# B&R Automation Studio project TD52 (part 114)

### Module_HA_IO.var - HalIO IO variables
```iecst
(********************************************************************
* COPYRIGHT -- INNIO Company
********************************************************************
* Package: HAL_IO
* File: HAL_IO.var
* Author: Automatically generated code
* Created: 29.01.2014
* corrected version from 04.09.2017
*********************************************************************
* Variables of package HAL_IO
********************************************************************)
VAR
	EO_FreshOilPump_Dem : BOOL; (*DO Aux FreshOilPump V4.14*)
	tEO_FreshOilPump_Dem : HALioDo_Type; (*DO Aux FreshOilPump V4.14*)
	EO_WasteOilPump_Dem : BOOL; (*DO Aux WasteOilPump V4.14*)
	tEO_WasteOilPump_Dem : HALioDo_Type; (*DO Aux WasteOilPump V4.14*)
	ActFiltAlarm : BOOL; (*DIactivfilteralarm*)
	ActFiltWarn : BOOL; (*DIactivfilterwarning*)
	Actuator2_Rel : BOOL; (*DO:Actuatorreleasecommand*)
	Actuator_Ok : BOOL; (*DI:Actuatorokay*)
	Actuator_Ok_CBV1 : BOOL; (*DI:Actuatorokaycompressorbypassvalve1*)
	Actuator_Ok_CBV2 : BOOL; (*DI:Actuatorokaycompressorbypassvalve2*)
	Actuator_Ok_TV1A : BOOL; (*DI:Actuatorokaythrottlevalve1A*)
	Actuator_Ok_TV1B : BOOL; (*DI:Actuatorokaythrottlevalve1B*)
	Actuator_Ok_TV2A : BOOL; (*DI:Actuatorokaythrottlevalve2A*)
	Actuator_Ok_TV2B : BOOL; (*DI:Actuatorokaythrottlevalve2B*)
	Actuator_Ok_DAI_A : BOOL; (* DI: Actuator ok DAI bank A *)
	Actuator_Ok_DAI_B : BOOL; (* DI: Actuator ok DAI bank B *)
	Actuator_Rel : BOOL; (*DO:Actuatorreleasecommand*)
	AirER_FS : BOOL; (*DIengineroomVEflowswitch*)
	AI_UniAi : ARRAY[0..250] OF INT; (*CustomerIOsystemHAL-connector*)
	AuxErrWarn : BOOL; (*DIauxiliarieserror*)
	AuxFail : BOOL; (*DIauxilariesfailure*)
	AuxOverVoltProt_Ok : BOOL; (*failureovervoltageprotectionauxiliariespowersupply*)
	AuxPoSuMains : BOOL; (*DOauxiliariespowersupplyfrommains*)
	AuxPoSuUPS : BOOL; (*DOauxiliariespowersupplyfromUPS*)
	AuxV_Eng_ok : BOOL; (*DIauxiliariesvoltageengineok*)
	ChC_Heating : BOOL; (*DO Demand charge cooler pre heating*)
	Island_Op : BOOL; (*DO Island operation*)
	Parallel_Op : BOOL; (*DO Mains parallel operation*)
	AuxV_Supply_Ok : BOOL; (*DIauxiliaryvoltagesupplyok*)
	BbBlower : BOOL; (*DO Blow-by Blower*)
	BbBlower_FC_Rdy : BOOL; (*DI Blow-by Blower FC ready *)
	BbBlower_y : INT; (*AO Blow-by Blower Percentage value to FU*)
	BB_Alive : BOOL; (*DIbusbaralive*)
	BB_Dead_MMD : ARRAY[0..2] OF BOOL; (*DIbusbardeadfromMMD*)
	bCAsymDO1 : ARRAY[0..2] OF BOOL; (*Set function of MMDsynch DO1 terminal*)
	bCNMaxDO1 : ARRAY[0..2] OF BOOL; (*Set function of MMDsynch DO1 terminal*)
	bCThermDO1 : ARRAY[0..2] OF BOOL; (*Set function of MMDsynch DO1 terminal*)
	bMMDReadyDO1 : ARRAY[0..2] OF BOOL; (*Set function of MMDsynch DO1 terminal*)
	bOFreqDO1 : ARRAY[0..2] OF BOOL; (*Set function of MMDsynch DO1 terminal*)
	bOVoltDO1 : ARRAY[0..2] OF BOOL; (*Set function of MMDsynch DO1 terminal*)
	bReactMinDO1 : ARRAY[0..2] OF BOOL; (*Set function of MMDsynch DO1 terminal*)
	bShortDO1 : ARRAY[0..2] OF BOOL; (*Set function of MMDsynch DO1 terminal*)
	bSyncCheckMode : ARRAY[0..2] OF BOOL; (*sync mode: check*)
	bSyncDeadBusMode : ARRAY[0..2] OF BOOL; (*sync mode: dead bus*)
	bSyncSlipMode : ARRAY[0..2] OF BOOL; (*sync mode: slip*)
	bUFreqDO1 : ARRAY[0..2] OF BOOL; (*Set function of MMDsynch DO1 terminal*)
	bUVolt2DO1 : ARRAY[0..2] OF BOOL; (*Set function of MMDsynch DO1 terminal*)
	bUVoltDO1 : ARRAY[0..2] OF BOOL; (*Set function of MMDsynch DO1 terminal*)
	bVAsymDO1 : ARRAY[0..2] OF BOOL; (*Set function of MMDsynch DO1 terminal*)
	CA_IgnP_Set : INT; (*AO:timingpoint*)
	CCWP_Op : BOOL; (*DIchargecoolingwaterpumpoperating*)
	ChargeOff_Dem : BOOL; (*DOchargingunitoffdemand*)
	ChC_DemFan1 : BOOL; (*DOchargecoolerdemandfan1*)
	ChC_DemFan2 : BOOL; (*DOchargecoolerdemandfan2*)
	ChC_DemFan3 : BOOL; (*DOchargecoolerdemandfan3*)
	ChC_DemFan4 : BOOL; (*DOchargecoolerdemandfan4*)
	ChC_DemFan5 : BOOL; (*DOchargecoolerdemandfan5*)
	ChC_DemFan6 : BOOL; (*DOchargecoolerdemandfan6*)
	ChC_DemFan7 : BOOL; (*DOchargecoolerdemandfan7*)
	ChC_DemFan8 : BOOL; (*DOchargecoolerdemandfan8*)
	ChC_DemFan9 : BOOL; (*DOchargecoolerdemandfan9*)
	ChC_DemFan10 : BOOL; (*DOchargecoolerdemandfan10*)
	ChC_DemFan11 : BOOL; (*DOchargecoolerdemandfan11*)
	ChC_DemFan12 : BOOL; (*DOchargecoolerdemandfan12*)
	ChC_DemFan13 : BOOL; (*DOchargecoolerdemandfan13*)
	ChC_DemFan14 : BOOL; (*DOchargecoolerdemandfan14*)
	ChC_DemFan15 : BOOL; (*DOchargecoolerdemandfan15*)
	ChC_DemFan16 : BOOL; (*DOchargecoolerdemandfan16*)
	ChC_DemPump : BOOL; (*DOchargecoolerdemandpump*)
	ChC_Failure : BOOL; (*DIchargecoolerfailure*)
	ChC_FanRdy : BOOL; (*DIchargecoolerfanready*)
	ChUnit1_CB_On : BOOL; (*Circuit breaker tripped Charging unit 1*)
	ChUnit2_CB_On : BOOL; (*Circuit breaker tripped Charging unit 2*)
	ChUnit3_CB_On : BOOL; (*Circuit breaker tripped +ENGIA Charging unit 1*)
	ChUnit4_CB_On : BOOL; (*Circuit breaker tripped +ENGIA Charging unit 2*)
	Cnt_GasImp : BOOL; (*DI	Impulsegascounter*)
	Cnt_OilPulse : BOOL; (*DIoilcounter*)
	Cnt_Oil_DC2395 : UINT; (*AIoilcountercircularbuffer*)
	Cnt_Oil_NC150 : INT; (*AIoilcounter*)
	CO2_Alarm : BOOL; (*DOCO2alarm*)
	CO2_Demand : BOOL; (*DICO2demand*)
	CO2_DemCodinox : BOOL; (*DOCO2demandCODINOX*)
	CO2_DevFailure : BOOL; (*DICO2devicefailure*)
	CO2_FanCoOn : BOOL; (*DOCO2demandfan*)
	CO2_FanFailure : BOOL; (*DICO2fanfailure*)
	CO2_MPMode : BOOL; (*DOCO2setCODINOXtomainsparallelmode*)
	CO2_Rdy : BOOL; (*DOCO2ready*)
	CO2_VaClosed : BOOL; (*DICO2valveclosed*)
	CO2_VaCoClose : BOOL; (*DOCO2valvecommandclose*)
	CO2_VaCoOpen : BOOL; (*DOCO2valvecommandopen*)
	CO2_VaFailure : BOOL; (*DICO2valvefailure*)
	CO2_VaLockout : BOOL; (*DIlockoutCO2valve*)
	CO2_VaOpened : BOOL; (*DICO2valveopened*)
	CO2_WD : BOOL; (*DOCO2watchdog*)
	Codinox_Rdy : BOOL; (*DICODINOXreadyforoperation*)
	CO_Alarm : BOOL; (*DICOalarm*)
	CO_PreAlarm : BOOL; (*DICOprealarm*)
	CP_CBTrip : BOOL; (*DImoduleand/orinterfacecontrolpanel-circuitbreakertripped*)
	CtrGenPF_Set : INT; (*AOGenerator???*)
	CtrTR_Heater_Set : INT; (*AO->Controlleroutput*)
	Ctr_ChCHP_Set : INT; (*AOchargetemperaturecoolerhighpressurecontrolvalve*)
	Ctr_ChCV_Set : INT; (*AOchargetemperaturecoolerventilation*)
	Ctr_ChC_Set : INT; (*AOchargetemperaturecoolercontrolvalve*)
	Ctr_CustOut : ARRAY[0..45] OF INT; (*AI: new output channel für direct usage of customized controllers on HAL*)
	Ctr_ECW_Set : INT; (*AOenginecoolingewatertemp.controlvalvesetpoint*)
	Ctr_EC_Set : INT; (*AOheatwaterreturntemperaturecontrolvalveemergencycooler*)
	Ctr_GC_Set : INT; (*AO Gas compressor*)
	Ctr_Gen_Set : INT; (*AOGenerator???*)
	Ctr_HWRe_Set : INT; (*AOheatwaterreturntemperaturecontrolvalve*)
	Ctr_HWSu_Set : INT; (*AOheatwatersupplytemperaturecontrolvalve*)
	CustAnaIn : ARRAY[0..120] OF INT; (*ReplacementforRAN_KANAL...*)
	CustAnaOut : ARRAY[0..60] OF INT; (*newreserveoutputchannel(likeANA.RAN1forinputs)*)
	CustDigIn : ARRAY[0..200] OF BOOL; (*new,reservedforProjectspecificuse*)
	CustDigOut : ARRAY[0..150] OF BOOL; (*ConnectiontoHAL*)
	P0_BLOCK_DEIE : BOOL; (*DI : Installed 1/0 switch *) (*OldName:Cust_switch_erdf PV;Cycle:2;*)
	CV_Eng_Low : BOOL; (*Control voltage min*)
	CV_TCA_Low : BOOL; (*Control voltage min*)
	C_CB_EDC : BOOL; (*DIcustomercircuitbreaker(engine*)
	C_CB_ESL : BOOL; (*DIcustomercircuitbreaker(engine*)
	C_CB_Off : BOOL; (*DIcustomercircuitbreakeropened*)
	C_CB_On : BOOL; (*DIcustomercircuitbreakerclosed*)
	DAI_V_Dem : BOOL; (* DO: DAI shut off valve open command *)
	DAI_V_Opened : BOOL; (* DI: DAI shut off valve position opened *)
	DAI_V_Closed : BOOL; (* DI: DAI shut off valve position closed *)
	DAI_Dem : BOOL; (*DO: Demand DAI actuator bank A and B *)
	Pos_DAI_Set_A : INT; (* AO: Position setpoint DAI control valve bank A *)
	Pos_DAI_Act_A : INT; (* AI: Position feedback DAI control valve bank A *)
	Pos_DAI_Set_B : INT; (* AO: Position setpoint DAI control valve bank B *)
	Pos_DAI_Act_B : INT; (* AI: Position feedback DAI control valve bank B *)
	DAI_CB_On : BOOL; (* DAI curcuit breaker feedback signal *)
	DemandBB : BOOL; (*demandbusbar*)
	DemEngOpExt : BOOL; (*externaldemandofengineoperation*)
	DemFlair : BOOL; (*DI	Demandgascompressorforflairoperationmode*)
	DemPurgeER : BOOL; (*DOdemandroomVEforpurgecycle*)
	DiffPrct : BOOL; (*DI:Differentialprotection*)
	DI_Dem_EU_Block : BOOL; (*externalrequestfromutility(evu*)
	DI_Dem_P_Red_EVU_Stage1 : BOOL; (*externalrequestfromutility(evu*)
	DI_Dem_P_Red_EVU_Stage2 : BOOL; (*externalrequestfromutility(evu*)
	DI_Dem_P_Red_EVU_Stage3 : BOOL; (*externalrequestfromutility(evu*)
	DI_Dem_P_Red_EVU_Stage4 : BOOL; (*externalrequestfromutility(external,vintagestyledutilisation*)
	DI_Dem_P_Red_EVU_Stage5 : BOOL; (*externalrequestfromutility(external,vintagestyledutilisation*)
	DI_UniDi : ARRAY[0..250] OF BOOL; (*CustomerIOsystemHAL-connector*)
	DO_Eng_Block_EVU : BOOL; (*acknowlegerequestfromutility(evu*)
	DO_P_Red_EVU_Stage0 : BOOL; (*acknowlegerequestfromutility(evu*)
	DO_P_Red_EVU_Stage1 : BOOL; (*acknowlegerequestfromutility(evu*)
	DO_P_Red_EVU_Stage2 : BOOL; (*acknowlegerequestfromutility(evu*)
	DO_P_Red_EVU_Stage3 : BOOL; (*acknowlegerequestfromutility(evu*)
	DO_P_Red_EVU_Stage4 : BOOL; (*acknowlegerequestfromutility(external,vintagestyledutilisationfeedback*)
	DO_P_Red_EVU_Stage5 : BOOL; (*acknowlegerequestfromutility(external,vintagestyledutilisationfeedback*)
	DPr_AirFilt : INT; (*engineairinletfilterdifferencepressure[bar]*)
	DPr_AirFilt_A : INT; (*engineairinletfilterdifferencepressureA[bar]*)
	DPr_AirFilt_B : INT; (*engineairinletfilterdifferencepressureB[bar]*)
	DPr_InAirFiltERV_Hi : BOOL; (*air inlet filter difference pressure high - engine room ventilation*) (*V04.04.00.00*)
	DPr_OilSkid_FiltHP_DE_Hi : BOOL; (*DI OilSkid heater - circuit breaker*)
	DPr_OilSkid_FiltHP_NDE_Hi : BOOL; (*DI OilSkid difference pressure - oil high pressure filter to NDE bearing*)
	DPr_OilSkid_FiltLP_Hi : BOOL; (*DI OilSkid difference pressure - oil low pressure filter*)
	EarthCB_Off : BOOL; (*DIearthcircuitbreakeropened,francecountryspecific*)
	ECWP1Dem : BOOL; (*DOenginecoolingwaterpump1demand*)
	ECWP2Dem : BOOL; (*DOenginecoolingwaterpump2demand*)
	ECWPrehV_Opened : BOOL; (*DIenginecoolingwaterpreheatingvalveopened*)
	ECWP_FC_Rdy : BOOL; (*DIenginecoolingwaterpumpfrequencyconverterreadyforoperation*)
	ECWP_Op : BOOL; (*DIenginecoolingwaterpumpoperating*)
	ECWP_PreH_CB_On : BOOL; (*Failure Engine jacket water Preheating pump*)
	ECWP_PreH_Dem : BOOL; (*DOenginecoolingwaterpreheatingpumpdemand*)
	ECWP_Service : BOOL; (*Service Pump Engine jacket water*)
	ECWP_Service_CB_On : BOOL; (*Failure Service Pump Engine jacket water*)
	ECWP_Service_COn : BOOL; (*Demand Service Pump Engine jacket water*)
	ECWV_Fail : BOOL; (*Failure Flap Preheating Engine jacket water*)
	ECW_DemBpP : BOOL; (*DOdemandenginecoolingwaterbypasspump(AMOT*)
	ECW_DemBpV : BOOL; (*DOdemandenginecoolingwaterbypassvalve(AMOT*)
	ECW_PreH1Dem : BOOL; (*DOenginecoolingwaterpreheating1demand*)
	ECW_PreH2Dem : BOOL; (*DOenginecoolingwaterpreheating2demand*)
	ECW_PreH3Dem : BOOL; (*DOenginecoolingwaterpreheating3demand*)
	ECW_PreHV_Closed : BOOL; (*DIenginecoolingwaterpreheatingvalvestatusclosed*)
	ECW_PreHV_CoClose : BOOL; (*DOenginecoolingwaterpreheatingvalve-commandclose*)
	ECW_PreHV_CoOpen : BOOL; (*DOenginecoolingwaterpreheatingvalve-commandopen*)
	ECW_PreHV_Opened : BOOL; (*DIenginecoolingwaterpreheatingvalvestatusopened*)
	ECW_PreH_Dem : BOOL; (*DOenginecoolingwaterpreheatingdemand*)
	EC_DemFan1 : BOOL; (*DOemergencycoolerdemandfan1*)
	EC_DemFan2 : BOOL; (*DOemergencycoolerdemandfan2*)
	EC_DemFan3 : BOOL; (*DOemergencycoolerdemandfan3*)
	EC_DemFan4 : BOOL; (*DOemergencycoolerdemandfan4*)
	EC_DemFan5 : BOOL; (*DOemergencycoolerdemandfan5*)
	EC_DemFan6 : BOOL; (*DOemergencycoolerdemandfan6*)
	EC_DemFan7 : BOOL; (*DOemergencycoolerdemandfan7*)
	EC_DemFan8 : BOOL; (*DOemergencycoolerdemandfan8*)
	EC_DemFan9 : BOOL; (*DOemergencycoolerdemandfan9*)
	EC_DemFan10 : BOOL; (*DOemergencycoolerdemandfan10*)
	EC_DemFan11 : BOOL; (*DOemergencycoolerdemandfan11*)
	EC_DemFan12 : BOOL; (*DOemergencycoolerdemandfan12*)
	EC_DemFan13 : BOOL; (*DOemergencycoolerdemandfan13*)
	EC_DemFan14 : BOOL; (*DOemergencycoolerdemandfan14*)
	EC_DemFan15 : BOOL; (*DOemergencycoolerdemandfan15*)
	EC_DemFan16 : BOOL; (*DOemergencycoolerdemandfan16*)
	EC_DemPump : BOOL; (*DOemergencycoolerdemandpump*)
	EC_Failure : BOOL; (*DIemergencycoolerfailure*)
	EGScavStart_Ext : BOOL; (*DIexhaustgasscavengingstartfromexternal*)
	EG_BoVaClosed : BOOL; (*DIexhaustgasboilervalveclosed*)
	EG_BoVaClosedTo : BOOL; (*DIexhaustgasboilervalveclosedtorch*)
	EG_BoVaCoClose : BOOL; (*DOexhaustgasboilervalvecommandclose*)
	EG_BoVaCoOpen : BOOL; (*DOexhaustgasboilervalvecommandopen*)
	EG_BoVaFailure : BOOL; (*DIexhaustgasboilervalvefailure*)
	EG_BoVaOpened : BOOL; (*DIexhaustgasboilervalveopened*)
	EG_BypassDemand : BOOL; (*DIdemandexhaustgasbypass*)
	EG_ByVaClosed : BOOL; (*DIexhaustgasbypassvalveclosed*)
	EG_ByVaClosedTo : BOOL; (*DIexhaustgasbypassvalveclosedtorch*)
	EG_ByVaCoClose : BOOL; (*DOexhaustgasbypassvalvecommandclose*)
	EG_ByVaCoOpen : BOOL; (*DOexhaustgasbypassvalvecommandopen*)
	EG_ByVaFailure : BOOL; (*DIexhaustgasbypassvalvefailure*)
	EG_ByVaOpened : BOOL; (*DIexhaustgasbypassvalveopened*)
	EleStarter_Dem : BOOL; (*DOelectricstarterdemand*)
	EmStop_MC : BOOL; (*DI emergency stop push button - module control panel (+A/+MC)*) (* *) (*V04.04.00.00*)
	EmStop_M : BOOL; (*DI emergency stop push button - module interface panel (+M)*) (* *) (*V04.04.00.00*)
	EmStop_ST : BOOL; (*DI emergency stop push button - master control panel (+ST)*) (* *) (*V04.04.00.00*)
	EmStop_IS : BOOL; (*DI emergency stop push button - interlock panel (+IS)*) (* *) (*V04.04.00.00*)
	EmStop_TS : BOOL; (*DI emergency stop push button - thermal reactor control panel (+TS)*) (* *) (*V04.04.00.00*)
	EmStop_GENI : BOOL; (*DI emergency stop push button - generator interface panel (+GENI)*) (* *) (*V04.04.00.00*)
	EmStop_ENGIA : BOOL; (*DI emergency stop push button - engine interface panel bank A (+ENGIA)*) (* *) (*V04.04.00.00*)
	EmStop_TCMI : BOOL; (*DI emergency stop push button - turbocharger module interface panel (+TCMI)*) (* *) (*V04.04.00.00*)
	EmStop_JWMI : BOOL; (*DI emergency stop push button - jacket water module interface panel (+JWMI)*) (* *) (*V04.04.00.00*)
	EmStop_OILMI : BOOL; (*DI emergency stop push button - oil module interface panel (+OILMI)*) (* *) (*V04.04.00.00*)
	EmStop_SCR : BOOL; (*DI emergency stop push button - exhaust gas after treatment control panel (+SCR)*) (* *) (*V04.04.00.00*)
	EmStop_TCMSCAV : BOOL; (*DI emergency stop push button - exhaust gas scavenging system (+TCMSCAV)*) (* *) (*V04.07.00.00*)
	EngDemIsland : BOOL; (*DIenginedemandforislandoperation*)
	ENGIA_UPS_CB_On : BOOL; (*Circuit breaker tripped supply UPS +TCAI --> +ENGIA*)
	EngStartFailure : BOOL; (*DIenginestartfailure*)
	EngTurn : BOOL; (*DIengineturnequipmentactive*)
	EngTurn2 : BOOL; (*Failure engine turning device*)
	Eng_Aux_Dem_CDR : BOOL; (*engineauxiliariesdemandwithcooldownrun*)
	Eng_Aux_Dem_CDR2 : BOOL; (*engineauxiliariesdemandwithcooldownrun*)
	Eng_Aux_Dem_CDR3 : BOOL; (*engineauxiliariesdemandwithcooldownrun*)
	Eng_Dem : BOOL; (*enginedemandedforMSY*)
	Eng_Dem_EPS_Ext : BOOL; (*enginedemandemergencypowersupplyfromexternal*)
	Eng_Rdy_Rem : BOOL; (*ReadyforRemoteOperation*)
	Eng_Ready : BOOL; (* DO: aggregate available (PLC run) 							*)
	Eng_Run : BOOL; (*enginerunning*)
	Eng_Run_Sy : BOOL; (*engineruning-synchronization*)
	Eng_SUExc_Rel : BOOL; (*start-upexcitationrelease*)
	EOF_DiffMax : BOOL; (*DI:Oildifferencepressuremaximum*)
	EOF_PreheatRel : BOOL; (*DO:Releaseoilpreheatingvalve*)
	EOP1AC_CB_trip : BOOL; (*DIengineoilpump1ACcircuitbreakertrip*)
	EOP1AC_Dem : BOOL; (*DOengineoilpump1AC*)
	EOP1DC_Dem : BOOL; (*DOengineoilpump1DC*)
	EOP_DemExt : BOOL; (*DIengineoilpumpdemandfromexternal*)
	EOP_FC_Rdy : BOOL; (*DI:engineoilpumpfreq.converteroperation/ready*)
	EOP_FC_Set : INT; (*AO:Setpointfrequencyconvertermotoroilpumpprelubrication,[100%=1.0]*)
	EOP_On : BOOL; (*DO:Engineoilpump,NPO602*)
	EOP_Op : BOOL; (*DIengineoilpumpoperating*)
	EOVal_DemOpen : BOOL; (*DOengineoilrefillvalvedemandopen*)
	EOVal_LT_Set : INT; (*Control signal Regulator valve NT Oil circuit*)
	EO_Level : INT; (*EngineOilPanLevel*)
	EO_Level_Hi : BOOL; (*DIengineoillevelhighfromlevelswitch*)
	EO_Level_Lo : BOOL; (*DIengineoillevellowfromlevelswitch*)
	EO_Preheat1 : BOOL; (*DO:engineoilpreheatingelement1*)
	EO_Preheat2 : BOOL; (*DO:engineoilpreheatingelement2*)
	EO_Preheat3 : BOOL; (*DO:engineoilpreheatingelement3*)
	EO_Quality : INT; (*AI:Oilqualitysensor,QTOil1/AI_*)
	EO_Refill : BOOL; (*DIengineoilrefillONfromlevelswitch*)
	EO_Supply_Fail : BOOL; (*DI:Oilsupplyfailure*)
	ERDF_BLOCK : BOOL; (* DO: Block von ERDF *) (* OldName: DI_EVU_BLOCK ; Cycle: 5 *)
	ERV_Op : BOOL; (*DIengineroomventilationoperating/airflowok*)
	ERV_InlAir_Op : BOOL; (*DIengineroominletairventilationoperating/airflowok*)
	ERV_OutlAir_Op : BOOL; (*DIengineroomoutletairventilationoperating/airflowok*)
	ER_DoorClosed : BOOL; (*DI engine room doors closed*)
	ER_Ext_Err : BOOL; (*DIengineroomVEfailure*)
	ER_InlAir_Ext_Err : BOOL; (*DIengineroominletairVEfailure*)
	ER_OutlAir_Ext_Err : BOOL; (*DIengineroomoutletairVEfailure*)
	ER_FC_Set : INT; (*AOengineroomfrequencyconvertersetpoint[%]*)
	EU_RM_BLOCK : BOOL; (*DO:	Separateunitofutilityandofactivenetwork*)
	EVU_PowerSet3Dem : BOOL; (*demandmoduleblockedbyutility*)
	ExCo_Rel : BOOL; (*DOexternalcoolerrelease*)
	FastAO_KN_A : INT; (*fastanalogoutputsignalsforvalidation*)
	FastAO_KN_B : INT; (*fastanalogoutputsignalsforvalidation*)
	FireAlarm : BOOL; (*DIfirealarm*)
	FlairRdy : BOOL; (*DI	Flairready*)
	Flow_Gen_Lube : BOOL; (*generatorlubricationfailure*)
	Flow_HW_Lo : BOOL; (*DIheatwaterflowlow*)
	Flow_OilSkid_DE : INT; (*AI OilSkid oil flow to DE bearing *)
	Flow_OilSkid_NDE : INT; (*AI OilSkid oil flow to NDE bearing (G.03-FI-003)*)
	FS_ECW : BOOL; (*DIflowswitchenginecoolingwater*)
	F_GenBear_DE1 : INT; (*vibration generator bearing drive end 1*) (*Oldname:AI_v_GenBearDE1;Cycle:5;*)
	F_GenBear_DE2 : INT; (*vibration generator bearing drive end 2*) (*Oldname:AI_v_GenBearDE2;Cycle:5;*)
	F_GenBear_NDE1 : INT; (*vibration generator bearing non drive end 1*) (*Oldname:AI_v_GenBearNDE1;Cycle:5;*)
	F_GenBear_NDE2 : INT; (*vibration generator bearing non drive end 2*) (*Oldname:AI_v_GenBearNDE2;Cycle:5;*)
	F_MMD : ARRAY[0..2] OF UINT; (* frequency multi measure device*)
	F_MMD_LimHi : ARRAY[0..2] OF BOOL; (*generatorfrequencytoohigh*)
	F_MMD_LimLo : ARRAY[0..2] OF BOOL; (*generatorfrequencytoolow*)
	F_MMD_Synch1 : ARRAY[0..2] OF UINT; (* Frequency Sync-network 1 *)
	F_MMD_Synch2 : ARRAY[0..2] OF UINT; (* Frequency Sync-network 2 *)
	F_N_DI_Dec : BOOL; (*synch.digitalindecreasespeed*)
	F_N_DI_Inc : BOOL; (*synch.digitalinincreasespeed*)
	GasAlarm : BOOL; (*DIgasalarm*)
	GasPreAlarm : BOOL; (*DIgasprealarm*)
	GCB_AGO : BOOL; (*DIallothergeneratorcircuitbreakeroff*)
	GCB_COf : BOOL; (*commandgcboff*)
	GCB_COn : BOOL; (*commandgcbon*)
	GCB_DRM : BOOL; (*DIgeneratorcircuitbreakerdemandMCBclosingreturntomains*)
	GCB_DSY : BOOL; (*DIgeneratorcircuitbreakerdemandsynchronization(synchline*)
	GCB_DVM : BOOL; (*voltagematchingforsynchronization*)
	GCB_DVS : BOOL; (*generatorcircuitbreakerdemandvoltageselection*)
	GCB_Earth : BOOL; (*DIgeneratorcircuitbreakerpositionearth*)
	GCB_EDC : BOOL; (*generatorcircuitbreakerenginedemandclose*)
	GCB_ESL : BOOL; (*generatorcircuitbreakerstatuslocked*)
	GCB_MDL : BOOL; (*DIgeneratorcircuitbreakermasterdemandlock(forclosingotherGCBtodeadBB*)
	GCB_MRC : BOOL; (*DIgeneratorcircuitbreakermasterreleaseclose(todeadbusbar*)
	GCB_Off : BOOL; (*DIgeneratorcircuitbreakeropened*)
	GCB_OGP : BOOL; (*DIgeneratorcircuitbreakerothergeneratorparallel*)
	GCB_On : BOOL; (*generatorcircuitbreakerclosed*)
	GCB_On_ReturnSign : BOOL; (*ReleaseforUnitrolAVR*)
	GCB_OpF : BOOL; (*generatorcircuitbreakeropeningfailure*)
	GCB_Rac : BOOL; (*DIgeneratorcircuitbreakerrackedin*)
	GCB_Rdy : BOOL; (*DIgeneratorcircuitbreakerready(forclose*)
	GCB_Rel : BOOL; (*generatorcircuitbreakerreleaseclosing*)
	GCB_RI : BOOL; (*DIgeneratorcircuitbreakerreelaseisland*)
	GCB_RSP : BOOL; (*generatorcircuitbreakerreleasesynchpulse*)
	GCB_RT : BOOL; (*generatorcircuitbreakerreleasetrip*)
	GCB_RUC : BOOL; (*generatorcircuitbreakerreleaseundervoltagecoil*)
	GCB_SM1 : BOOL; (*DIgeneratorcircuitbreakeroutputsignalmonitoring1*)
	GCB_SM2 : BOOL; (*DIgeneratorcircuitbreakercontactsignalmonitoring2*)
	GCB_SOn : BOOL; (* DO: Generator switch is on 									*)
	GenCtrResetSp : BOOL; (*Generator controller reset setpoint*)
	GenCtr_CktBkr_Trip : BOOL; (*generatorcicuitbreakeroff*)
	GenDeexitDem : BOOL; (*DOgeneratordeexitationdemand*)
	GenIF_CB_On : BOOL; (*Circuit breaker tripped supply +TCAI --> +GENI*)
	GenPrctTrip : BOOL; (*DI:Generatorprotectiontrip*)
	Gen_DVM : BOOL; (*Generatorvoltagematchingoutput(LeroySomer*)
	Gen_Exc_Off : BOOL; (*de-excitation*)
	Gen_LO_CoolingSys_Fail : BOOL; (*generatorlubeoilcoolingsystemfailure*)
	Gen_PreHDem : BOOL; (*DOGeneratorpreheatdemand*)
	Gen_RVM : BOOL; (*DIgeneratorreleasevoltagematching(leroysomer*)
	Gen_T_In : INT; (*actualvaluegeneratorinlettemperature*)
	Gen_T_In2 : INT; (*actualvaluegeneratorinlettemperature2*)
	GF_OilSystem : BOOL; (*DI general failure oil system*) (*OldName:newPV; Cycle:5*) (*STM*)
	GndFailure : BOOL; (*DI:earthfailure*)
	GnlTrip : BOOL; (*DOenginegeneraltrip*)
	GnlWarning : BOOL; (*DOenginegeneralwarning*)
	GrC_DCon : BOOL; (* DO: FALSE = Disconnect from Grid due to GridCode Event*)
	GT1_1_SafeDevice : BOOL; (*DO	Gassafetydevice1line1*)
	GT1_1_SafeDevOK : BOOL; (*DIGassafetydevice1line1*)
	GT1_2_SafeDevice : BOOL; (*DO	Gassafetydevice1line2*)
	GT1_2_SafeDevOK : BOOL; (*DI	Gassafetydevice2line2*)
	GT1_3_SafeDevice : BOOL; (*DO	Gassafetydevice1line3*)
	GT1_3_SafeDevOK : BOOL; (*DIGassafetydevice3line3*)
	GT1_4_SafeDevice : BOOL; (*DO	Gassafetydevice1line4*)
	GT1_4_SafeDevOK : BOOL; (*DIGassafetydevice4line4*)
	GT1_SafeDevice : BOOL; (*DO	Gassafetydevice1*)
	GT1_SafeDevOK : BOOL; (*DI	Gassafetydevice1*)
	GT2_SafeDevice : BOOL; (*DO	Gassafetydevice2*)
	GT2_SafeDevOK : BOOL; (*DI	Gassafetydevice2*)
	GT3_SafeDevOK : BOOL; (*DI	Gassafetydevice3*) (*SAFETY PLC*) (*V04.14.00.00*)
	GT4_SafeDevOK : BOOL; (*DI	Gassafetydevice4*) (*SAFETY PLC*) (*V04.14.00.00*)
	GT_AirSupply_LoLo : BOOL; (*DI FALSE = compressed air supply pressure for gas train too low - error*) (*Oldname : DI_GT_AirSupply_LoLo Cyclic: 2; *)
	GT1_1_BackFireDev : BOOL; (*DIAntibackfiredevice1line1*)
	GT1_2_BackFireDev : BOOL; (*DIAntibackfiredevice1line2*)
	GT1_3_BackFireDev : BOOL; (*DIAntibackfiredevice1line3*)
	GT1_4_BackFireDev : BOOL; (*DIAntibackfiredevice1line4*)
	PCbComp_BackFireDev : BOOL; (*DIAntibackfire device prechamper before compressor*)
	PCaComp_BackFireDev : BOOL; (*DIAntibackfire device prechamper after compressor*)
	GT_BackFireDev : BOOL; (*DI	Antibackfiredevice*)
	GT_CalibrateActive : BOOL; (*DI	CalibrationGasanalysis*)
	GT_CH4 : INT; (*IF653CH4content	*)
	GT_CV : INT; (*AI	Calorificvalue*)
	GT_FlairFail : BOOL; (*DI	Flarefailure*)
	GT_Flap1_Close : BOOL; (*DO	Closegasflap1*)
	GT_Flap1_Closed : BOOL; (*DI	Gasflap1closed(Feedback*)
	GT_Flap1_Open : BOOL; (*DO	Opengasflap1*)
	GT_Flap1_Opened : BOOL; (*DI	Gasflap1opened(Feedback*)
	GT_Flap2_Close : BOOL; (*DO	Closegasflap2*)
	GT_Flap2_Closed : BOOL; (*DI	Gasflap2closed(Feedback*)
	GT_Flap2_Open : BOOL; (*DO	Opengasflap2*)
	GT_Flap2_Opened : BOOL; (*DI	Gasflap2opened(Feedback*)
	GT_FlareOpMod : BOOL; (*DI	Flareinoperationalmode*)
	GT_GC_Dem : BOOL; (*DO	Demandgascompressor*)
	GT_GC_Fail : BOOL; (*DI	Gascompressorfailure*)
	GT_O2 : INT; (*IF656O2content	*)
	GT_RelFlair : BOOL; (*DO	Releaseflare*)
	GT_SelectRatioMix : BOOL; (*DI: Digital input to select gas mixing (1-3 or 1_2-3)*)
	GT_TypSwitch : BOOL; (*DI	Gastypeswitchtosecondgas*)
	GV1Mega_Open : BOOL; (*DO	Openmegagasvalve1*)
	GV1_1_Open : BOOL; (*DO	opengasvalve1_1(GASV1_1*)
	GV1_2_Open : BOOL; (*DO	opengasvalve1_1(GASV1_2*)
	GV1_Open : BOOL; (*DO	opengasvalve1*)
	GV2Mega_Open : BOOL; (*DO	Openmegagasvalve2*)
	GV2_Open : BOOL; (*DO	opengasvalve2*)
	GV3_Open : BOOL; (*DO	opengasvalve3*) (*SAFETY PLC*) (*V04.14.00.00*)
	GV4_Open : BOOL; (*DO	opengasvalve4*) (*SAFETY PLC*) (*V04.14.00.00*)
	GT1_GV1_Open : BOOL; (*DO Gastrain1 - Gasvalve 1*) (*SAFETY PLC*) (*V04.14.00.00*)
	GT1_GV2_Open : BOOL; (*DO Gastrain1 - Gasvalve 2*) (*SAFETY PLC*) (*V04.14.00.00*)
	GT2_GV1_Open : BOOL; (*DO Gastrain2 - Gasvalve 1*) (*SAFETY PLC*) (*V04.14.00.00*)
	GT2_GV2_Open : BOOL; (*DO Gastrain2 - Gasvalve 2*) (*SAFETY PLC*) (*V04.14.00.00*)
	GT3_GV1_Open : BOOL; (*DO Gastrain3 - Gasvalve 1*) (*SAFETY PLC*) (*V04.14.00.00*)
	GT3_GV2_Open : BOOL; (*DO Gastrain3 - Gasvalve 2*) (*SAFETY PLC*) (*V04.14.00.00*)
	GT4_GV1_Open : BOOL; (*DO Gastrain4 - Gasvalve 1*) (*SAFETY PLC*) (*V04.14.00.00*)
	GT4_GV2_Open : BOOL; (*DO Gastrain4 - Gasvalve 2*) (*SAFETY PLC*) (*V04.14.00.00*)
	GV_Rel : BOOL; (*DO	Releasegasvalves*)
	Horn : BOOL; (*DOhorn*)
	Horn_Trip : BOOL; (*DOhornengineshutdown*)
	Horn_Warning : BOOL; (*DOhornwarning*)
	Humidity_AirIn : INT;
	HWP_Dem : BOOL; (*DOheatingwaterpumpdemand*)
	HWP_Op : BOOL; (*DIheatingwaterpumpoperating*)
	IFCP_CBTrip : BOOL; (*DIinterfacecontrolpanel-circuitbreakertripped*)
	Ign2_Run_Hal : BOOL; (*DI:Ignitionsystemdoublerunning*)
	Ign_Dem : BOOL; (*demandignition*)
	Ign_OverspeedRelay : BOOL; (*DI:Overspeedrelay*)
	Ign_Run_Hal : BOOL; (*DI:Ignitionsystemrunning*)
	Imp_OpHour : BOOL; (*impulseforoperationhourcounter*)
	InAirER_Fan1DemOn : BOOL; (*DOdemandairinletventilator1*)
	InAirER_Fan2DemOn : BOOL; (*DOdemandairinletventilator2*)
	InAirER_Lou1DemOpen : BOOL; (*DOdemandopenairinletlouver1*)
	InAirER_Lou1Opened : BOOL; (*DIintakeairengineroomlouver1open*)
	InAirER_Lou2DemOpen : BOOL; (*DOdemandopenairinletlouver2*)
	InAirER_Lou2Opened : BOOL; (*DIintakeairengineroomlouver2open*)
	DemERVentInLou_Cust : BOOL; (*DO inlet louvers demand for customer*)
	IsoCB_Off : BOOL; (*DIdisconnectingcircuitbreakeropened,francecountryspecific*)
	I_Avg : ARRAY[0..2] OF INT; (*IF513gen.currentaveragev.	*)
	I_Diff : BOOL; (*generatordifferentialprotectiontrip*)
	I_L1 : ARRAY[0..2] OF INT; (*PhasecurrentgeneratorI1*)
	I_L2 : ARRAY[0..2] OF INT; (*PhasecurrentgeneratorI2*)
	I_L3 : ARRAY[0..2] OF INT; (*PhasecurrentgeneratorI3*)
	I_MMD_Asy : ARRAY[0..2] OF BOOL; (*generatorcurrentnegativesequencetoohigh*)
	I_MMD_LimHi : BOOL; (*MMD:overloadshortcircuit*)
	I_MMD_Neutr_LimHi : ARRAY[0..2] OF BOOL; (*generatorneutralcurrenttoohigh*)
	KLS90_1 : INT; (*AI:KLS90sensor1signal*)
	KLS90_2 : INT; (*AI:KLS90sensor1signal*)
	Lam_Act : INT; (*actualLambdavalue*)
	LOS_Dem : BOOL; (*Generatordemandlubeoilsystem*)
	LeroySomer_AuxContactor : BOOL; (*LEROY-SOMERAuxiliaryContactor*)
	Lev_OilSkid_Sump_Hi : BOOL; (*DI OilSkid oil in safety sump *)
	Lev_OilSkid_Tank : INT; (*AI OilSkid tank level*)
	LineCB_On : BOOL; (*DIlinecircuitbreakerclosed*)
	Lock_C_MCB : BOOL; (*lockcustomermainscircuitbreaker*)
	LSL_In : INT; (*AIloadsharingline*)
	LSL_Out : INT; (*AOloadsharingline*)
	LS_Dem : BOOL; (*DOloadsheddingdemand*)
	L_ECW_Lo : BOOL; (*DIenginecoolingwaterlevellow*)
	L_ECW_LoLo : BOOL; (*DIenginecoolingwaterlevellowlow*)
	L_FreshOilTank_Lo : BOOL; (*DIfreshoiltanklevellow*)
	L_FreshOilTank_Hi : BOOL; (*DI fresh oil tank level high*) (*OldName:newPV; Cycle:5*) (*STM*)
	Leak_FreshOilPump : BOOL; (*DI leakage fresh oil pump*) (*OldName:newPV; Cycle:5*) (*STM*)
	Leak_FreshOilTank : BOOL; (*DI leakage fresh oil tank*) (*OldName:newPV; Cycle:5*) (*STM*)
	Leak_WasteOilPump : BOOL; (*DI leakage waste oil pump*) (*OldName:newPV; Cycle:5*) (*STM*)
	Leak_WasteOilTank : BOOL; (*DI leakage waste oil tank*) (*OldName:newPV; Cycle:5*) (*STM*)
	L_InMa_Hi : BOOL; (*DIwateringressintoinletmanifold*)
	L_InMa_NotHi : BOOL; (*DIwateringressintoinletmanifoldnegated*)
	L_OilSump3Hi : BOOL; (*DIleveloilsump3high*)
	L_OilSump2Hi : BOOL; (*DIleveloilsump2high*)
	L_OilSumpHi : BOOL; (*DIleveloilsumphigh*)
	L_WasteOilTank_Hi : BOOL; (*DIwasteoiltanklevelhigh*)
	MainGV_Rel : BOOL; (*DOmaingasvalverelease*)
	MainsStartDevDem : BOOL; (*DOmainsstartdevicedemand*)
	MainsStartDevFail : BOOL; (*DImainsstartdevicefailure*)
	MainsStartDevOk : BOOL; (*DImainsstartingdeviceOK*)
	MCB_COf : BOOL; (*commandmcboff*)
	MCB_COn : BOOL; (*mainscircuitbreakercomandon*)
	MCB_DcpQu_SetEUCOf : BOOL; (* DI: reset decoupling quickly from EU (ERDF) *) (*OldName:DI_RFDemMCBoff PV;Cycle:2;*)
	MCB_DcpQu_SetEUCOn : BOOL; (* DI: set decoupling quickly from EU (ERDF) *) (*OldName:DI_SFDemMCBoff PV;Cycle:2;*)
	MCB_Dcp_SetEUCOf : BOOL; (* DI: rest requirement decoupling from EU(ERDF),DIs *) (*OldName:DI_RDemandMCBoff PV;Cycle:2;*)
	MCB_Dcp_SetEUCOn : BOOL; (* DI: set requirement  decoupling from EU(ERDF),DIs *) (*OldName:DI_SDemandMCBoff PV;Cycle:2;*)
	MCB_DVS : BOOL; (*mainscircuitbreakerdemandvoltageselection*)
	MCB_EDF_SOn : BOOL; (* DO: feedback Engine off get  								*)
	MCB_Off : BOOL; (*DImainscircuitbreakeropened*)
	MCB_OL : BOOL; (*DImainscircuitbreakeroverload*)
	MCB_On : BOOL; (*SS447NetzschalterEIN*)
	MCB_Rac : BOOL; (*DImainscircuitbreakerrackedin*)
	MCB_Rdy : BOOL; (*DImainscircuitbreakerready(forclose*)
	MCB_Rel_Sync : BOOL; (* DI: release synchronization from EU(ERDF) *) (*OldName:DI_ReleaseMCBon PV;Cycle:2;*)
	MCB_Rel_Sync_SOn : BOOL; (* DO: releas decoupling quickly from EU (ERDF)  				*)
	MCB_Rem : BOOL; (*DImainscircuitbreakerremote(operatingmode*)
	MCB_RSP : BOOL; (*mainscircuitbreakerreleasesynchpulse*)
	MCB_RT : BOOL; (*mainscircuitbreakerreleasetrip*)
	MCB_SM : BOOL; (*DImainscircuitbreakersignalmonitoring*)
	MCB_SOn : BOOL; (* DO: receive requested Command form machine 					*)
	MCP_CBTrip : BOOL; (*DImodulecontrolpanel-circuitbreakertripped*)
	MGT_BOV : BOOL; (*DO BlowOff valve*) (*Oldname: DO_MGT_BOV; Cycle:5; *)
	MGT_DBOV : BOOL; (* DO Main gas train dome blow off valve *)
	MMD_FW_Version : ARRAY[0..2] OF UINT; (* program version MMD firmware *)
	MnsOk : BOOL; (*DImainsok	*)
	MnsOk_C13100 : BOOL; (*DImainsokC13.100monitoringdevice,francecountryspecific*)
	MnsOk_GTE : BOOL; (*DImainsokGTEmonitoringdevice,francecountryspecific*)
	MnsOk_TGS : BOOL; (*DImainsokTGSmonitoringdevice,francecountryspecific*)
	Mns_MDF : BOOL; (*DImainsmonitoringdevicefailure*)
	MonitoringOn : BOOL; (*DOmonitoringonpulse(safetyloop*)
	MO_PowerOverload : BOOL; (*DI:SAFI ignition power module 1 overload*)
	MO_PowerOverload2 : BOOL; (*DI:SAFI ignition power module 2 overload*)
	MO_PowerOverload3 : BOOL; (*DI:SAFI ignition power module 3 overload*)
	MO_PowerOverload4 : BOOL; (*DI:SAFI ignition power module 4 overload*)
	MO_PwrReply : BOOL; (*DI:MORIS Ignition Power Module 1 On*)
	MO_PwrReply2 : BOOL; (*DI:MORIS Ignition Power Module 2 On*)
	MO_PwrReply3 : BOOL; (*DI:MORIS Ignition Power Module 3 On*)
	MO_PwrReply4 : BOOL; (*DI:MORIS Ignition Power Module 4 On*)
	MO_PwrRequest : BOOL; (*DO:MORIS Ignition Power Module 1 Request*)
	MO_PwrRequest2 : BOOL; (*DO:MORIS Ignition Power Module 2 Request*)
	MO_PwrRequest3 : BOOL; (*DO:MORIS Ignition Power Module 3 Request*)
	MO_PwrRequest4 : BOOL; (*DO:MORIS Ignition Power Module 4 Request*)
	MO_SaftyLoop : BOOL; (*DI:MORISSavetyloopclosed*)
	N2_GV1_Closed : BOOL; (*DIN2gasvalve1closedstatus*)
	N2_GV2_Closed : BOOL; (*DIN2gasvalve2closedstatus*)
	N2_ScavGV_CoOpen : BOOL; (*DON2GasValvesvommandopen*)
	N2_ScavSigLampOn : BOOL; (*DOSignallampforscavenging*)
	N_ECWP_Set : INT; (*AOspeedenginecoolingwaterpumpsetpoint*)
	N_EngStart : BOOL; (*DOenginestartupspeedexceeded*)
	N_Set_ExtAI_Norm : INT; (*Externalspeedsetpoint*)
	N_TCHP : INT; (*highpressureturbochargerspeed[rpm]*)
	N_TCHP_A : INT; (*highpressureturbochargerspeedA[rpm]*)
	N_TCHP_B : INT; (*highpressureturbochargerspeedB[rpm]*)
	N_TCLP : INT; (*lowpressureturbochargerspeed[rpm]*)
	N_TCLP_A : INT; (*lowpressureturbochargerspeedA[rpm]*)
	N_TCLP_B : INT; (*lowpressureturbochargerspeedB[rpm]*)
	OilSkid_AuxV_Ok : BOOL; (*DI OilSkid auxiliaries voltage not available*)
	OilSkid_AuxV_Ok_UPS : BOOL; (*DI OilSkid auxiliaries voltage not available - UPS*)
	OilSkid_Fan : BOOL; (*DO OilSkid fan*)
	OilSkid_Fan_CBOk : BOOL; (*DI OilSkid fan - circuit breaker*)
	OilSkid_Heater : BOOL; (*DO OilSkid heater*)
	OilSkid_Heater_CBOk : BOOL; (*DI OilSkid heater - circuit breaker*)
	OilSkid_MCB : BOOL; (*DI OilSkid main switch auxiliaries opened*)
	OilSkid_PumpC : BOOL; (*DO OilSkid circulation pump (G.03-M-004)*)
	OilSkid_PumpC_CBOk : BOOL; (*DI OilSkid circulation pump - circuit breaker*)
	OilSkid_PumpHP : BOOL; (*DO OilSkid high pressure pump *)
	OilSkid_PumpHP_CBOk : BOOL; (*DI OilSkid high pressure pump - circuit breaker*)
	OilSkid_PumpHP_CBOk_UPS : BOOL; (*DI OilSkid high pressure pump - circuit breaker UPS*)
	OilSkid_PumpHP_DemOff : BOOL; (*DI OilSkid high pressure pump - demand OFF*)
	OilSkid_PumpHP_DemOn : BOOL; (*DI OilSkid high pressure pump - demand ON*)
	OilSkid_PumpHP_Soft : BOOL; (*DO OilSkid high pressure pump - Soft*)
	OilSkid_PumpHP_UPS : BOOL; (*DO OilSkid high pressure pump - UPS *)
	OilSkid_PumpLP : BOOL; (*DO OilSkid low pressure pump *)
	OilSkid_PumpLP_CBOk : BOOL; (*DI OilSkid low pressure pump - circuit breaker*)
	OlShortCirc : BOOL; (*DI:Overload/shortcircuit*)
	OF_FreshOilTank : BOOL; (*DI overfill prevention device fresh oil tank*) (*OldName:newPV; Cycle:5*) (*STM*)
	OF_WasteOilTank : BOOL; (*DI overfill prevention device waste oil tank*) (*OldName:newPV; Cycle:5*) (*STM*)
	OMSS_Aut : BOOL; (*operationmodeselectorswitch-AUTO*)
	OMSS_Man : BOOL; (*operationmodeselectorswitch-MANUAL*)
	OMSS_MAT : BOOL; (*operationmodeselectorswitch-MANUALAUTOTEST*)
	Only_Island : BOOL; (*DIonlyislandoperation*)
	OutAirER_LouDemOpen : BOOL; (*DOdemandopenairoutletlouver*)
	OutAirER_LouOpened : BOOL; (*DIoutletairengineroomlouveropen*)
	OV_Ctrl_Set : INT; (*AO:hightemperatureengineoilcoolersetpoint*)
	PCG_DemCoolFan : BOOL; (*DO	Prechambergascompressor,Demandcoolingventilator*)
	PCG_DemReliefValve : BOOL; (*DO	DemandReliefvalve*)
	PCG_DemValCW : BOOL; (*DO	Prechambergascompressor,Demandcoolingwatervalve*)
	PCG_GC_Fail : BOOL; (*DI	Failureprechambergascompressor*)
	PCG_GC_Oil_Min : BOOL; (*DI	prechambergascompressoroillevel*)
	PCG_GV_DelOpen : BOOL; (*DO	PrechambergasvalveswithdelayON*)
	PCG_GV_Open : BOOL; (*DO	Prechambergasvalves*)
	PCG_BPV_Open : BOOL; (*DO Pre chamber gas bypass valve*)
	PFC_SetCOf : BOOL; (*DI:primaryfrequencycontrol-off(deactivate*)
	PFC_SetCOn : BOOL; (*DI:primaryfrequencycontrol-on(activate*)
	PFC_SOf : BOOL; (*DO:primaryfrequencycontrolisoff*)
	PFC_SOn : BOOL; (*DO:primaryfrequencycontrolison*)
	PFUC_GenC_SetEUCOf : BOOL; (*DI:setpointreactivepowercharacteristicsCOS(phi*)
	PFUC_GenC_SetEUCOn : BOOL; (*DI:setpointreactivepowercharacteristicsCOS(phi*)
	QP_GenC_SetEUCOn : BOOL; (*DI:setpointreactivepowercharacteristicsQ(P)*)
	QP_GenC_SetEUCOf : BOOL; (*DI:setpointreactivepowercharacteristicsQ(P)*)
	PFUC_GenC_SOf : BOOL; (*DO:reactivepowercharacteristicsCOS(phi*)
	PFUC_GenC_SOn : BOOL; (*DO:reactivepowercharacteristicsCOS(phi*)
	QP_GenC_SOn : BOOL; (*DO:reactivepowercharacteristicsQ(P)*)
	QP_GenC_SOf : BOOL; (*DO:reactivepowercharacteristicsQ(P)*)
	PF_Act : ARRAY[0..2] OF INT; (*powerfactor,actualcosphivalue*)
	PF_AO_PF_I : INT; (*AOpowerfactorgenerator,mAsignal*)
	PF_AO_PF_U : INT; (*AO:powerfactorgenerator*)
	PF_CosPCtr_Ena : BOOL; (*powerfactorcontrollerenabled*)
	PF_CUSTGenC : INT; (*customiz:scalingvaluegenetarorpowerfactor(COSPHI*)
	PF_GenC_Act : INT; (*AO:generatorpowerfactor(COSPHI*)
	PF_GenC_Fix1SOn : BOOL; (*DO:genetarorpowerfactor(COSPHI*)
	PF_GenC_Fix2SOn : BOOL; (*DO:genetarorpowerfactor(COSPHI*)
	PF_GenC_Fix3SOn : BOOL; (*DO:genetarorpowerfactor(COSPHI*)
	PF_GenC_Fix4SOn : BOOL; (*DO:genetarorpowerfactor(COSPHI*)
	PF_GenC_Fix5SOn : BOOL; (*DO:genetarorpowerfactor(COSPHI*)
	PF_GenC_SetEU : INT; (*AI:setpointgenetarorpowerfactor(COSPHI*)
	PF_GenC_SetEUCOf : BOOL; (*DI:setpointgenetarorpowerfactor(COSPHI*)
	PF_GenC_SetEUCOn : BOOL; (*DI:setpointgenetarorpowerfactor(COSPHI*)
	PF_GenC_SetFix1EU : BOOL; (*DI:setpointgenetarorpowerfactor(COSPHI*)
	PF_GenC_SetFix2EU : BOOL; (*DI:setpointgenetarorpowerfactor(COSPHI*)
	PF_GenC_SetFix3EU : BOOL; (*DI:setpointgenetarorpowerfactor(COSPHI*)
	PF_GenC_SetFix4EU : BOOL; (*DI:setpointgenetarorpowerfactor(COSPHI*)
	PF_GenC_SetFix5EU : BOOL; (*DI:setpointgenetarorpowerfactor(COSPHI*)
	PF_GenC_SOf : BOOL; (*DO:generatorpowerfactor(COSPHI*)
	PF_GenC_SOn : BOOL; (*DO:generatorpowerfactor(COSPHI*)
	PLim_GenC_Act : BOOL; (*DO:powerlimitation(Plim*)
	PLim_GenC_SetEU : INT; (*AI:setpointpowerlimitation(Plim*)
	PLim_GenC_SetEUCOf : BOOL; (*DI:setpointpowerlimitation(Plim*)
	PLim_GenC_SetEUCOn : BOOL; (*DI:setpointpowerlimitation(Plim*)
	PLim_GenC_SetEUPFix1 : BOOL; (*DI:powerlimitationfixvalue1*)
	PLim_GenC_SetEUPFix2 : BOOL; (*DI:powerlimitationfixvalue2*)
	PLim_GenC_SetEUPFix3 : BOOL; (*DI:powerlimitationfixvalue3*)
	PLim_GenC_SetEUPFix4 : BOOL; (*DI:powerlimitationfixvalue4*)
	PLim_GenC_SetEUPFix5 : BOOL; (*DI:powerlimitationfixvalue5*)
	PLim_GenC_SOf : BOOL; (*DO:powerlimitation(Plim*)
	PLim_GenC_SOn : BOOL; (*DO:powerlimitation(Plim*)
	Pos_Act_CBV_A1 : INT; (*AI: compressor bypass valve position A1*)
	Pos_Act_CBV_A2 : INT; (*AI: compressor bypass valve position A2*)
	Pos_Act_CBV_B1 : INT; (*AI: compressor bypass valve position B1*)
	Pos_Act_CBV_B2 : INT; (*AI: compressor bypass valve position B2*)
	Pos_Act_GM1_Norm : INT; (*gasmixer1-normedactualpositionfrompotentiometer[%]*)
	Pos_Act_GM2_Norm : INT; (*gasmixer2-normedactualpositionfrompotentiometer[%]*)
	Pos_Act_TV : INT; (*AI: throttle valve bypass valve position*)
	Pos_Act_TV_A1 : INT; (*AI: throttle valve bypass valve position A1*)
	Pos_Act_TV_A2 : INT; (*AI: throttle valve bypass valve position A2*)
	Pos_Act_TV_B1 : INT; (*AI: throttle valve bypass valve position B1*)
	Pos_Act_TV_B2 : INT; (*AI: throttle valve bypass valve position B2*)
	Pos_Act_WG : INT; (*wastegatevalveposition*)
	Pos_Act_WG_A : INT; (*wastegatevalvepositionA*)
	Pos_Act_WG_B : INT; (*wastegatevalvepositionB*)
	Pos_CBV : INT; (*compressorbypassvalveposition*)
	Pos_CBV34 : INT; (*compressorbypassvalveposition*)
	Pos_CBV_A1 : INT; (*compressorbypassvalvepositionA1*)
	Pos_CBV_A2 : INT; (*compressorbypassvalvepositionA2*)
	Pos_CBV_B1 : INT; (*compressorbypassvalvepositionB1*)
	Pos_CBV_B2 : INT; (*compressorbypassvalvepositionB2*)
	Pos_Set_WG : INT; (*wastegatevalveposition*)
	Pos_Set_WG_A : INT; (*wastegatevalvepositionA*)
	Pos_Set_WG_B : INT; (*wastegatevalvepositionB*)
	Pos_SGM_Enc1 : INT; (*SGM encoder position stepper 1 [1]*)
	Pos_SGM_Enc2 : INT; (*SGM encoder position stepper 2 [1]*)
	Pos_SGM_Enc3 : INT; (*SGM encoder position stepper 3 [1]*)
	Pos_ThR_Val_In1 : BOOL; (*DI1thermalreactorflapinpositionmovedin*)
	Pos_ThR_Val_In2 : BOOL; (*DI2thermalreactorflapinpositionmovedin*)
	Pos_ThR_Val_Mid : BOOL; (*DIthermalreactorflapinmiddleposition*)
	Pos_ThR_Val_Out1 : BOOL; (*DI1thermalreactorflapinpositionmovedout*)
	Pos_ThR_Val_Out2 : BOOL; (*DI2thermalreactorflapinpositionmovedout*)
	Pos_TV : INT; (*throttlevalveposition*)
	Pos_TV_A1 : INT; (*throttlevalvepositionA1*)
	Pos_TV_A2 : INT; (*throttlevalvepositionA2*)
	Pos_TV_B1 : INT; (*throttlevalvepositionB1*)
	Pos_TV_B2 : INT; (*throttlevalvepositionB2*)
	P_Heat : INT; (*heating power engine heat water circuit*) (*STM 2*)
	P_Heat_Imp : BOOL; (*heating power engine heat water circuit impulse*) (*STM 2*)
	Pr_a_BbFilt : INT; (*AI Pressure after Blow-by filter *)
	Pr_a_BbFilt_A : INT; (*AI Pressure after Blow-by filter A*)
	Pr_a_BbFilt_B : INT; (*AI Pressure after Blow-by filter B*)
	Pr_Baro : INT; (*AI	Barometricpressure*)
	Pr_CC : INT; (*AIpressurecrankcase[bar]*)
	Pr_CCircuit_Lo : BOOL; (*DIwaterpressurecoolercircuitlow*)
	Pr_ChC_Lo : BOOL; (*DIchargecoolerwaterpressurelow*)
	Pr_Ch_P1HP : INT; (*chargepressurep1beforehighpressureTC[bar]*)
	Pr_Ch_P1HP_A : INT; (*chargepressurep1beforehighpressureTCA[bar]*)
	Pr_Ch_P1HP_B : INT; (*chargepressurep1beforehighpressureTCB[bar]*)
	Pr_Ch_P1LP_A : INT; (*charge pressure before low-pressure TC A [bar]*) (*V04.04.00.00*)
	Pr_Ch_P1LP_B : INT; (*charge pressure before low-pressure TC B [bar]*) (*V04.04.00.00*)
	Pr_Ch_P2 : INT; (*actualchargepressurebeforethrottlevalve*)
	Pr_Ch_P2s : INT; (*actualchargepressure*)
	Pr_Ch_P2s_A : INT; (*chargepressurep2'afterthrottlevalveA[bar]*)
	Pr_Ch_P2s_B : INT; (*chargepressurep2'afterthrottlevalveB[bar]*)
	Pr_Ch_P2_A : INT; (*chargepressurep2beforethrottlevalveA[bar]*)
	Pr_Ch_P2_B : INT; (*chargepressurep2beforethrottlevalveB[bar]*)
	Pr_DAI_A : INT; (*pressure before DAI control valve bank A [bar]*)
	Pr_DAI_B : INT; (*pressure before DAI control valve bank B [bar]*)
	Pr_DAI_In : INT; (*pressure before DAI shut off valve [bar]*)
	Pr_ECW : INT; (*AIpressureenginecoolingwater*)
	Pr_ECWaEng : INT; (*Cooling water pressure downstream of the engine*)
	Pr_EGaHPTC_A : INT; (* AI: Exhaust gas pressure after high-pressure turbocharger A  (M.02-PI-153) *) (* OldName: AI_M_02_PI_153	; Cyclic: 5; *)
	Pr_EGaHPTC_B : INT; (* AI: Exhaust gas pressure after high-pressure turbocharger B  (M.02-PI-253) *) (* OldName: AI_M_02_PI_253	; Cyclic: 5; *)
	Pr_EGaLPTC_A : INT; (* AI: Exhaust gas pressure after low-pressure turbocharger A  (M.02-PI-154) *) (* OldName: AI_M_02_PI_154	; Cyclic: 5; *)
	Pr_EGaLPTC_B : INT; (* AI: Exhaust gas pressure after low-pressure turbocharger B  (M.02-PI-254) *) (* OldName: AI_M_02_PI_254	; Cyclic: 5; *)
	Pr_EGbHPTC_A : INT; (* AI: Exhaust gas pressure before high-pressure turbocharger A (M.02-PI-152) *) (* OldName: AI_M_02_PI_152	; Cyclic: 5; *)
	Pr_EGbHPTC_B : INT; (* AI: Exhaust gas pressure before high-pressure turbocharger B (M.02-PI-252) *) (* OldName: AI_M_02_PI_252	; Cyclic: 5; *)
	Pr_EG_Hi : BOOL; (*DIexhaustgasbackpressurehigh*)
	Pr_EngLubOil : INT; (*AIenginelubricatingoilpressure*)
	Pr_EOF_After : INT; (*AI:Engineoilpressureafteroilfilter,NUP57/AI_M_03_PI_057*)
	Pr_EOF_DiffMon : INT; (*AI:Oilpressurebeforeoilfilter*)
	Pr_EO_Gear_Min : BOOL; (*DI:Oilpressurelowtransmission*)
	Pr_f_BbFilt : INT; (*AI Pressure before Blow-by filter *)
	Pr_f_BbFilt_A : INT; (*AI Pressure before Blow-by filter A*)
	Pr_f_BbFilt_B : INT; (*AI Pressure before Blow-by filter B*)
	Pr_GR_I : INT; (*AI Gas Pressure in Gas Rail number 1 *) (* OldName: AIPressGasRail	; Cyclic: 2; *)
	Pr_GR_II : INT; (*AI Gas Pressure in Gas Rail number 2*) (* OldName: AIPressGasRail_II	; Cyclic: 2; *)
	Pr_GT1 : INT; (*AI	Gaspressuregastrain1afterfilter*)
	Pr_GT1_1_Max : BOOL; (*DI	Gaspressuremaximumgastrain1-line1*)
	Pr_GT1_1_Min : BOOL; (*DI	Gaspressurelowgastrain1-line1*)
	Pr_GT1_2_Max : BOOL; (*DI	Gaspressuremaximumgastrain1-line2*)
	Pr_GT1_2_Min : BOOL; (*DI	Gaspressurelowgastrain1-line2*)
	Pr_GT1_3_Max : BOOL; (*DI	Gaspressuremaximumgastrain1-line3*)
	Pr_GT1_3_Min : BOOL; (*DI	Gaspressurelowgastrain1-line3*)
	Pr_GT1_4_Max : BOOL; (*DI	Gaspressuremaximumgastrain1-line4*)
	Pr_GT1_4_Min : BOOL; (*DI	Gaspressurelowgastrain1-line4*)
	Pr_GT1_Max : BOOL; (*DI	Gaspressuremaximumgastrain1*)
	Pr_GT1_Min : BOOL; (*DI	Gaspressurelowgastrain1*)
	Pr_GT2_Max : BOOL; (*DI	Gaspressuremaximumgastrain2*)
	Pr_GT2_Min : BOOL; (*DI	Gaspressurelowgastrain2*)
	Pr_GT_Gas : INT; (*IF654gaspressure	*)
	Pr_GT_MinBefCompr : BOOL; (*DI	Gaspressurelowbeforegascompressor*)
	Pr_GT_Suct : INT; (*IF655suctionpressure	*)
	Pr_HW_Hi : BOOL; (*DIheatwaterpressurehigh*)
	Pr_HW_Hi1 : BOOL; (*DIheatwaterpressurehigh*)
	Pr_HW_Lo : BOOL; (*DIheatwaterpressurelow*)
	Pr_HW_Su_HT : INT; (*supply water pressure HT circuit*) (*OldName:AI_p_VL_HT; Cycle:5;*)
	Pr_HW_Su_LT : INT; (*supply water pressure LT circuit*) (*OldName:AI_p_VL_NT; Cycle:5;*)
	Pr_MGT_a_Filt : INT; (*AI main gas train pressure after filter [bar]*) (* OldName: AI_p_GT1; Cyclic: 2; *)
	Pr_MGT_sp : INT; (*AO pressure gas rail set point with Offset considered*) (*OldName:rPr_MGT_sp; Cycle:5;*)
	Pr_N2_Hi : BOOL; (*DIpressureN2high*)
	Pr_N2_Lo : BOOL; (*DIpressureN2low*)
	Pr_OilSkid_HP_DE : INT; (*AI OilSkid oil pressure in high pressure circuit to DE bearing*)
	Pr_OilSkid_HP_NDE : INT; (*AI OilSkid oil pressure in high pressure circuit to NDE bearing *)
	Pr_Oil_LPTC_In_A : INT; (*oil pressure LP turbo charger A inlet*) (*OldName:P_OEL_ND_EintrittA; Cycle:5;*)
	Pr_Oil_LPTC_In_B : INT; (*oil pressure LP turbo charger B inlet*) (*OldName:P_OEL_ND_EintrittB; Cycle:5;*)
	Pr_PC : INT; (*AI	Pressureprechamber*)
	Pr_PCG : INT; (*IF650prechambergaspressure	*)
	Pr_PCGBefComp_Lo : BOOL; (*DIsuctionpressureprechambergascompressorhigh*)
	Pr_PCGT : INT; (*AI	Gaspressureprechambergastrainafterfilter*)
	Pr_PCGT_Out : INT; (*AI Warning measuring signal failure - gas pressure after pre chamber gas pressure regulator*) (* OldName: AI_p_PCGT_Out; Cyclic: 2; *)
	Pr_PCGT_sp : INT; (*AO main gas train pressure - set point with Offset considered*) (*OldName:rPr_PCGT_sp; Cycle:5;*)
	Pr_PCG_GC_Dem : BOOL; (*DO	Demandprechampergascompressor*)
	Pr_PCG_Min : BOOL; (*DI	Prechambergascompressorpressureminimum*)
	Pr_PC_Diff : INT; (*IFF	-	IF652prechamberdiff.pressure	*)
	Pr_TCOF_EOF_DiffMax : BOOL; (*DI:Differencepressureturbochargeroilfilterhigh*)
	Pr_TC_EOF_After : INT; (*AIoilpressureafterturbochargeroilfilter,NUP62/AI_M_03_PI_062*)
	Pr_TC_EOF_Before : INT; (*AI:Oilpressureinfrontofturbochargeroilfilter,NUP61/AI_M_03_PI_061*)
	Pr_ThR_AirLo : BOOL; (*DIthermalreactorcompressedairpressurelow*)
	PS400V_ENGIA_CB_On : BOOL; (*Supply disconnecting device 400VAC +ENGIA on*)
	PulseMainsOk : BOOL; (*pulsemainsok*)
	P_Act : ARRAY[0..2] OF INT; (*actualelectricpower[kW]*)
	P_Act_AO : INT; (*actualpowerrelatedtorP_nomfilteredT=1s*)
	P_GenC_Bloc : BOOL; (*DO:internalblockingsignal*)
	P_GenC_Fix0SOn : BOOL; (*DO:nolimitingpowervalue-P-fixvalue0fromEUison*)
	P_GenC_Fix1SOn : BOOL; (*DO:powervalue-P-fixvalue1fromEUison*)
	P_GenC_Fix2SOn : BOOL; (*DO:powervalue-P-fixvalue2fromEUison*)
	P_GenC_Fix3SOn : BOOL; (*DO:powervalue-P-fixvalue3fromEUison*)
	P_GenC_Fix4SOn : BOOL; (*DO:powervalue-P-fixvalue4fromEUison*)
	P_GenC_Fix5SOn : BOOL; (*DO:powervalue-P-fixvalue5fromEUison*)
	P_GenC_SetEU : INT; (*AI:requestpowervaluefromEU*)
	P_GenC_SetEUCOf : BOOL; (*DI:requestpowervaluefromEU-off(deactivate*)
	P_GenC_SetEUCOn : BOOL; (*DI:requestpowervaluefromEU-on(activate*)
	P_GenC_SetFix1EU : BOOL; (*DI:powervalue-P-fixvalue1fromEU*)
	P_GenC_SetFix2EU : BOOL; (*DI:powervalue-P-fixvalue2fromEU*)
	P_GenC_SetFix3EU : BOOL; (*DI:powervalue-P-fixvalue3fromEU*)
	P_GenC_SetFix4EU : BOOL; (*DI:powervalue-P-fixvalue4fromEU*)
	P_GenC_SetFix5EU : BOOL; (*DI:powervalue-P-fixvalue5fromEU*)
	P_GenC_SOf : BOOL; (*DO:powervaluefonEUisoff*)
	P_GenC_SOn : BOOL; (*DO:powervaluefonEUison*)
	P_GT_Max_Backfire : BOOL; (*DI	gaspressurehigh-backfire*)
	P_Lo : BOOL; (*DOpowerlow(foropeningGCB*)
	P_Red_Active : BOOL; (*powerreductionactive-anykind-HALIOOutput*)
	P_Red_AI_Norm : INT; (*Externalpowerreduction	*)
	P_Red_CH4Active : BOOL; (* Power limitation because of CH4 content active *) (*OldName: CH4RED_0; Cyclic:5*)
	P_Red_GasPrActive : BOOL; (* Power limitation because OF gas pressure active*) (*OldName: GD_RED_0; Cyclic:5;*)
	P_Red_Norm : INT; (*powerreduction*)
	P_Red_SuctPrActive : BOOL; (* Power limitation because OF suction pressure active*) (*OldName: SD_RED_0; Cyclic:5;*)
	P_Set_ExtAI_Norm : INT; (*Externalpowersetpoint	*)
	QLim_GenC_Act : BOOL; (*DO:reactivepowerlimitation(Plim*)
	QLim_GenC_SetEU : INT; (*AI:setpointreactivepowerlimitation(Qlim*)
	QLim_GenC_SetEUCOf : BOOL; (*DI:setpointreactivepowerlimitation(Qlim*)
	QLim_GenC_SetEUCOn : BOOL; (*DI:setpointreactivepowerlimitation(Qlim*)
	QLim_GenC_SOf : BOOL; (*DO:reactivepowerlimiting(QLim*)
	QLim_GenC_SOn : BOOL; (*DO:reactivepowerlimiting(QLim*)
	QPC_GenC_SetEUCOf : BOOL; (*DI:setpointreactivepowercharacteristicsCOS(phi*)
	QPC_GenC_SetEUCOn : BOOL; (*DI:setpointreactivepowercharacteristicsCOS(phi*)
	QPC_GenC_SOf : BOOL; (*DO:reactivepowercharacteristicsCOS(phi*)
	QPC_GenC_SOn : BOOL; (*DO:reactivepowercharacteristicsCOS(phi*)
	QUC_GenC_SetEUCOf : BOOL; (*DI:setpointreactivepowercharacteristicsQ=f(U*)
	QUC_GenC_SetEUCOn : BOOL; (*DI:setpointreactivepowercharacteristicsQ=f(U*)
	QUC_GenC_SOf : BOOL; (*DO:reactivepowercharacteristicsQ=f(U*)
	QUC_GenC_SOn : BOOL; (*DO:reactivepowercharacteristicsQ=f(U*)
	QU_GenC_Set : INT; (*AI:setpointgeneratorvoltageforrectivepowercontrol[%]vorEU*)
	Q_Act : ARRAY[0..2] OF INT; (*actualreactivepower[kVar]*)
	Q_GenC_Act : INT; (*AO:reactivepoweractuelevalue*)
	Q_GenC_CUST : INT; (*costumiz:scalingvalueforreactivepower(Q*)
	Q_GenC_Fix1SOn : BOOL; (*DO:reactivepower(Q*)
	Q_GenC_Fix2SOn : BOOL; (*DO:reactivepower(Q*)
	Q_GenC_Fix3SOn : BOOL; (*DO:reactivepower(Q*)
	Q_GenC_Fix4SOn : BOOL; (*DO:reactivepower(Q*)
	Q_GenC_Fix5SOn : BOOL; (*DO:reactivepower(Q*)
	Q_GenC_SetEU : INT; (*AI:setpointreactivepowercharacteristic(Q*)
	Q_GenC_SetEUCOf : BOOL; (*DI:setpointreactivepowercharacteristic(Q*)
	Q_GenC_SetEUCOn : BOOL; (*DI:setpointreactivepowercharacteristic(Q*)
	Q_GenC_SetFix1EU : BOOL; (*DI:reactivepower(Q*)
	Q_GenC_SetFix2EU : BOOL; (*DI:reactivepower(Q*)
	Q_GenC_SetFix3EU : BOOL; (*DI:reactivepower(Q*)
	Q_GenC_SetFix4EU : BOOL; (*DI:reactivepower(Q*)
	Q_GenC_SetFix5EU : BOOL; (*DI:reactivepower(Q*)
	Q_GenC_SOf : BOOL; (*DO:reactivepowercharacteristic(Q*)
	Q_GenC_SOn : BOOL; (*DO:reactivepowercharacteristic(Q*)
	Rdy_MSy : BOOL; (*enginereadyforMSY*)
	RelAux : BOOL; (*DIreleaseengineoperationfromauxiliarieswithmonitoring*)
	RelAuxNoMon : BOOL; (*DIreleaseengineoperationfromauxiliarieswithnomonitoring*)
	RelEngOpFromGSy : BOOL; (*DIreleaseengineoperationfrom'gemeinsame'synchronization*)
	RelGasPlant : BOOL; (*DI	Releasefromgasplantmissing.FALSE=Missing*)
	RelMainGVext : BOOL; (*DIreleasemaingasvalvefromexternal*)
	Rel_BS : BOOL; (*DIreleaseblackstart*)
	Rel_ER_Fan : BOOL; (*DOdemandVE>min.speed*)
	Rel_ER_FC : BOOL; (*DOreleasefrequencyconverterforroomVE*)
	Rel_ER_PurgeCycle : BOOL; (*DIreleasepurgecycle*)
	Rel_I : BOOL; (*DIreleaseislandoperation*)
	Rel_LS : BOOL; (*DIreleaseloadshedding*)
	Rel_MasCtr : BOOL; (*releasefrommastercontrol*)
	Rel_Sync_Load : BOOL; (*DO:releaseofsynchronizationandload*)
	Rel_U_Sel_LS_Gen : BOOL; (*ReleasevoltageselectionLS-Generator*)
	Req_PeakLoad : BOOL; (*requestpeakload*)
	Req_PowMod : BOOL; (*DIrequestpoweroperationmode*)
	Req_Test : BOOL; (*requesttestmode*)
	ResetRemExt : BOOL; (*resetremoteexternal*)
	ResetRemoteExt : BOOL; (*resetremoteexternal*)
	ResetTrip : BOOL; (*DOresettrippulse*)
	ResetWarning : BOOL; (*DOresetwarningpulse*)
	RMC_SetCOf : BOOL; (*DI:regulationmargincontrol-off(deactivate*)
	RMC_SetCOn : BOOL; (*DI:regulationmargincontrol-on(activate*)
	RMC_SOf : BOOL; (*DO:regulationmargincontrolisoff*)
	RMC_SOn : BOOL; (*DO:regulationmargincontrolison*)
	RotatingLight : BOOL; (*DOrotatinglightyellow*)
	RSE_SetEUCOf : BOOL; (* DI: reset decoupling RSE from EU (ERDF) *) (*OldName:DI_RDEmRSE PV;Cycle:2;*)
	RSE_SetEUCOn : BOOL; (* DI: set decoupling RSE from EU (ERDF) *) (*OldName:DI_SDEmRSE PV;Cycle:2;*)
	RSE_SOn : BOOL; (* DO: decoupling RSE from EU (ERDF)  							*)
	SafetyLoop_EmStop : BOOL; (*safetyloopemergencystopok*)
	SafetyLoop_Eng : BOOL; (*safetyloopengine*)
	SafetyLoop_Gas : BOOL; (*DIsafetyloopgasok*)
	SafetyLoop_HWC : BOOL; (*safetyloopheatwatercircuitok*)
	ScavFanCB_trip : BOOL; (*DIexhaustgasscavengingfancircuitbreakertripped*)
	ScavFanCoOn : BOOL; (*DOscavengingfancomandON*)
	ScavFanFC_P_Lo : BOOL; (*DIexhaustgasscavengingfanfrequencyconverterpowerlow*)
	ScavFanFC_Rdy : BOOL; (*DIexhaustgasscavengingfanfrequencyconverterreadyforoperation*)
	ScavFanOp : BOOL; (*DIexhaustgasscavengingfanoperating*)
	ScavFan_Sp : INT; (*AOscavengingfansetpoint*)
	ScavVaClosed : BOOL; (*DIscavengingvalveclosed*)
	ScavVaCoClose : BOOL; (*DOscavengingvalvecommandclose*)
	ScavVaCoOpen : BOOL; (*DOscavengingvalvecommandopen*)
	ScavVaFailure : BOOL; (*DIscavengingvalvefailure*)
	ScavVaOpened : BOOL; (*DIscavengingvalveopened*)
	SelGasTyp : BOOL; (*DI:Selectiongastype-general*)
	SelGasTyp2 : BOOL; (*DI:Selectiongastype2*)
	SelGasTyp3 : BOOL; (*DI:Selectiongastype3*)
	SelGasTyp4 : BOOL; (*DI:Selectiongastype4*)
	Set_ER_Fan_Min : BOOL; (*DOdemandVEmin.speed*)
	SGM_DirStepper1 : BOOL; (*DO SGM direction stepper 1 *)
	SGM_DirStepper2 : BOOL; (*DO SGM direction stepper 2 *)
	SGM_DirStepper3 : BOOL; (*DO SGM direction stepper 3 *)
	SGM_EnabStepper1 : BOOL; (*DO SGM enable stepper 1 *)
	SGM_EnabStepper2 : BOOL; (*DO SGM enable stepper 2 *)
	SGM_EnabStepper3 : BOOL; (*DO SGM enable stepper 3 *)
	Signal1R1 : BOOL; (*DOsignallamp1redcontinuouslight*)
	Signal1R2 : BOOL; (*DOsignallamp2redcontinuouslight*)
	SignalG1 : BOOL; (*DOsignallamp1greencontinuouslight*)
	SignalG2 : BOOL; (*DOsignallamp2greencontinuouslight*)
	SignalR1 : BOOL; (*DOsignallamp1redflashing*)
	SignalR2 : BOOL; (*DOsignallamp2redflashing*)
	SignalY1 : BOOL; (*DOsignallamp1yellowcontinuouslight*)
	SignalY2 : BOOL; (*DOsignallamp2yellowcontinuouslight*)
	ssFreqDiffMin : ARRAY[0..2] OF INT; (*maximum frequence difference (negative) [-0,49..0,00Hz]*)
	ssIN : ARRAY[0..2] OF INT; (* neutral current [A] *)
	ssReactMin : ARRAY[0..2] OF INT; (* min. reactive power monit. limit *)
	ssSynchAngleDeviation : ARRAY[0..2] OF INT; (*Deviation angle between synchronis *)
	ssSynchVoltDeviation : ARRAY[0..2] OF INT; (*Deviation voltage between synchron *)
	StUpSpeed : BOOL; (*DOstartupspeed*)
	Sys_Run : BOOL; (*RUNDigitaOutbittoHAL*)
	Sys_Run1 : BOOL; (*RUNDigitaOutbittoHAL*)
	Sys_Run2 : BOOL; (*RUNDigitaOutbittoHAL*)
	Sys_Run3 : BOOL; (*RUNDigitaOutbittoHAL*)
	Sys_Run4 : BOOL; (*RUNDigitaOutbittoHAL*)
	Sys_Run5 : BOOL; (*RUNDigitaOutbittoHAL*)
	Sys_Run6 : BOOL; (*RUNDigitaOutbittoHAL*)
	Sy_N_Down : BOOL; (*DIexternalspeedmatchingDOWN*)
	Sy_N_Up : BOOL; (*DIexternalspeedmatchingUP*)
	S_Act : ARRAY[0..2] OF INT; (* appearent power [kV] *)
	tActFiltAlarm : HALioDi_Type; (*DIactivfilteralarm*)
	tActFiltWarn : HALioDi_Type; (*DIactivfilterwarning*)
	tActuator2_Rel : HALioDo_Type; (*DO:Actuatorreleasecommand*)
	tActuator_Ok : HALioDi_Type; (*DI:Actuatorokay*)
	tActuator_Ok_CBV1 : HALioDi_Type; (*DI:Actuatorokaycompressorbypassvalve1*)
	tActuator_Ok_CBV2 : HALioDi_Type; (*DI:Actuatorokaycompressorbypassvalve2*)
	tActuator_Ok_TV1A : HALioDi_Type; (*DI:Actuatorokaythrottlevalve1A*)
	tActuator_Ok_TV1B : HALioDi_Type; (*DI:Actuatorokaythrottlevalve1B*)
	tActuator_Ok_TV2A : HALioDi_Type; (*DI:Actuatorokaythrottlevalve2A*)
	tActuator_Ok_TV2B : HALioDi_Type; (*DI:Actuatorokaythrottlevalve2B*)
	tActuator_Rel : HALioDo_Type; (*DO:Actuatorreleasecommand*)
	tAirER_FS : HALioDi_Type; (*DIengineroomVEflowswitch*)
	tAI_UniAi : ARRAY[0..250] OF HALioAi_Type; (*CustomerIOsystemHAL-connector*)
	tAuxErrWarn : HALioDi_Type; (*DIauxiliarieserror*)
	tAuxFail : HALioDi_Type; (*DIauxilariesfailure*)
	tAuxOverVoltProt_Ok : HALioDi_Type; (*failureovervoltageprotectionauxiliariespowersupply*)
	tAuxPoSuMains : HALioDo_Type; (*DOauxiliariespowersupplyfrommains*)
	tAuxPoSuUPS : HALioDo_Type; (*DOauxiliariespowersupplyfromUPS*)
	tAuxV_Eng_ok : HALioDi_Type; (*DIauxiliariesvoltageengineok*)
	tChC_Heating : HALioDo_Type; (*Demand charge cooler pre heating*)
	tIsland_Op : HALioDo_Type; (*Island operation*)
	tParallel_Op : HALioDo_Type; (*Mains parallel operation*)
	tAuxV_Supply_Ok : HALioDi_Type; (*DIauxiliaryvoltagesupplyok*)
	tBbBlower : HALioDo_Type; (*DO Blow-by Blower*)
	tBbBlower_FC_Rdy : HALioDi_Type; (*DI Blow-by Blower FC ready *)
	tBbBlower_y : HALioAo_Type; (*AO Blow-by Blower Percentage value to FU*)
	tBB_Alive : HALioDi_Type; (*DIbusbaralive*)
	tBB_Dead_MMD : ARRAY[0..2] OF HALioDi_Type; (*DIbusbardeadfromMMD*)
	TBMode : BOOL; (*DItestbenchmode*)
	tCA_IgnP_Set : HALioAo_Type; (*AO:timingpoint*)
	tCCWP_Op : HALioDi_Type; (*DIchargecoolingwaterpumpoperating*)
	tChargeOff_Dem : HALioDo_Type; (*DOchargingunitoffdemand*)
	tChC_DemFan1 : HALioDo_Type; (*DOchargecoolerdemandfan1*)
	tChC_DemFan2 : HALioDo_Type; (*DOchargecoolerdemandfan2*)
	tChC_DemFan3 : HALioDo_Type; (*DOchargecoolerdemandfan3*)
	tChC_DemFan4 : HALioDo_Type; (*DOchargecoolerdemandfan4*)
	tChC_DemFan5 : HALioDo_Type; (*DOchargecoolerdemandfan5*)
	tChC_DemFan6 : HALioDo_Type; (*DOchargecoolerdemandfan6*)
	tChC_DemFan7 : HALioDo_Type; (*DOchargecoolerdemandfan7*)
	tChC_DemFan8 : HALioDo_Type; (*DOchargecoolerdemandfan8*)
	tChC_DemFan9 : HALioDo_Type; (*DOchargecoolerdemandfan9*)
	tChC_DemFan10 : HALioDo_Type; (*DOchargecoolerdemandfan10*)
	tChC_DemFan11 : HALioDo_Type; (*DOchargecoolerdemandfan11*)
	tChC_DemFan12 : HALioDo_Type; (*DOchargecoolerdemandfan12*)
	tChC_DemFan13 : HALioDo_Type; (*DOchargecoolerdemandfan13*)
	tChC_DemFan14 : HALioDo_Type; (*DOchargecoolerdemandfan14*)
	tChC_DemFan15 : HALioDo_Type; (*DOchargecoolerdemandfan15*)
	tChC_DemFan16 : HALioDo_Type; (*DOchargecoolerdemandfan16*)
	tChC_DemPump : HALioDo_Type; (*DOchargecoolerdemandpump*)
	tChC_Failure : HALioDi_Type; (*DIchargecoolerfailure*)
	tChC_FanRdy : HALioDi_Type; (*DIchargecoolerfanready*)
	tChUnit1_CB_On : HALioDi_Type; (*Circuit breaker tripped Charging unit 1*)
	tChUnit2_CB_On : HALioDi_Type; (*Circuit breaker tripped Charging unit 2*)
	tChUnit3_CB_On : HALioDi_Type; (*Circuit breaker tripped +ENGIA Charging unit 1*)
	tChUnit4_CB_On : HALioDi_Type; (*Circuit breaker tripped +ENGIA Charging unit 2*)
	tCnt_GasImp : HALioDi_Type; (*DI	Impulsegascounter*)
	tCnt_OilPulse : HALioDi_Type; (*DIoilcounter*)
	tCnt_Oil_DC2395 : HALioAi_INT_Type; (*AIoilcountercircularbuffer*)
	tCnt_Oil_NC150 : HALioAi_Type; (*AIoilcounter*)
	tCO2_Alarm : HALioDo_Type; (*DOCO2alarm*)
	tCO2_Demand : HALioDi_Type; (*DICO2demand*)
	tCO2_DemCodinox : HALioDo_Type; (*DOCO2demandCODINOX*)
	tCO2_DevFailure : HALioDi_Type; (*DICO2devicefailure*)
	tCO2_FanCoOn : HALioDo_Type; (*DOCO2demandfan*)
	tCO2_FanFailure : HALioDi_Type; (*DICO2fanfailure*)
	tCO2_MPMode : HALioDo_Type; (*DOCO2setCODINOXtomainsparallelmode*)
	tCO2_Rdy : HALioDo_Type; (*DOCO2ready*)
	tCO2_VaClosed : HALioDi_Type; (*DICO2valveclosed*)
	tCO2_VaCoClose : HALioDo_Type; (*DOCO2valvecommandclose*)
	tCO2_VaCoOpen : HALioDo_Type; (*DOCO2valvecommandopen*)
	tCO2_VaFailure : HALioDi_Type; (*DICO2valvefailure*)
	tCO2_VaLockout : HALioDi_Type; (*DIlockoutCO2valve*)
	tCO2_VaOpened : HALioDi_Type; (*DICO2valveopened*)
	tCO2_WD : HALioDo_Type; (*DOCO2watchdog*)
	tCodinox_Rdy : HALioDi_Type; (*DICODINOXreadyforoperation*)
	TCOP_CB_On : BOOL; (*Failure Pump Turbocharger pressure*)
	TCOP_Grid : BOOL; (*turbo charger oil pump mains voltage ok*)
	TCOP_GridOk : BOOL; (*turbo charger oil pump mains voltage ok*)
	TCOP_Op : BOOL; (*DIturbochargeroilpumpoperating*)
	TCOP_UPS_CB_On : BOOL; (*Circuit breaker tripped Prelubrication oil pump / Cool down oilpump*)
	tCO_Alarm : HALioDi_Type; (*DICOalarm*)
	tCO_PreAlarm : HALioDi_Type; (*DICOprealarm*)
	tCP_CBTrip : HALioDi_Type; (*DImoduleand/orinterfacecontrolpanel-circuitbreakertripped*)
	tCtrGenPF_Set : HALioAo_Type; (*AOGenerator???*)
	tCtrTR_Heater_Set : HALioAo_Type; (*AO->Controlleroutput*)
	tCtr_ChCHP_Set : HALioAo_Type; (*AOchargetemperaturecoolerhighpressurecontrolvalve*)
	tCtr_ChCV_Set : HALioAo_Type; (*AOchargetemperaturecoolerventilation*)
	tCtr_ChC_Set : HALioAo_Type; (*AOchargetemperaturecoolercontrolvalve*)
	tCtr_CustOut : ARRAY[0..45] OF HALioAo_Type; (*AI: new output channel für direct usage of customized controllers on HAL*)
	tCtr_ECW_Set : HALioAo_Type; (*AOenginecoolingewatertemp.controlvalvesetpoint*)
	tCtr_EC_Set : HALioAo_Type; (*AOheatwaterreturntemperaturecontrolvalveemergencycooler*)
	tCtr_GC_Set : HALioAo_Type; (*AO Gas compressor*)
	tCtr_Gen_Set : HALioAo_Type; (*AOGenerator???*)
	tCtr_HWRe_Set : HALioAo_Type; (*AOheatwaterreturntemperaturecontrolvalve*)
	tCtr_HWSu_Set : HALioAo_Type; (*AOheatwatersupplytemperaturecontrolvalve*)
	tCustAnaIn : ARRAY[0..120] OF HALioAi_Type; (*ReplacementforRAN_KANAL...*)
	tCustAnaOut : ARRAY[0..60] OF HALioAo_Type; (*newreserveoutputchannel(likeANA.RAN1forinputs)*)
	tCustDigIn : ARRAY[0..200] OF HALioDi_Type; (*new,reservedforProjectspecificuse*)
	tCustDigOut : ARRAY[0..150] OF HALioDo_Type; (*ConnectiontoHAL*)
	tP0_BLOCK_DEIE : HALioDi_Type; (*DI : Installed 1/0 switch *) (*OldName:Cust_switch_erdf PV;Cycle:2;*)
	tCV_Eng_Low : HALioDi_Type; (*Control voltage min*)
	tCV_TCA_Low : HALioDi_Type; (*Control voltage min*)
	tC_CB_EDC : HALioDi_Type; (*DIcustomercircuitbreaker(engine*)
	tC_CB_ESL : HALioDi_Type; (*DIcustomercircuitbreaker(engine*)
	tC_CB_Off : HALioDi_Type; (*DIcustomercircuitbreakeropened*)
	tC_CB_On : HALioDi_Type; (*DIcustomercircuitbreakerclosed*)
	TC_EOP_On : BOOL; (*DO:Engineoilpump,NPO601*)
	TC_EOP_OnUSV : BOOL; (*DO:Engineoilpump,NPO601viaUSV*)
	tDAI_V_Dem : HALioDo_Type; (*DO: DAI shut off valve open command *)
	tDAI_V_Opened : HALioDi_Type; (*DI: DAI shut off valve position opened *)
	tDAI_V_Closed : HALioDi_Type; (*DI: DAI shut off valve position closed *)
	tDAI_Dem : HALioDo_Type; (*DO: Demand DAI actuator bank A and B *)
	tPos_DAI_Set_A : HALioAo_Type; (* AO: Position setpoint DAI control valve bank A *)
	tPos_DAI_Act_A : HALioAi_Type; (* AI: Position feedback DAI control valve bank A *)
	tPos_DAI_Set_B : HALioAo_Type; (* AO: Position setpoint DAI control valve bank B *)
	tPos_DAI_Act_B : HALioAi_Type; (* AI: Position feedback DAI control valve bank B *)
	tDAI_CB_On : HALioDi_Type; (* DI: DAI curcuit breaker feedback signal *)
	tActuator_Ok_DAI_A : HALioDi_Type; (* DI: Actuator ok DAI bank A *)
	tActuator_Ok_DAI_B : HALioDi_Type; (* DI: Actuator ok DAI bank B *)
	tDemandBB : HALioDo_Type; (*demandbusbar*)
	tDemEngOpExt : HALioDi_Type; (*externaldemandofengineoperation*)
	tDemFlair : HALioDi_Type; (*DI	Demandgascompressorforflairoperationmode*)
	tDemPurgeER : HALioDo_Type; (*DOdemandroomVEforpurgecycle*)
	tDiffPrct : HALioDi_Type; (*DI:Differentialprotection*)
	tDI_Dem_EU_MnsConBlock : HALioDi_Type; (*Demand block mains connection energy provider*)
	tDI_Dem_EU_Block : HALioDi_Type; (*externalrequestfromutility(evu*)
	tDI_Dem_P_Red_EVU_Stage1 : HALioDi_Type; (*externalrequestfromutility(evu*)
	tDI_Dem_P_Red_EVU_Stage2 : HALioDi_Type; (*externalrequestfromutility(evu*)
	tDI_Dem_P_Red_EVU_Stage3 : HALioDi_Type; (*externalrequestfromutility(evu*)
	tDI_Dem_P_Red_EVU_Stage4 : HALioDi_Type; (*externalrequestfromutility(external,vintagestyledutilisation*)
	tDI_Dem_P_Red_EVU_Stage5 : HALioDi_Type; (*externalrequestfromutility(external,vintagestyledutilisation*)
	tDI_UniDi : ARRAY[0..250] OF HALioDi_Type; (*CustomerIOsystemHAL-connector*)
	tDO_Eng_Block_EVU : HALioDo_Type; (*acknowlegerequestfromutility(evu*)
	tDO_P_Red_EVU_Stage0 : HALioDo_Type; (*acknowlegerequestfromutility(evu*)
	tDO_P_Red_EVU_Stage1 : HALioDo_Type; (*acknowlegerequestfromutility(evu*)
	tDO_P_Red_EVU_Stage2 : HALioDo_Type; (*acknowlegerequestfromutility(evu*)
	tDO_P_Red_EVU_Stage3 : HALioDo_Type; (*acknowlegerequestfromutility(evu*)
	tDO_P_Red_EVU_Stage4 : HALioDo_Type; (*acknowlegerequestfromutility(external,vintagestyledutilisationfeedback*)
	tDO_P_Red_EVU_Stage5 : HALioDo_Type; (*acknowlegerequestfromutility(external,vintagestyledutilisationfeedback*)
	tDPr_AirFilt : HALioAi_Type; (*engineairinletfilterdifferencepressure[bar]*)
	tDPr_AirFilt_A : HALioAi_Type; (*engineairinletfilterdifferencepressureA[bar]*)
	tDPr_AirFilt_B : HALioAi_Type; (*engineairinletfilterdifferencepressureB[bar]*)
	tDPr_InAirFiltERV_Hi : HALioDi_Type; (*air inlet filter difference pressure high - engine room ventilation*) (*V04.04.00.00*)
	tDPr_OilSkid_FiltHP_DE_Hi : HALioDi_Type; (*DI OilSkid difference pressure - oil high pressure filter to DE bearing*)
	tDPr_OilSkid_FiltHP_NDE_Hi : HALioDi_Type; (*DI OilSkid fan - circuit breaker*)
	tDPr_OilSkid_FiltLP_Hi : HALioDi_Type; (*DI OilSkid difference pressure - oil low pressure filter*)
	tEarthCB_Off : HALioDi_Type; (*DIearthcircuitbreakeropened,francecountryspecific*)
	tECWP1Dem : HALioDo_Type; (*DOenginecoolingwaterpump1demand*)
	tECWP2Dem : HALioDo_Type; (*DOenginecoolingwaterpump2demand*)
	tECWPrehV_Opened : HALioDi_Type; (*DIenginecoolingwaterpreheatingvalveopened*)
	tECWP_FC_Rdy : HALioDi_Type; (*DIenginecoolingwaterpumpfrequencyconverterreadyforoperation*)
	tECWP_Op : HALioDi_Type; (*DIenginecoolingwaterpumpoperating*)
	tECWP_PreH_CB_On : HALioDi_Type; (*Failure Engine jacket water Preheating pump*)
	tECWP_PreH_Dem : HALioDo_Type; (*DOenginecoolingwaterpreheatingpumpdemand*)
	tECWP_Service : HALioDo_Type; (*Service Pump Engine jacket water*)
	tECWP_Service_CB_On : HALioDi_Type; (*Failure Service Pump Engine jacket water*)
	tECWP_Service_COn : HALioDi_Type; (*Demand Service Pump Engine jacket water*)
	tECWV_Fail : HALioDi_Type; (*Failure Flap Preheating Engine jacket water*)
	tECW_DemBpP : HALioDo_Type; (*DOdemandenginecoolingwaterbypasspump(AMOT*)
	tECW_DemBpV : HALioDo_Type; (*DOdemandenginecoolingwaterbypassvalve(AMOT*)
	tECW_PreH1Dem : HALioDo_Type; (*DOenginecoolingwaterpreheating1demand*)
	tECW_PreH2Dem : HALioDo_Type; (*DOenginecoolingwaterpreheating2demand*)
	tECW_PreH3Dem : HALioDo_Type; (*DOenginecoolingwaterpreheating3demand*)
	tECW_PreHV_Closed : HALioDi_Type; (*DIenginecoolingwaterpreheatingvalvestatusclosed*)
	tECW_PreHV_CoClose : HALioDo_Type; (*DOenginecoolingwaterpreheatingvalve-commandclose*)
	tECW_PreHV_CoOpen : HALioDo_Type; (*DOenginecoolingwaterpreheatingvalve-commandopen*)
	tECW_PreHV_Opened : HALioDi_Type; (*DIenginecoolingwaterpreheatingvalvestatusopened*)
	tECW_PreH_Dem : HALioDo_Type; (*DOenginecoolingwaterpreheatingdemand*)
	tEC_DemFan1 : HALioDo_Type; (*DOemergencycoolerdemandfan1*)
	tEC_DemFan2 : HALioDo_Type; (*DOemergencycoolerdemandfan2*)
	tEC_DemFan3 : HALioDo_Type; (*DOemergencycoolerdemandfan3*)
	tEC_DemFan4 : HALioDo_Type; (*DOemergencycoolerdemandfan4*)
	tEC_DemFan5 : HALioDo_Type; (*DOemergencycoolerdemandfan5*)
	tEC_DemFan6 : HALioDo_Type; (*DOemergencycoolerdemandfan6*)
	tEC_DemFan7 : HALioDo_Type; (*DOemergencycoolerdemandfan7*)
	tEC_DemFan8 : HALioDo_Type; (*DOemergencycoolerdemandfan8*)
	tEC_DemFan9 : HALioDo_Type; (*DOemergencycoolerdemandfan9*)
	tEC_DemFan10 : HALioDo_Type; (*DOemergencycoolerdemandfan10*)
	tEC_DemFan11 : HALioDo_Type; (*DOemergencycoolerdemandfan11*)
	tEC_DemFan12 : HALioDo_Type; (*DOemergencycoolerdemandfan12*)
	tEC_DemFan13 : HALioDo_Type; (*DOemergencycoolerdemandfan13*)
	tEC_DemFan14 : HALioDo_Type; (*DOemergencycoolerdemandfan14*)
	tEC_DemFan15 : HALioDo_Type; (*DOemergencycoolerdemandfan15*)
	tEC_DemFan16 : HALioDo_Type; (*DOemergencycoolerdemandfan16*)
	tEC_DemPump : HALioDo_Type; (*DOemergencycoolerdemandpump*)
	tEC_Failure : HALioDi_Type; (*DIemergencycoolerfailure*)
	tEGScavStart_Ext : HALioDi_Type; (*DIexhaustgasscavengingstartfromexternal*)
	tEG_BoVaClosed : HALioDi_Type; (*DIexhaustgasboilervalveclosed*)
	tEG_BoVaClosedTo : HALioDi_Type; (*DIexhaustgasboilervalveclosedtorch*)
	tEG_BoVaCoClose : HALioDo_Type; (*DOexhaustgasboilervalvecommandclose*)
	tEG_BoVaCoOpen : HALioDo_Type; (*DOexhaustgasboilervalvecommandopen*)
	tEG_BoVaFailure : HALioDi_Type; (*DIexhaustgasboilervalvefailure*)
	tEG_BoVaOpened : HALioDi_Type; (*DIexhaustgasboilervalveopened*)
	tEG_BypassDemand : HALioDi_Type; (*DIdemandexhaustgasbypass*)
	tEG_ByVaClosed : HALioDi_Type; (*DIexhaustgasbypassvalveclosed*)
	tEG_ByVaClosedTo : HALioDi_Type; (*DIexhaustgasbypassvalveclosedtorch*)
	tEG_ByVaCoClose : HALioDo_Type; (*DOexhaustgasbypassvalvecommandclose*)
	tEG_ByVaCoOpen : HALioDo_Type; (*DOexhaustgasbypassvalvecommandopen*)
	tEG_ByVaFailure : HALioDi_Type; (*DIexhaustgasbypassvalvefailure*)
	tEG_ByVaOpened : HALioDi_Type; (*DIexhaustgasbypassvalveopened*)
	tEleStarter_Dem : HALioDo_Type; (*DOelectricstarterdemand*)
	tEmStop_MC : HALioDi_Type; (*DI emergency stop push button - module control panel (+A/+MC)*) (* *) (*V04.04.00.00*)
	tEmStop_M : HALioDi_Type; (*DI emergency stop push button - module interface panel (+M)*) (* *) (*V04.04.00.00*)
	tEmStop_ST : HALioDi_Type; (*DI emergency stop push button - master control panel (+ST)*) (* *) (*V04.04.00.00*)
	tEmStop_IS : HALioDi_Type; (*DI emergency stop push button - interlock panel (+IS)*) (* *) (*V04.04.00.00*)
	tEmStop_TS : HALioDi_Type; (*DI emergency stop push button - thermal reactor control panel (+TS)*) (* *) (*V04.04.00.00*)
	tEmStop_GENI : HALioDi_Type; (*DI emergency stop push button - generator interface panel (+GENI)*) (* *) (*V04.04.00.00*)
	tEmStop_ENGIA : HALioDi_Type; (*DI emergency stop push button - engine interface panel bank A (+ENGIA)*) (* *) (*V04.04.00.00*)
	tEmStop_TCMI : HALioDi_Type; (*DI emergency stop push button - turbocharger module interface panel (+TCMI)*) (* *) (*V04.04.00.00*)
	tEmStop_JWMI : HALioDi_Type; (*DI emergency stop push button - jacket water module interface panel (+JWMI)*) (* *) (*V04.04.00.00*)
	tEmStop_OILMI : HALioDi_Type; (*DI emergency stop push button - oil module interface panel (+OILMI)*) (* *) (*V04.04.00.00*)
	tEmStop_SCR : HALioDi_Type; (*DI emergency stop push button - exhaust gas after treatment control panel (+SCR)*) (* *) (*V04.04.00.00*)
	tEmStop_TCMSCAV : HALioDi_Type; (*DI emergency stop push button - exhaust gas scavenging system (+TCMSCAV)*) (* *) (*V04.07.00.00*)
	tEngDemIsland : HALioDi_Type; (*DIenginedemandforislandoperation*)
	tENGIA_UPS_CB_On : HALioDi_Type; (*Circuit breaker tripped supply UPS +TCAI --> +ENGIA*)
	tEngStartFailure : HALioDi_Type; (*DIenginestartfailure*)
	tEngTurn : HALioDi_Type; (*DIengineturnequipmentactive*)
	tEngTurn2 : HALioDi_Type; (*Failure engine turning device*)
	tEng_Aux_Dem_CDR : HALioDo_Type; (*engineauxiliariesdemandwithcooldownrun*)
	tEng_Aux_Dem_CDR2 : HALioDo_Type; (*engineauxiliariesdemandwithcooldownrun*)
	tEng_Aux_Dem_CDR3 : HALioDo_Type; (*engineauxiliariesdemandwithcooldownrun*)
	tEng_Dem : HALioDo_Type; (*enginedemandedforMSY*)
	tEng_Dem_EPS_Ext : HALioDi_Type; (*enginedemandemergencypowersupplyfromexternal*)
	tEng_Rdy_Rem : HALioDo_Type; (*ReadyforRemoteOperation*)
	tEng_Ready : HALioDo_Type; (* DO: aggregate available (PLC run) 							*)
	tEng_Run : HALioDo_Type; (*enginerunning*)
	tEng_Run_Sy : HALioDo_Type; (*engineruning-synchronization*)
	tEng_SUExc_Rel : HALioDi_Type; (*start-upexcitationrelease*)
	tEOF_DiffMax : HALioDi_Type; (*DI:Oildifferencepressuremaximum*)
	tEOF_PreheatRel : HALioDo_Type; (*DO:Releaseoilpreheatingvalve*)
	tEOP1AC_CB_trip : HALioDi_Type; (*DIengineoilpump1ACcircuitbreakertrip*)
	tEOP1AC_Dem : HALioDo_Type; (*DOengineoilpump1AC*)
	tEOP1DC_Dem : HALioDo_Type; (*DOengineoilpump1DC*)
	tEOP_DemExt : HALioDi_Type; (*DIengineoilpumpdemandfromexternal*)
	tEOP_FC_Rdy : HALioDi_Type; (*DI:engineoilpumpfreq.converteroperation/ready*)
	tEOP_FC_Set : HALioAo_Type; (*AO:Setpointfrequencyconvertermotoroilpumpprelubrication,[100%=1.0]*)
	tEOP_On : HALioDo_Type; (*DO:Engineoilpump,NPO602*)
	tEOP_Op : HALioDi_Type; (*DIengineoilpumpoperating*)
	tEOVal_DemOpen : HALioDo_Type; (*DOengineoilrefillvalvedemandopen*)
	tEOVal_LT_Set : HALioAo_Type; (*Control signal Regulator valve NT Oil circuit*)
	tEO_Level : HALioAi_Type; (*EngineOilPanLevel*)
	tEO_Level_Hi : HALioDi_Type; (*DIengineoillevelhighfromlevelswitch*)
	tEO_Level_Lo : HALioDi_Type; (*DIengineoillevellowfromlevelswitch*)
	tEO_Preheat1 : HALioDo_Type; (*DO:engineoilpreheatingelement1*)
	tEO_Preheat2 : HALioDo_Type; (*DO:engineoilpreheatingelement2*)
	tEO_Preheat3 : HALioDo_Type; (*DO:engineoilpreheatingelement3*)
	tEO_Quality : HALioAi_Type; (*AI:Oilqualitysensor,QTOil1/AI_*)
	tEO_Refill : HALioDi_Type; (*DIengineoilrefillONfromlevelswitch*)
	tEO_Supply_Fail : HALioDi_Type; (*DI:Oilsupplyfailure*)
	tERDF_BLOCK : HALioDo_Type; (* DO: Block von ERDF *) (* OldName: DI_EVU_BLOCK ; Cycle: 5 *)
	tERV_Op : HALioDi_Type; (*DIengineroomventilationoperating/airflowok (Safety-related application software source code (EN 13849-1 / 4.6.3))*)
	tERV_InlAir_Op : HALioDi_Type; (*DIengineroominletairventilationoperating/airflowok*)
	tERV_OutlAir_Op : HALioDi_Type; (*DIengineroomoutletairventilationoperating/airflowok*)
	tER_DoorClosed : HALioDi_Type; (*DI engine room doors closed (Safety-related application software source code (EN 13849-1 / 4.6.3))*)
	tER_Ext_Err : HALioDi_Type; (*DIengineroomVEfailure*)
	tER_InlAir_Ext_Err : HALioDi_Type; (*DIengineroominletairVEfailure*)
	tER_OutlAir_Ext_Err : HALioDi_Type; (*DIengineroomoutletairVEfailure*)
	tER_FC_Set : HALioAo_Type; (*AOengineroomfrequencyconvertersetpoint[%]*)
	tEU_RM_BLOCK : HALioDo_Type; (*DO:	Separateunitofutilityandofactivenetwork*)
	tEVU_PowerSet3Dem : HALioDi_Type; (*demandmoduleblockedbyutility*)
	tExCo_Rel : HALioDo_Type; (*DOexternalcoolerrelease*)
	tFastAO_KN_A : HALioAo_Type; (*fastanalogoutputsignalsforvalidation*)
	tFastAO_KN_B : HALioAo_Type; (*fastanalogoutputsignalsforvalidation*)
	tFireAlarm : HALioDi_Type; (*DIfirealarm*)
	tFlairRdy : HALioDi_Type; (*DI	Flairready*)
	tFlow_Gen_Lube : HALioDi_Type; (*generatorlubricationfailure*)
	tFlow_HW_Lo : HALioDi_Type; (*DIheatwaterflowlow*)
	tFlow_OilSkid_DE : HALioAi_Type; (*AI OilSkid oil flow to DE bearing *)
	tFlow_OilSkid_NDE : HALioAi_Type; (*AI OilSkid oil flow to NDE bearing (G.03-FI-003)*)
	tFS_ECW : HALioDi_Type; (*DIflowswitchenginecoolingwater*)
	tF_GenBear_DE1 : HALioAi_Type; (*vibration generator bearing drive end 1*) (*Oldname:AI_v_GenBearDE1;Cycle:5;*)
	tF_GenBear_DE2 : HALioAi_Type; (*vibration generator bearing drive end 2*) (*Oldname:AI_v_GenBearDE2;Cycle:5;*)
	tF_GenBear_NDE1 : HALioAi_Type; (*vibration generator bearing non drive end 1*) (*Oldname:AI_v_GenBearNDE1;Cycle:5;*)
	tF_GenBear_NDE2 : HALioAi_Type; (*vibration generator bearing non drive end 2*) (*Oldname:AI_v_GenBearNDE2;Cycle:5;*)
	tF_MMD : ARRAY[0..2] OF HALioAi_Type; (*actualgeneratorfrequency*)
	tF_MMD_LimHi : ARRAY[0..2] OF HALioDi_Type; (*generatorfrequencytoohigh*)
	tF_MMD_LimLo : ARRAY[0..2] OF HALioDi_Type; (*generatorfrequencytoolow*)
	tF_MMD_Synch1 : ARRAY[0..2] OF HALioAi_Type; (* Frequency Sync-network 1 *)
	tF_MMD_Synch2 : ARRAY[0..2] OF HALioAi_Type; (* Frequency Sync-network 2 *)
	tF_N_DI_Dec : HALioDi_Type; (*synch.digitalindecreasespeed*)
	tF_N_DI_Inc : HALioDi_Type; (*synch.digitalinincreasespeed*)
	tGasAlarm : HALioDi_Type; (*DIgasalarm*)
	tGasPreAlarm : HALioDi_Type; (*DIgasprealarm*)
	tGCB_AGO : HALioDi_Type; (*DIallothergeneratorcircuitbreakeroff*)
	tGCB_COf : HALioDo_Type; (*commandgcboff*)
	tGCB_COn : HALioDo_Type; (*commandgcbon*)
	tGCB_DRM : HALioDi_Type; (*DIgeneratorcircuitbreakerdemandMCBclosingreturntomains*)
	tGCB_DSY : HALioDi_Type; (*DIgeneratorcircuitbreakerdemandsynchronization(synchline*)
	tGCB_DVM : HALioDi_Type; (*voltagematchingforsynchronization*)
	tGCB_DVS : HALioDo_Type; (*generatorcircuitbreakerdemandvoltageselection*)
	tGCB_Earth : HALioDi_Type; (*DIgeneratorcircuitbreakerpositionearth*)
	tGCB_EDC : HALioDo_Type; (*generatorcircuitbreakerenginedemandclose*)
	tGCB_ESL : HALioDo_Type; (*generatorcircuitbreakerstatuslocked*)
	tGCB_MDL : HALioDi_Type; (*DIgeneratorcircuitbreakermasterdemandlock(forclosingotherGCBtodeadBB*)
	tGCB_MRC : HALioDi_Type; (*DIgeneratorcircuitbreakermasterreleaseclose(todeadbusbar*)
	tGCB_Off : HALioDi_Type; (*DIgeneratorcircuitbreakeropened*)
	tGCB_OGP : HALioDi_Type; (*DIgeneratorcircuitbreakerothergeneratorparallel*)
	tGCB_On : HALioDi_Type; (*generatorcircuitbreakerclosed*)
	tGCB_On_ReturnSign : HALioDo_Type; (*ReleaseforUnitrolAVR*)
	tGCB_OpF : HALioDo_Type; (*generatorcircuitbreakeropeningfailure*)
	tGCB_Rac : HALioDi_Type; (*DIgeneratorcircuitbreakerrackedin*)
	tGCB_Rdy : HALioDi_Type; (*DIgeneratorcircuitbreakerready(forclose*)
	tGCB_Rel : HALioDo_Type; (*generatorcircuitbreakerreleaseclosing*)
	tGCB_RI : HALioDi_Type; (*DIgeneratorcircuitbreakerreelaseisland*)
	tGCB_RSP : HALioDo_Type; (*generatorcircuitbreakerreleasesynchpulse*)
	tGCB_RT : HALioDo_Type; (*generatorcircuitbreakerreleasetrip*)
	tGCB_RUC : HALioDo_Type; (*generatorcircuitbreakerreleaseundervoltagecoil*)
	tGCB_SM1 : HALioDi_Type; (*DIgeneratorcircuitbreakeroutputsignalmonitoring1*)
	tGCB_SM2 : HALioDi_Type; (*DIgeneratorcircuitbreakercontactsignalmonitoring2*)
	tGCB_SOn : HALioDo_Type; (* DO: Generator switch is on 									*)
	tGenCtrResetSp : HALioDo_Type; (*Generator controller reset setpoint*)
	tGenCtr_CktBkr_Trip : HALioDi_Type; (*generatorcicuitbreakeroff*)
	tGenDeexitDem : HALioDo_Type; (*DOgeneratordeexitationdemand*)
	tGenIF_CB_On : HALioDi_Type; (*Circuit breaker tripped supply +TCAI --> +GENI*)
	tGenPrctTrip : HALioDi_Type; (*DI:Generatorprotectiontrip*)
	tGen_DVM : HALioDo_Type; (*Generatorvoltagematchingoutput(LeroySomer*)
	tGen_Exc_Off : HALioDi_Type; (*de-excitation*)
	tGen_LO_CoolingSys_Fail : HALioDi_Type; (*generatorlubeoilcoolingsystemfailure*)
	tGen_PreHDem : HALioDo_Type; (*DOGeneratorpreheatdemand*)
	tGen_RVM : HALioDi_Type; (*DIgeneratorreleasevoltagematching(leroysomer*)
	tGen_T_In : HALioAi_Type; (*actualvaluegeneratorinlettemperature*)
	tGen_T_In2 : HALioAi_Type; (*actualvaluegeneratorinlettemperature2*)
	tGndFailure : HALioDi_Type; (*DI:earthfailure*)
	tGnlTrip : HALioDo_Type; (*DOenginegeneraltrip*)
	tGnlWarning : HALioDo_Type; (*DOenginegeneralwarning*)
	tGrC_DCon : HALioDo_Type; (* DO: FALSE = Disconnect from Grid due to GridCode Event*)
	tGT1_1_SafeDevice : HALioDo_Type; (*DO	Gassafetydevice1line1*)
	tGT1_1_SafeDevOK : HALioDi_Type; (*DIGassafetydevice1line1*)
	tGT1_2_SafeDevice : HALioDo_Type; (*DO	Gassafetydevice1line2*)
	tGT1_2_SafeDevOK : HALioDi_Type; (*DI	Gassafetydevice2line2*)
	tGT1_3_SafeDevice : HALioDo_Type; (*DO	Gassafetydevice1line3*)
	tGT1_3_SafeDevOK : HALioDi_Type; (*DIGassafetydevice3line3*)
	tGT1_4_SafeDevice : HALioDo_Type; (*DO	Gassafetydevice1line4*)
	tGT1_4_SafeDevOK : HALioDi_Type; (*DIGassafetydevice4line4*)
	tGT1_SafeDevice : HALioDo_Type; (*DO	Gassafetydevice1*)
	tGT1_SafeDevOK : HALioDi_Type; (*DI	Gassafetydevice1*)
	tGT2_SafeDevice : HALioDo_Type; (*DO	Gassafetydevice2*)
	tGT2_SafeDevOK : HALioDi_Type; (*DI	Gassafetydevice2*)
	tGT3_SafeDevOK : HALioDi_Type; (*DI	Gassafetydevice3*) (*SAFETY PLC*) (*V04.14.00.00*)
	tGT4_SafeDevOK : HALioDi_Type; (*DI	Gassafetydevice4*) (*SAFETY PLC*) (*V04.14.00.00*)
	tGT_AirSupply_LoLo : HALioDi_Type; (*DI FALSE = compressed air supply pressure for gas train too low - error*) (*Oldname : DI_GT_AirSupply_LoLo Cyclic: 2; *)
	tGT_BackFireDev : HALioDi_Type; (*DI	Antibackfiredevice*)
	tGT1_1_BackFireDev : HALioDi_Type; (*DIAntibackfiredevice1line1*)
	tGT1_2_BackFireDev : HALioDi_Type; (*DIAntibackfiredevice1line2*)
	tGT1_3_BackFireDev : HALioDi_Type; (*DIAntibackfiredevice1line3*)
	tGT1_4_BackFireDev : HALioDi_Type; (*DIAntibackfiredevice1line4*)
	tPCbComp_BackFireDev : HALioDi_Type; (*DIAntibackfire device prechamper before compressor*)
	tPCaComp_BackFireDev : HALioDi_Type; (*DIAntibackfire device prechamper after compressor*)
	tGT_CalibrateActive : HALioDi_Type; (*DI	CalibrationGasanalysis*)
	tGT_CH4 : HALioAi_Type; (*IF653CH4content	*)
	tGT_CV : HALioAi_Type; (*AI	Calorificvalue*)
	tGT_FlairFail : HALioDi_Type; (*DI	Flarefailure*)
	tGT_Flap1_Close : HALioDo_Type; (*DO	Closegasflap1*)
	tGT_Flap1_Closed : HALioDi_Type; (*DI	Gasflap1closed(Feedback*)
	tGT_Flap1_Open : HALioDo_Type; (*DO	Opengasflap1*)
	tGT_Flap1_Opened : HALioDi_Type; (*DI	Gasflap1opened(Feedback*)
	tGT_Flap2_Close : HALioDo_Type; (*DO	Closegasflap2*)
	tGT_Flap2_Closed : HALioDi_Type; (*DI	Gasflap2closed(Feedback*)
	tGT_Flap2_Open : HALioDo_Type; (*DO	Opengasflap2*)
	tGT_Flap2_Opened : HALioDi_Type; (*DI	Gasflap2opened(Feedback*)
	tGT_FlareOpMod : HALioDi_Type; (*DI	Flareinoperationalmode*)
	tGT_GC_Dem : HALioDo_Type; (*DO	Demandgascompressor*)
	tGT_GC_Fail : HALioDi_Type; (*DI	Gascompressorfailure*)
	tGT_O2 : HALioAi_Type; (*IF656O2content	*)
	tGT_RelFlair : HALioDo_Type; (*DO	Releaseflare*)
	tGT_SelectRatioMix : HALioDi_Type; (*DI: Digital input to select gas mixing (1-3 or 1_2-3)*)
	tGT_TypSwitch : HALioDi_Type; (*DI	Gastypeswitchtosecondgas*)
	tGV1Mega_Open : HALioDo_Type; (*DO	Openmegagasvalve1*)
	tGV1_1_Open : HALioDo_Type; (*DO	opengasvalve1_1(GASV1_1*)
	tGV1_2_Open : HALioDo_Type; (*DO	opengasvalve1_1(GASV1_2*)
	tGV1_Open : HALioDo_Type; (*DO	opengasvalve1*)
	tGV2Mega_Open : HALioDo_Type; (*DO	Openmegagasvalve2*)
	tGV2_Open : HALioDo_Type; (*DO	opengasvalve2*)
	tGV3_Open : HALioDo_Type; (*DO	opengasvalve3*) (*SAFETY PLC*) (*V04.14.00.00*)
	tGV4_Open : HALioDo_Type; (*DO	opengasvalve4*) (*SAFETY PLC*) (*V04.14.00.00*)
	tGT1_GV1_Open : HALioDo_Type; (*DO Gastrain1 - Gasvalve 1*) (*SAFETY PLC*) (*V04.14.00.00*)
	tGT1_GV2_Open : HALioDo_Type; (*DO Gastrain1 - Gasvalve 2*) (*SAFETY PLC*) (*V04.14.00.00*)
	tGT2_GV1_Open : HALioDo_Type; (*DO Gastrain2 - Gasvalve 1*) (*SAFETY PLC*) (*V04.14.00.00*)
	tGT2_GV2_Open : HALioDo_Type; (*DO Gastrain2 - Gasvalve 2*) (*SAFETY PLC*) (*V04.14.00.00*)
	tGT3_GV1_Open : HALioDo_Type; (*DO Gastrain3 - Gasvalve 1*) (*SAFETY PLC*) (*V04.14.00.00*)
	tGT3_GV2_Open : HALioDo_Type; (*DO Gastrain3 - Gasvalve 2*) (*SAFETY PLC*) (*V04.14.00.00*)
	tGT4_GV1_Open : HALioDo_Type; (*DO Gastrain4 - Gasvalve 1*) (*SAFETY PLC*) (*V04.14.00.00*)
	tGT4_GV2_Open : HALioDo_Type; (*DO Gastrain4 - Gasvalve 2*) (*SAFETY PLC*) (*V04.14.00.00*)
	tGV_Rel : HALioDo_Type; (*DO	Releasegasvalves*)
	tHorn : HALioDo_Type; (*DOhorn*)
	tHorn_Trip : HALioDo_Type; (*DOhornengineshutdown*)
	tHorn_Warning : HALioDo_Type; (*DOhornwarning*)
	ThR_Contactor : BOOL; (*DOthermalreactorcontactor*)
	ThR_CV_CDec : BOOL; (*DOthermalreactorgascontrolvalvecommanddecrease*)
	ThR_CV_CInc : BOOL; (*DOthermalreactorgascontrolvalvecommandincrease*)
	ThR_EH11 : BOOL; (*DOthermalreactorelectricalheatingelementgroup1output1*)
	ThR_EH12 : BOOL; (*DOthermalreactorelectricalheatingelementgroup1output2*)
	ThR_EH13 : BOOL; (*DOthermalreactorelectricalheatingelementgroup1output3*)
	ThR_EH21 : BOOL; (*DOthermalreactorelectricalheatingelementgroup2output1*)
	ThR_EH22 : BOOL; (*DOthermalreactorelectricalheatingelementgroup2output2*)
	ThR_EH23 : BOOL; (*DOthermalreactorelectricalheatingelementgroup2output3*)
	ThR_EH31 : BOOL; (*DOthermalreactorelectricalheatingelementgroup3output1*)
	ThR_EH32 : BOOL; (*DOthermalreactorelectricalheatingelementgroup3output2*)
	ThR_EH33 : BOOL; (*DOthermalreactorelectricalheatingelementgroup3output3*)
	ThR_ErrLamp : BOOL; (*DOthermalreactorfailurelamp*)
	ThR_GT_COn1 : BOOL; (*DO1thermalreactorgasinjectioncommandon*)
	ThR_GT_COn2 : BOOL; (*DO2thermalreactorgasinjectioncommandon*)
	ThR_LampTest : BOOL; (*DIthermalreactorlamptest*)
	ThR_RunLamp : BOOL; (*DOthermalreactoroperatinglamp*)
	ThR_SL : BOOL; (*DIthermalreactorsafetyloop*)
	ThR_Swth_On : BOOL; (*DIthermalreactoroperationswitchon*)
	ThR_Val_Air : BOOL; (*DOthermalreactorpurgeairvalve*)
	ThR_Val_CCylIn : BOOL; (*DOthermalreactorflapcommandmoveincylinder*)
	ThR_Val_CCylOut : BOOL; (*DOthermalreactorflapcommandmoveoutcylinder*)
	tGF_OilSystem : HALioDi_Type; (*DI general failure oil system*) (*OldName:newPV; Cycle:5*) (*STM*)
	tHumidity_AirIn : HALioAi_Type;
	tHWP_Dem : HALioDo_Type; (*DOheatingwaterpumpdemand*)
	tHWP_Op : HALioDi_Type; (*DIheatingwaterpumpoperating*)
	tIFCP_CBTrip : HALioDi_Type; (*DIinterfacecontrolpanel-circuitbreakertripped*)
	tIgn2_Run_Hal : HALioDi_Type; (*DI:Ignitionsystemdoublerunning*)
	tIgn_Dem : HALioDo_Type; (*demandignition*)
	tIgn_OverspeedRelay : HALioDi_Type; (*DI:Overspeedrelay*)
	tIgn_Run_Hal : HALioDi_Type; (*DI:Ignitionsystemrunning*)
	tImp_OpHour : HALioDo_Type; (*impulseforoperationhourcounter*)
	tInAirER_Fan1DemOn : HALioDo_Type; (*DOdemandairinletventilator1*)
	tInAirER_Fan2DemOn : HALioDo_Type; (*DOdemandairinletventilator2*)
	tInAirER_Lou1DemOpen : HALioDo_Type; (*DOdemandopenairinletlouver1*)
	tInAirER_Lou1Opened : HALioDi_Type; (*DIintakeairengineroomlouver1open*)
	tInAirER_Lou2DemOpen : HALioDo_Type; (*DOdemandopenairinletlouver2*)
	tInAirER_Lou2Opened : HALioDi_Type; (*DIintakeairengineroomlouver2open*)
	tDemERVentInLou_Cust : HALioDo_Type; (*DO inlet louvers demand for customer*)
	tIsoCB_Off : HALioDi_Type; (*DIdisconnectingcircuitbreakeropened,francecountryspecific*)
	tI_Avg : ARRAY[0..2] OF HALioAi_Type; (*IF513gen.currentaveragev.	*)
	tI_Diff : HALioDi_Type; (*generatordifferentialprotectiontrip*)
	tI_L1 : ARRAY[0..2] OF HALioAi_Type; (*PhasecurrentgeneratorI1*)
	tI_L2 : ARRAY[0..2] OF HALioAi_Type; (*PhasecurrentgeneratorI2*)
	tI_L3 : ARRAY[0..2] OF HALioAi_Type; (*PhasecurrentgeneratorI3*)
	tI_MMD_Asy : ARRAY[0..2] OF HALioDi_Type; (*generatorcurrentnegativesequencetoohigh*)
	tI_MMD_LimHi : HALioDi_Type; (*MMD:overloadshortcircuit*)
	tI_MMD_Neutr_LimHi : ARRAY[0..2] OF HALioDi_Type; (*generatorneutralcurrenttoohigh*)
	tKLS90_1 : HALioAi_Type; (*AI:KLS90sensor1signal*)
	tKLS90_2 : HALioAi_Type; (*AI:KLS90sensor1signal*)
	tLam_Act : HALioAi_Type; (*actualLambdavalue*)
	tLOS_Dem : HALioDo_Type; (*Generatordemandlubeoilsystem*)
	tLeroySomer_AuxContactor : HALioDo_Type; (*LEROY-SOMERAuxiliaryContactor*)
	tLev_OilSkid_Sump_Hi : HALioDi_Type; (*DI OilSkid oil in safety sump *)
	tLev_OilSkid_Tank : HALioAi_Type; (*AI OilSkid tank level*)
	tLineCB_On : HALioDi_Type; (*DIlinecircuitbreakerclosed*)
	tLock_C_MCB : HALioDo_Type; (*lockcustomermainscircuitbreaker*)
	tLSL_In : HALioAi_Type; (*AIloadsharingline*)
	tLSL_Out : HALioAo_Type; (*AOloadsharingline*)
	tLS_Dem : HALioDo_Type; (*DOloadsheddingdemand*)
	tL_ECW_Lo : HALioDi_Type; (*DIenginecoolingwaterlevellow*)
	tL_ECW_LoLo : HALioDi_Type; (*DIenginecoolingwaterlevellowlow*)
	tL_FreshOilTank_Lo : HALioDi_Type; (*DIfreshoiltanklevellow*)
	tL_FreshOilTank_Hi : HALioDi_Type; (*DI fresh oil tank level high*) (*OldName:newPV; Cycle:5*) (*STM*)
	tL_InMa_Hi : HALioDi_Type; (*DIwateringressintoinletmanifold*)
	tL_InMa_NotHi : HALioDi_Type; (*DIwateringressintoinletmanifoldnegated*)
	tL_OilSump3Hi : HALioDi_Type; (*DIleveloilsump3high*)
	tL_OilSump2Hi : HALioDi_Type; (*DIleveloilsump2high*)
	tL_OilSumpHi : HALioDi_Type; (*DIleveloilsumphigh*)
	tL_WasteOilTank_Hi : HALioDi_Type; (*DIwasteoiltanklevelhigh*)
	tLeak_FreshOilPump : HALioDi_Type; (*DI leakage fresh oil pump*) (*OldName:newPV; Cycle:5*) (*STM*)
	tLeak_FreshOilTank : HALioDi_Type; (*DI leakage fresh oil tank*) (*OldName:newPV; Cycle:5*) (*STM*)
	tLeak_WasteOilPump : HALioDi_Type; (*DI leakage waste oil pump*) (*OldName:newPV; Cycle:5*) (*STM*)
	tLeak_WasteOilTank : HALioDi_Type; (*DI leakage waste oil tank*) (*OldName:newPV; Cycle:5*) (*STM*)
	tMainGV_Rel : HALioDo_Type; (*DOmaingasvalverelease*)
	tMainsStartDevDem : HALioDo_Type; (*DOmainsstartdevicedemand*)
	tMainsStartDevFail : HALioDi_Type; (*DImainsstartdevicefailure*)
	tMainsStartDevOk : HALioDi_Type; (*DImainsstartingdeviceOK*)
	tMCB_COf : HALioDo_Type; (*commandmcboff*)
	tMCB_COn : HALioDo_Type; (*mainscircuitbreakercomandon*)
	tMCB_DcpQu_SetEUCOf : HALioDi_Type; (* DI: reset decoupling quickly from EU (ERDF) *) (*OldName:DI_RFDemMCBoff PV;Cycle:2;*)
	tMCB_DcpQu_SetEUCOn : HALioDi_Type; (* DI: set decoupling quickly from EU (ERDF) *) (*OldName:DI_SFDemMCBoff PV;Cycle:2;*)
	tMCB_Dcp_SetEUCOf : HALioDi_Type; (* DI: rest requirement decoupling from EU(ERDF),DIs *) (*OldName:DI_RDemandMCBoff PV;Cycle:2;*)
	tMCB_Dcp_SetEUCOn : HALioDi_Type; (* DI: set requirement  decoupling from EU(ERDF),DIs *) (*OldName:DI_SDemandMCBoff PV;Cycle:2;*)
	tMCB_DVS : HALioDo_Type; (*mainscircuitbreakerdemandvoltageselection*)
	tMCB_EDF_SOn : HALioDo_Type; (* DO: feedback Engine off get  								*)
	tMCB_Off : HALioDi_Type; (*DImainscircuitbreakeropened*)
	tMCB_OL : HALioDi_Type; (*DImainscircuitbreakeroverload*)
	tMCB_On : HALioDi_Type; (*SS447NetzschalterEIN*)
	tMCB_Rac : HALioDi_Type; (*DImainscircuitbreakerrackedin*)
	tMCB_Rdy : HALioDi_Type; (*DImainscircuitbreakerready(forclose*)
	tMCB_Rel_Sync : HALioDi_Type; (* DI: release synchronization from EU(ERDF) *) (*OldName:DI_ReleaseMCBon PV;Cycle:2;*)
	tMCB_Rel_Sync_SOn : HALioDo_Type; (* DO: releas decoupling quickly from EU (ERDF)  				*)
	tMCB_Rem : HALioDi_Type; (*DImainscircuitbreakerremote(operatingmode*)
	tMCB_RSP : HALioDo_Type; (*mainscircuitbreakerreleasesynchpulse*)
	tMCB_RT : HALioDo_Type; (*mainscircuitbreakerreleasetrip*)
	tMCB_SM : HALioDi_Type; (*DImainscircuitbreakersignalmonitoring*)
	tMCB_SOn : HALioDo_Type; (* DO: receive requested Command form machine 					*)
	tMCP_CBTrip : HALioDi_Type; (*DImodulecontrolpanel-circuitbreakertripped*)
	tMGT_BOV : HALioDo_Type; (*DO BlowOff valve*) (*Oldname: DO_MGT_BOV; Cycle:5; *)
	tMGT_DBOV : HALioDo_Type; (*DO main gas train dome blow off valve *)
	tMMD_FW_Version : ARRAY[0..2] OF HALioAi_INT_Type; (* program version MMD firmware *)
	tMnsOk : HALioDi_Type; (*DImainsok	*)
	tMnsOk_C13100 : HALioDi_Type; (*DImainsokC13.100monitoringdevice,francecountryspecific*)
	tMnsOk_GTE : HALioDi_Type; (*DImainsokGTEmonitoringdevice,francecountryspecific*)
	tMnsOk_TGS : HALioDi_Type; (*DImainsokTGSmonitoringdevice,francecountryspecific*)
	tMns_MDF : HALioDi_Type; (*DImainsmonitoringdevicefailure*)
	tMonitoringOn : HALioDo_Type; (*DOmonitoringonpulse(safetyloop*)
	tMO_PowerOverload : HALioDi_Type; (*DI:SAFI ignition power module 1 overload *)
	tMO_PowerOverload2 : HALioDi_Type; (*DI:SAFI ignition power module 2 overload *)
	tMO_PowerOverload3 : HALioDi_Type; (*DI:SAFI ignition power module 3 overload *)
	tMO_PowerOverload4 : HALioDi_Type; (*DI:SAFI ignition power module 4 overload *)
	tMO_PwrReply : HALioDi_Type; (*DI:MORIS Ignition Power Module 1 On*)
	tMO_PwrReply2 : HALioDi_Type; (*DI:MORIS Ignition Power Module 2 On*)
	tMO_PwrReply3 : HALioDi_Type; (*DI:MORIS Ignition Power Module 3 On*)
	tMO_PwrReply4 : HALioDi_Type; (*DI:MORIS Ignition Power Module 4 On*)
	tMO_PwrRequest : HALioDo_Type; (*DO:MORIS Ignition Power Module 1 Request*)
	tMO_PwrRequest2 : HALioDo_Type; (*DO:MORIS Ignition Power Module 2 Request*)
	tMO_PwrRequest3 : HALioDo_Type; (*DO:MORIS Ignition Power Module 3 Request*)
	tMO_PwrRequest4 : HALioDo_Type; (*DO:MORIS Ignition Power Module 4 Request*)
	tMO_SaftyLoop : HALioDi_Type; (*DI:MORISSavetyloopclosed*)
	tN2_GV1_Closed : HALioDi_Type; (*DIN2gasvalve1closedstatus*)
	tN2_GV2_Closed : HALioDi_Type; (*DIN2gasvalve2closedstatus*)
	tN2_ScavGV_CoOpen : HALioDo_Type; (*DON2GasValvesvommandopen*)
	tN2_ScavSigLampOn : HALioDo_Type; (*DOSignallampforscavenging*)
	tN_ECWP_Set : HALioAo_Type; (*AOspeedenginecoolingwaterpumpsetpoint*)
	tN_EngStart : HALioDo_Type; (*DOenginestartupspeedexceeded*)
	tN_Set_ExtAI_Norm : HALioAi_Type; (*Externalspeedsetpoint*)
	tN_TCHP : HALioAi_Type; (*highpressureturbochargerspeed[rpm]*)
	tN_TCHP_A : HALioAi_Type; (*highpressureturbochargerspeedA[rpm]*)
	tN_TCHP_B : HALioAi_Type; (*highpressureturbochargerspeedB[rpm]*)
	tN_TCLP : HALioAi_Type; (*lowpressureturbochargerspeed[rpm]*)
	tN_TCLP_A : HALioAi_Type; (*lowpressureturbochargerspeedA[rpm]*)
	tN_TCLP_B : HALioAi_Type; (*lowpressureturbochargerspeedB[rpm]*)
	tOF_FreshOilTank : HALioDi_Type; (*DI overfill prevention device fresh oil tank*) (*OldName:newPV; Cycle:5*) (*STM*)
	tOF_WasteOilTank : HALioDi_Type; (*DI overfill prevention device waste oil tank*) (*OldName:newPV; Cycle:5*) (*STM*)
	tOilSkid_AuxV_Ok : HALioDi_Type; (*DI OilSkid auxiliaries voltage not available*)
	tOilSkid_AuxV_Ok_UPS : HALioDi_Type; (*DI OilSkid auxiliaries voltage not available - UPS*)
	tOilSkid_Fan : HALioDo_Type; (*DO OilSkid fan*)
	tOilSkid_Fan_CBOk : HALioDi_Type; (*DI OilSkid fan - circuit breaker*)
	tOilSkid_Heater : HALioDo_Type; (*DO OilSkid heater*)
	tOilSkid_Heater_CBOk : HALioDi_Type; (*DI OilSkid heater - circuit breaker*)
	tOilSkid_MCB : HALioDi_Type; (*DI OilSkid main switch auxiliaries opened*)
	tOilSkid_PumpC : HALioDo_Type; (*DO OilSkid circulation pump (G.03-M-004)*)
	tOilSkid_PumpC_CBOk : HALioDi_Type; (*DI OilSkid circulation pump - circuit breaker*)
	tOilSkid_PumpHP : HALioDo_Type; (*DO OilSkid high pressure pump *)
	tOilSkid_PumpHP_CBOk : HALioDi_Type; (*DI OilSkid high pressure pump - circuit breaker*)
	tOilSkid_PumpHP_CBOk_UPS : HALioDi_Type; (*DI OilSkid high pressure pump - circuit breaker UPS*)
	tOilSkid_PumpHP_DemOff : HALioDi_Type; (*DI OilSkid high pressure pump - demand OFF*)
	tOilSkid_PumpHP_DemOn : HALioDi_Type; (*DI OilSkid high pressure pump - demand ON*)
	tOilSkid_PumpHP_Soft : HALioDo_Type; (*DO OilSkid high pressure pump - Soft*)
	tOilSkid_PumpHP_UPS : HALioDo_Type; (*DO OilSkid high pressure pump - UPS *)
	tOilSkid_PumpLP : HALioDo_Type; (*DO OilSkid low pressure pump *)
	tOilSkid_PumpLP_CBOk : HALioDi_Type; (*DI OilSkid low pressure pump - circuit breaker*)
	tOlShortCirc : HALioDi_Type; (*DI:Overload/shortcircuit*)
	tOMSS_Aut : HALioDo_Type; (*operationmodeselectorswitch-AUTO*)
	tOMSS_Man : HALioDo_Type; (*operationmodeselectorswitch-MANUAL*)
	tOMSS_MAT : HALioDo_Type; (*operationmodeselectorswitch-MANUALAUTOTEST*)
	tOnly_Island : HALioDi_Type; (*DIonlyislandoperation*)
	tOutAirER_LouDemOpen : HALioDo_Type; (*DOdemandopenairoutletlouver*)
	tOutAirER_LouOpened : HALioDi_Type; (*DIoutletairengineroomlouveropen*)
	tOV_Ctrl_Set : HALioAo_Type; (*AO:hightemperatureengineoilcoolersetpoint*)
	tPCG_DemCoolFan : HALioDo_Type; (*DO	Prechambergascompressor,Demandcoolingventilator*)
	tPCG_DemReliefValve : HALioDo_Type; (*DO	DemandReliefvalve*)
	tPCG_DemValCW : HALioDo_Type; (*DO	Prechambergascompressor,Demandcoolingwatervalve*)
	tPCG_GC_Fail : HALioDi_Type; (*DI	Failureprechambergascompressor*)
	tPCG_GC_Oil_Min : HALioDi_Type; (*DI	prechambergascompressoroillevel*)
	tPCG_GV_DelOpen : HALioDo_Type; (*DO	PrechambergasvalveswithdelayON*)
	tPCG_GV_Open : HALioDo_Type; (*DO	Prechambergasvalves*)
	tPCG_BPV_Open : HALioDo_Type; (*DO Pre chamber gas bypass valve*)
	tPFC_SetCOf : HALioDi_Type; (*DI:primaryfrequencycontrol-off(deactivate*)
	tPFC_SetCOn : HALioDi_Type; (*DI:primaryfrequencycontrol-on(activate*)
	tPFC_SOf : HALioDo_Type; (*DO:primaryfrequencycontrolisoff*)
	tPFC_SOn : HALioDo_Type; (*DO:primaryfrequencycontrolison*)
	tPFUC_GenC_SetEUCOf : HALioDi_Type; (*DI:setpointreactivepowercharacteristicsCOS(phi*)
	tPFUC_GenC_SetEUCOn : HALioDi_Type; (*DI:setpointreactivepowercharacteristicsCOS(phi*)
	tQP_GenC_SetEUCOn : HALioDi_Type; (*DI:setpointreactivepowercharacteristicsQ(P)*)
	tQP_GenC_SetEUCOf : HALioDi_Type; (*DI:setpointreactivepowercharacteristicsQ(P)*)
	tPFUC_GenC_SOf : HALioDo_Type; (*DO:reactivepowercharacteristicsCOS(phi*)
	tPFUC_GenC_SOn : HALioDo_Type; (*DO:reactivepowercharacteristicsCOS(phi*)
	tQP_GenC_SOn : HALioDo_Type; (*DO:reactivepowercharacteristicsQ(P)*)
	tQP_GenC_SOf : HALioDo_Type; (*DO:reactivepowercharacteristicsQ(P)*)
	tPF_Act : ARRAY[0..2] OF HALioAi_Type; (*powerfactor,actualcosphivalue*)
	tPF_AO_PF_I : HALioAo_Type; (*AOpowerfactorgenerator,mAsignal*)
	tPF_AO_PF_U : HALioAo_Type; (*AO:powerfactorgenerator*)
	tPF_CosPCtr_Ena : HALioDo_Type; (*powerfactorcontrollerenabled*)
	tPF_CUSTGenC : HALioAi_Type; (*customiz:scalingvaluegenetarorpowerfactor(COSPHI*)
	tPF_GenC_Act : HALioAo_Type; (*AO:generatorpowerfactor(COSPHI*)
	tPF_GenC_Fix1SOn : HALioDo_Type; (*DO:genetarorpowerfactor(COSPHI*)
	tPF_GenC_Fix2SOn : HALioDo_Type; (*DO:genetarorpowerfactor(COSPHI*)
	tPF_GenC_Fix3SOn : HALioDo_Type; (*DO:genetarorpowerfactor(COSPHI*)
	tPF_GenC_Fix4SOn : HALioDo_Type; (*DO:genetarorpowerfactor(COSPHI*)
	tPF_GenC_Fix5SOn : HALioDo_Type; (*DO:genetarorpowerfactor(COSPHI*)
	tPF_GenC_SetEU : HALioAi_Type; (*AI:setpointgenetarorpowerfactor(COSPHI*)
	tPF_GenC_SetEUCOf : HALioDi_Type; (*DI:setpointgenetarorpowerfactor(COSPHI*)
	tPF_GenC_SetEUCOn : HALioDi_Type; (*DI:setpointgenetarorpowerfactor(COSPHI*)
	tPF_GenC_SetFix1EU : HALioDi_Type; (*DI:setpointgenetarorpowerfactor(COSPHI*)
	tPF_GenC_SetFix2EU : HALioDi_Type; (*DI:setpointgenetarorpowerfactor(COSPHI*)
	tPF_GenC_SetFix3EU : HALioDi_Type; (*DI:setpointgenetarorpowerfactor(COSPHI*)
	tPF_GenC_SetFix4EU : HALioDi_Type; (*DI:setpointgenetarorpowerfactor(COSPHI*)
	tPF_GenC_SetFix5EU : HALioDi_Type; (*DI:setpointgenetarorpowerfactor(COSPHI*)
	tPF_GenC_SOf : HALioDo_Type; (*DO:generatorpowerfactor(COSPHI*)
	tPF_GenC_SOn : HALioDo_Type; (*DO:generatorpowerfactor(COSPHI*)
	tPLim_GenC_Act : HALioDo_Type; (*DO:powerlimitation(Plim*)
	tPLim_GenC_SetEU : HALioAi_Type; (*AI:setpointpowerlimitation(Plim*)
	tPLim_GenC_SetEUCOf : HALioDi_Type; (*DI:setpointpowerlimitation(Plim*)
	tPLim_GenC_SetEUCOn : HALioDi_Type; (*DI:setpointpowerlimitation(Plim*)
	tPLim_GenC_SetEUPFix1 : HALioDi_Type; (*DI:powerlimitationfixvalue1*)
	tPLim_GenC_SetEUPFix2 : HALioDi_Type; (*DI:powerlimitationfixvalue2*)
	tPLim_GenC_SetEUPFix3 : HALioDi_Type; (*DI:powerlimitationfixvalue3*)
	tPLim_GenC_SetEUPFix4 : HALioDi_Type; (*DI:powerlimitationfixvalue4*)
	tPLim_GenC_SetEUPFix5 : HALioDi_Type; (*DI:powerlimitationfixvalue5*)
	tPLim_GenC_SOf : HALioDo_Type; (*DO:powerlimitation(Plim*)
	tPLim_GenC_SOn : HALioDo_Type; (*DO:powerlimitation(Plim*)
	tPos_Act_CBV_A1 : HALioAi_Type; (*AI: compressor bypass valve position A1*)
	tPos_Act_CBV_A2 : HALioAi_Type; (*AI: compressor bypass valve position A2*)
	tPos_Act_CBV_B1 : HALioAi_Type; (*AI: compressor bypass valve position B1*)
	tPos_Act_CBV_B2 : HALioAi_Type; (*AI: compressor bypass valve position B2*)
	tPos_Act_GM1_Norm : HALioAi_Type; (*gasmixer1-normedactualpositionfrompotentiometer[%]*)
	tPos_Act_GM2_Norm : HALioAi_Type; (*gasmixer2-normedactualpositionfrompotentiometer[%]*)
	tPos_Act_TV : HALioAi_Type; (*AI: throttle valve bypass valve position*)
	tPos_Act_TV_A1 : HALioAi_Type; (*AI: throttle valve bypass valve position A1*)
	tPos_Act_TV_A2 : HALioAi_Type; (*AI: throttle valve bypass valve position A2*)
	tPos_Act_TV_B1 : HALioAi_Type; (*AI: throttle valve bypass valve position B1*)
	tPos_Act_TV_B2 : HALioAi_Type; (*AI: throttle valve bypass valve position B2*)
	tPos_Act_WG : HALioAi_Type; (*wastegatevalveposition*)
	tPos_Act_WG_A : HALioAi_Type; (*wastegatevalvepositionA*)
	tPos_Act_WG_B : HALioAi_Type; (*wastegatevalvepositionB*)
	tPos_CBV : HALioAo_Type; (*compressorbypassvalveposition*)
	tPos_CBV34 : HALioAo_Type; (*compressorbypassvalveposition*)
	tPos_CBV_A1 : HALioAo_Type; (*compressorbypassvalvepositionA1*)
	tPos_CBV_A2 : HALioAo_Type; (*compressorbypassvalvepositionA2*)
	tPos_CBV_B1 : HALioAo_Type; (*compressorbypassvalvepositionB1*)
	tPos_CBV_B2 : HALioAo_Type; (*compressorbypassvalvepositionB2*)
	tPos_Set_WG : HALioAo_Type; (*wastegatevalveposition*)
	tPos_Set_WG_A : HALioAo_Type; (*wastegatevalvepositionA*)
	tPos_Set_WG_B : HALioAo_Type; (*wastegatevalvepositionB*)
	tPos_SGM_Enc1 : HALioAi_INT_Type; (*SGM encoder position stepper 1 [1]*)
	tPos_SGM_Enc2 : HALioAi_INT_Type; (*SGM encoder position stepper 2 [1]*)
	tPos_SGM_Enc3 : HALioAi_INT_Type; (*SGM encoder position stepper 3 [1]*)
	tPos_ThR_Val_In1 : HALioDi_Type; (*DI1thermalreactorflapinpositionmovedin*)
	tPos_ThR_Val_In2 : HALioDi_Type; (*DI2thermalreactorflapinpositionmovedin*)
	tPos_ThR_Val_Mid : HALioDi_Type; (*DIthermalreactorflapinmiddleposition*)
	tPos_ThR_Val_Out1 : HALioDi_Type; (*DI1thermalreactorflapinpositionmovedout*)
	tPos_ThR_Val_Out2 : HALioDi_Type; (*DI2thermalreactorflapinpositionmovedout*)
	tPos_TV : HALioAo_Type; (*throttlevalveposition*)
	tPos_TV_A1 : HALioAo_Type; (*throttlevalvepositionA1*)
	tPos_TV_A2 : HALioAo_Type; (*throttlevalvepositionA2*)
	tPos_TV_B1 : HALioAo_Type; (*throttlevalvepositionB1*)
	tPos_TV_B2 : HALioAo_Type; (*throttlevalvepositionB2*)
	tP_Heat_Imp : HALioDi_Type; (*heating power engine heat water circuit impulse*) (*STM 2*)
	tPr_a_BbFilt : HALioAi_Type; (*AI Pressure after Blow-by filter *)
	tPr_a_BbFilt_A : HALioAi_Type; (*AI Pressure after Blow-by filter A*)
	tPr_a_BbFilt_B : HALioAi_Type; (*AI Pressure after Blow-by filter B*)
	tPr_Baro : HALioAi_Type; (*AI	Barometricpressure*)
	tPr_CC : HALioAi_Type; (*AIpressurecrankcase[bar]*)
	tPr_CCircuit_Lo : HALioDi_Type; (*DIwaterpressurecoolercircuitlow*)
	tPr_ChC_Lo : HALioDi_Type; (*DIchargecoolerwaterpressurelow*)
	tPr_Ch_P1HP : HALioAi_Type; (*chargepressurep1beforehighpressureTC[bar]*)
	tPr_Ch_P1HP_A : HALioAi_Type; (*chargepressurep1beforehighpressureTCA[bar]*)
	tPr_Ch_P1HP_B : HALioAi_Type; (*chargepressurep1beforehighpressureTCB[bar]*)
	tPr_Ch_P1LP_A : HALioAi_Type; (*charge pressure before low-pressure TC A [bar]*) (*V04.04.00.00*)
	tPr_Ch_P1LP_B : HALioAi_Type; (*charge pressure before low-pressure TC B [bar]*) (*V04.04.00.00*)
	tPr_Ch_P2 : HALioAi_Type; (*actualchargepressurebeforethrottlevalve*)
	tPr_Ch_P2s : HALioAi_Type; (*actualchargepressure*)
	tPr_Ch_P2s_A : HALioAi_Type; (*chargepressurep2'afterthrottlevalveA[bar]*)
	tPr_Ch_P2s_B : HALioAi_Type; (*chargepressurep2'afterthrottlevalveB[bar]*)
	tPr_Ch_P2_A : HALioAi_Type; (*chargepressurep2beforethrottlevalveA[bar]*)
	tPr_Ch_P2_B : HALioAi_Type; (*chargepressurep2beforethrottlevalveB[bar]*)
	tPr_DAI_A : HALioAi_Type; (*Pressure before DAI control valve bank A [bar] *)
	tPr_DAI_B : HALioAi_Type; (*Pressure before DAI control valve bank B [bar] *)
	tPr_DAI_In : HALioAi_Type; (*Pressure before DAI shut off valve [bar] *)
	tPr_ECW : HALioAi_Type; (*AIpressureenginecoolingwater (Safety-related application software source code (EN 13849-1 / 4.6.3))*)
	tPr_ECWaEng : HALioAi_Type; (*Cooling water pressure downstream of the engine*)
	tPr_EGaHPTC_A : HALioAi_Type; (* AI: Exhaust gas pressure after high-pressure turbocharger A  (M.02-PI-153) *) (* OldName: AI_M_02_PI_153	; Cyclic: 5; *)
	tPr_EGaHPTC_B : HALioAi_Type; (* AI: Exhaust gas pressure after high-pressure turbocharger B  (M.02-PI-253) *) (* OldName: AI_M_02_PI_253	; Cyclic: 5; *)
	tPr_EGaLPTC_A : HALioAi_Type; (* AI: Exhaust gas pressure after low-pressure turbocharger A  (M.02-PI-154) *) (* OldName: AI_M_02_PI_154	; Cyclic: 5; *)
	tPr_EGaLPTC_B : HALioAi_Type; (* AI: Exhaust gas pressure after low-pressure turbocharger B  (M.02-PI-254) *) (* OldName: AI_M_02_PI_254	; Cyclic: 5; *)
	tPr_EGbHPTC_A : HALioAi_Type; (* AI: Exhaust gas pressure before high-pressure turbocharger A (M.02-PI-152) *) (* OldName: AI_M_02_PI_152	; Cyclic: 5; *)
	tPr_EGbHPTC_B : HALioAi_Type; (* AI: Exhaust gas pressure before high-pressure turbocharger B (M.02-PI-252) *) (* OldName: AI_M_02_PI_252	; Cyclic: 5; *)
	tPr_EG_Hi : HALioDi_Type; (*DIexhaustgasbackpressurehigh*)
	tPr_EngLubOil : HALioAi_Type; (*AIenginelubricatingoilpressure (Safety-related application software source code (EN 13849-1 / 4.6.3))*)
	tPr_EOF_After : HALioAi_Type; (*AI:Engineoilpressureafteroilfilter,NUP57/AI_M_03_PI_057 (Safety-related application software source code (EN 13849-1 / 4.6.3))*)
	tPr_EOF_DiffMon : HALioAi_Type; (*AI:Oilpressurebeforeoilfilter*)
	tPr_EO_Gear_Min : HALioDi_Type; (*DI:Oilpressurelowtransmission*)
	tPr_f_BbFilt : HALioAi_Type; (*AI Pressure before Blow-by filter *)
	tPr_f_BbFilt_A : HALioAi_Type; (*AI Pressure before Blow-by filter A*)
	tPr_f_BbFilt_B : HALioAi_Type; (*AI Pressure before Blow-by filter B*)
	tPr_GR_I : HALioAi_Type; (*AI Gas Pressure in Gas Rail number 1 *) (* OldName: AIPressGasRail	; Cyclic: 2; *)
	tPr_GR_II : HALioAi_Type; (*AI Gas Pressure in Gas Rail number 2*) (* OldName: AIPressGasRail_II	; Cyclic: 2; *)
	tPr_GT1 : HALioAi_Type; (*AI	Gaspressuregastrain1afterfilter*)
	tPr_GT1_1_Max : HALioDi_Type; (*DI	Gaspressuremaximumgastrain1-line1*)
	tPr_GT1_1_Min : HALioDi_Type; (*DI	Gaspressurelowgastrain1-line1*)
	tPr_GT1_2_Max : HALioDi_Type; (*DI	Gaspressuremaximumgastrain1-line2*)
	tPr_GT1_2_Min : HALioDi_Type; (*DI	Gaspressurelowgastrain1-line2*)
	tPr_GT1_3_Max : HALioDi_Type; (*DI	Gaspressuremaximumgastrain1-line3*)
	tPr_GT1_3_Min : HALioDi_Type; (*DI	Gaspressurelowgastrain1-line3*)
	tPr_GT1_4_Max : HALioDi_Type; (*DI	Gaspressuremaximumgastrain1-line4*)
	tPr_GT1_4_Min : HALioDi_Type; (*DI	Gaspressurelowgastrain1-line4*)
	tPr_GT1_Max : HALioDi_Type; (*DI	Gaspressuremaximumgastrain1*)
	tPr_GT1_Min : HALioDi_Type; (*DI	Gaspressurelowgastrain1*)
	tPr_GT2_Max : HALioDi_Type; (*DI	Gaspressuremaximumgastrain2*)
	tPr_GT2_Min : HALioDi_Type; (*DI	Gaspressurelowgastrain2*)
	tPr_GT_Gas : HALioAi_Type; (*IF654gaspressure	*)
	tPr_GT_MinBefCompr : HALioDi_Type; (*DI	Gaspressurelowbeforegascompressor*)
	tPr_GT_Suct : HALioAi_Type; (*IF655suctionpressure	*)
	tPr_HW_Hi : HALioDi_Type; (*DIheatwaterpressurehigh*)
	tPr_HW_Hi1 : HALioDi_Type; (*DIheatwaterpressurehigh*)
	tPr_HW_Lo : HALioDi_Type; (*DIheatwaterpressurelow*)
	tPr_HW_Su_HT : HALioAi_Type; (*supply water pressure HT circuit*) (*OldName:AI_p_VL_HT; Cycle:5;*)
	tPr_HW_Su_LT : HALioAi_Type; (*supply water pressure LT circuit*) (*OldName:AI_p_VL_NT; Cycle:5;*)
	tPr_MGT_a_Filt : HALioAi_Type; (*AI main gas train pressure after filter [bar]*) (* OldName: AI_p_GT1; Cyclic: 2; *)
	tPr_MGT_sp : HALioAo_Type; (*AO pressure gas rail set point with Offset considered*) (*OldName:rPr_MGT_sp; Cycle:5;*)
	tPr_N2_Hi : HALioDi_Type; (*DIpressureN2high*)
	tPr_N2_Lo : HALioDi_Type; (*DIpressureN2low*)
	tPr_OilSkid_HP_DE : HALioAi_Type; (*AI OilSkid oil pressure in high pressure circuit to DE bearing*)
	tPr_OilSkid_HP_NDE : HALioAi_Type; (*AI OilSkid oil pressure in high pressure circuit to NDE bearing *)
	tPr_Oil_LPTC_In_A : HALioAi_Type; (*oil pressure LP turbo charger A inlet*) (*OldName:P_OEL_ND_EintrittA; Cycle:5;*)
	tPr_Oil_LPTC_In_B : HALioAi_Type; (*oil pressure LP turbo charger B inlet*) (*OldName:P_OEL_ND_EintrittB; Cycle:5;*)
	tPr_PC : HALioAi_Type; (*AI	Pressureprechamber*)
	tPr_PCG : HALioAi_Type; (*IF650prechambergaspressure	*)
	tPr_PCGBefComp_Lo : HALioDi_Type; (*DIsuctionpressureprechambergascompressorhigh*)
	tPr_PCGT : HALioAi_Type; (*AI	Gaspressureprechambergastrainafterfilter*)
	tPr_PCGT_Out : HALioAi_Type; (*AI Warning measuring signal failure - gas pressure after pre chamber gas pressure regulator*) (* OldName: AI_p_PCGT_Out; Cyclic: 2; *)
	tPr_PCGT_sp : HALioAo_Type; (*AO main gas train pressure - set point with Offset considered*) (*OldName:rPr_PCGT_sp; Cycle:5;*)
	tPr_PCG_GC_Dem : HALioDo_Type; (*DO	Demandprechampergascompressor*)
	tPr_PCG_Min : HALioDi_Type; (*DI	Prechambergascompressorpressureminimum*)
	tPr_PC_Diff : HALioAi_Type; (*IFF	-	IF652prechamberdiff.pressure	*)
	tPr_TCOF_EOF_DiffMax : HALioDi_Type; (*DI:Differencepressureturbochargeroilfilterhigh*)
	tPr_TC_EOF_After : HALioAi_Type; (*AIoilpressureafterturbochargeroilfilter,NUP62/AI_M_03_PI_062*)
	tPr_TC_EOF_Before : HALioAi_Type; (*AI:Oilpressureinfrontofturbochargeroilfilter,NUP61/AI_M_03_PI_061*)
	tPr_ThR_AirLo : HALioDi_Type; (*DIthermalreactorcompressedairpressurelow*)
	tPS400V_ENGIA_CB_On : HALioDi_Type; (*Supply disconnecting device 400VAC +ENGIA on*)
	tPulseMainsOk : HALioDo_Type; (*pulsemainsok*)
	tP_Act : ARRAY[0..2] OF HALioAi_Type; (*actualelectricpower[kW]*)
	tP_Act_AO : HALioAo_Type; (*actualpowerrelatedtorP_nomfilteredT=1s*)
	tP_GenC_Bloc : HALioDo_Type; (*DO:internalblockingsignal*)
	tP_GenC_Fix0SOn : HALioDo_Type; (*DO:nolimitingpowervalue-P-fixvalue0fromEUison*)
	tP_GenC_Fix1SOn : HALioDo_Type; (*DO:powervalue-P-fixvalue1fromEUison*)
	tP_GenC_Fix2SOn : HALioDo_Type; (*DO:powervalue-P-fixvalue2fromEUison*)
	tP_GenC_Fix3SOn : HALioDo_Type; (*DO:powervalue-P-fixvalue3fromEUison*)
	tP_GenC_Fix4SOn : HALioDo_Type; (*DO:powervalue-P-fixvalue4fromEUison*)
	tP_GenC_Fix5SOn : HALioDo_Type; (*DO:powervalue-P-fixvalue5fromEUison*)
	tP_GenC_SetEU : HALioAi_Type; (*AI:requestpowervaluefromEU*)
	tP_GenC_SetEUCOf : HALioDi_Type; (*DI:requestpowervaluefromEU-off(deactivate*)
	tP_GenC_SetEUCOn : HALioDi_Type; (*DI:requestpowervaluefromEU-on(activate*)
	tP_GenC_SetFix1EU : HALioDi_Type; (*DI:powervalue-P-fixvalue1fromEU*)
	tP_GenC_SetFix2EU : HALioDi_Type; (*DI:powervalue-P-fixvalue2fromEU*)
	tP_GenC_SetFix3EU : HALioDi_Type; (*DI:powervalue-P-fixvalue3fromEU*)
	tP_GenC_SetFix4EU : HALioDi_Type; (*DI:powervalue-P-fixvalue4fromEU*)
	tP_GenC_SetFix5EU : HALioDi_Type; (*DI:powervalue-P-fixvalue5fromEU*)
	tP_GenC_SOf : HALioDo_Type; (*DO:powervaluefonEUisoff*)
	tP_GenC_SOn : HALioDo_Type; (*DO:powervaluefonEUison*)
	tP_GT_Max_Backfire : HALioDi_Type; (*DI	gaspressurehigh-backfire*)
	tP_Lo : HALioDo_Type; (*DOpowerlow(foropeningGCB*)
	tP_Red_Active : HALioDo_Type; (*powerreductionactive-anykind-HALIOOutput*)
	tP_Red_AI_Norm : HALioAi_Type; (*Externalpowerreduction	*)
	tP_Red_CH4Active : HALioDi_Type; (* Power limitation because of CH4 content active *) (*OldName: CH4RED_0; Cyclic:5*)
	tP_Red_GasPrActive : HALioDi_Type; (* Power limitation because OF gas pressure active*) (*OldName: GD_RED_0; Cyclic:5;*)
	tP_Red_Norm : HALioAo_Type; (*powerreduction*)
	tP_Red_SuctPrActive : HALioDi_Type; (* Power limitation because OF suction pressure active*) (*OldName: SD_RED_0; Cyclic:5;*)
	tP_Set_ExtAI_Norm : HALioAi_Type; (*Externalpowersetpoint	*)
	tQLim_GenC_Act : HALioDo_Type; (*DO:reactivepowerlimitation(Plim*)
	tQLim_GenC_SetEU : HALioAi_Type; (*AI:setpointreactivepowerlimitation(Qlim*)
	tQLim_GenC_SetEUCOf : HALioDi_Type; (*DI:setpointreactivepowerlimitation(Qlim*)
	tQLim_GenC_SetEUCOn : HALioDi_Type; (*DI:setpointreactivepowerlimitation(Qlim*)
	tQLim_GenC_SOf : HALioDo_Type; (*DO:reactivepowerlimiting(QLim*)
	tQLim_GenC_SOn : HALioDo_Type; (*DO:reactivepowerlimiting(QLim*)
	tQPC_GenC_SetEUCOf : HALioDi_Type; (*DI:setpointreactivepowercharacteristicsCOS(phi*)
	tQPC_GenC_SetEUCOn : HALioDi_Type; (*DI:setpointreactivepowercharacteristicsCOS(phi*)
	tQPC_GenC_SOf : HALioDo_Type; (*DO:reactivepowercharacteristicsCOS(phi*)
	tQPC_GenC_SOn : HALioDo_Type; (*DO:reactivepowercharacteristicsCOS(phi*)
	tQUC_GenC_SetEUCOf : HALioDi_Type; (*DI:setpointreactivepowercharacteristicsQ=f(U*)
	tQUC_GenC_SetEUCOn : HALioDi_Type; (*DI:setpointreactivepowercharacteristicsQ=f(U*)
	tQUC_GenC_SOf : HALioDo_Type; (*DO:reactivepowercharacteristicsQ=f(U*)
	tQUC_GenC_SOn : HALioDo_Type; (*DO:reactivepowercharacteristicsQ=f(U*)
	tQU_GenC_Set : HALioAi_Type; (*AI:setpointgeneratorvoltageforrectivepowercontrol[%]vorEU*)
	tQ_Act : ARRAY[0..2] OF HALioAi_Type; (*actualreactivepower[kVar]*)
	tQ_GenC_Act : HALioAo_Type; (*AO:reactivepoweractuelevalue*)
	tQ_GenC_CUST : HALioAi_Type; (*costumiz:scalingvalueforreactivepower(Q*)
	tQ_GenC_Fix1SOn : HALioDo_Type; (*DO:reactivepower(Q*)
	tQ_GenC_Fix2SOn : HALioDo_Type; (*DO:reactivepower(Q*)
	tQ_GenC_Fix3SOn : HALioDo_Type; (*DO:reactivepower(Q*)
	tQ_GenC_Fix4SOn : HALioDo_Type; (*DO:reactivepower(Q*)
	tQ_GenC_Fix5SOn : HALioDo_Type; (*DO:reactivepower(Q*)
	tQ_GenC_SetEU : HALioAi_Type; (*AI:setpointreactivepowercharacteristic(Q*)
	tQ_GenC_SetEUCOf : HALioDi_Type; (*DI:setpointreactivepowercharacteristic(Q*)
	tQ_GenC_SetEUCOn : HALioDi_Type; (*DI:setpointreactivepowercharacteristic(Q*)
	tQ_GenC_SetFix1EU : HALioDi_Type; (*DI:reactivepower(Q*)
	tQ_GenC_SetFix2EU : HALioDi_Type; (*DI:reactivepower(Q*)
	tQ_GenC_SetFix3EU : HALioDi_Type; (*DI:reactivepower(Q*)
	tQ_GenC_SetFix4EU : HALioDi_Type; (*DI:reactivepower(Q*)
	tQ_GenC_SetFix5EU : HALioDi_Type; (*DI:reactivepower(Q*)
	tQ_GenC_SOf : HALioDo_Type; (*DO:reactivepowercharacteristic(Q*)
	tQ_GenC_SOn : HALioDo_Type; (*DO:reactivepowercharacteristic(Q*)
	TransformerTrip : BOOL; (*DItransformerfailure*)
	TransformerWarning : BOOL; (*DItransformerfailure*)
	tRdy_MSy : HALioDo_Type; (*enginereadyforMSY*)
	tRelAux : HALioDi_Type; (*DIreleaseengineoperationfromauxiliarieswithmonitoring*)
	tRelAuxNoMon : HALioDi_Type; (*DIreleaseengineoperationfromauxiliarieswithnomonitoring*)
	tRelEngOpFromGSy : HALioDi_Type; (*DIreleaseengineoperationfrom'gemeinsame'synchronization*)
	tRelGasPlant : HALioDi_Type; (*DI	Releasefromgasplantmissing.FALSE=Missing*)
	tRelMainGVext : HALioDi_Type; (*DIreleasemaingasvalvefromexternal*)
	tRel_BS : HALioDi_Type; (*DIreleaseblackstart*)
	tRel_ER_Fan : HALioDo_Type; (*DOdemandVE>min.speed*)
	tRel_ER_FC : HALioDo_Type; (*DOreleasefrequencyconverterforroomVE*)
	tRel_ER_PurgeCycle : HALioDi_Type; (*DIreleasepurgecycle*)
	tRel_I : HALioDi_Type; (*DIreleaseislandoperation*)
	tRel_LS : HALioDi_Type; (*DIreleaseloadshedding*)
	tRel_MasCtr : HALioDi_Type; (*releasefrommastercontrol*)
	tRel_Sync_Load : HALioDo_Type; (*DO:releaseofsynchronizationandload*)
	tRel_U_Sel_LS_Gen : HALioDi_Type; (*ReleasevoltageselectionLS-Generator*)
	tReq_PeakLoad : HALioDi_Type; (*requestpeakload*)
	tReq_Test : HALioDi_Type; (*requesttestmode*)
	tResetRemExt : HALioDi_Type; (*resetremoteexternal*)
	tResetRemoteExt : HALioDi_Type; (*resetremoteexternal*)
	tResetTrip : HALioDo_Type; (*DOresettrippulse*)
	tResetWarning : HALioDo_Type; (*DOresetwarningpulse*)
	tRMC_SetCOf : HALioDi_Type; (*DI:regulationmargincontrol-off(deactivate*)
	tRMC_SetCOn : HALioDi_Type; (*DI:regulationmargincontrol-on(activate*)
	tRMC_SOf : HALioDo_Type; (*DO:regulationmargincontrolisoff*)
	tRMC_SOn : HALioDo_Type; (*DO:regulationmargincontrolison*)
	tRotatingLight : HALioDo_Type; (*DOrotatinglightyellow*)
	tRSE_SetEUCOf : HALioDi_Type; (* DI: reset decoupling RSE from EU (ERDF) *) (*OldName:DI_RDEmRSE PV;Cycle:2;*)
	tRSE_SetEUCOn : HALioDi_Type; (* DI: set decoupling RSE from EU (ERDF) *) (*OldName:DI_SDEmRSE PV;Cycle:2;*)
	tRSE_SOn : HALioDo_Type; (* DO: decoupling RSE from EU (ERDF)							*)
	tSafetyLoop_EmStop : HALioDi_Type; (*safetyloopemergencystopok*)
	tSafetyLoop_Eng : HALioDi_Type; (*safetyloopengine*)
	tSafetyLoop_Gas : HALioDi_Type; (*DIsafetyloopgasok*)
	tSafetyLoop_HWC : HALioDi_Type; (*safetyloopheatwatercircuitok*)
	tScavFanCB_trip : HALioDi_Type; (*DIexhaustgasscavengingfancircuitbreakertripped*)
	tScavFanCoOn : HALioDo_Type; (*DOscavengingfancomandON*)
	tScavFanFC_P_Lo : HALioDi_Type; (*DIexhaustgasscavengingfanfrequencyconverterpowerlow*)
	tScavFanFC_Rdy : HALioDi_Type; (*DIexhaustgasscavengingfanfrequencyconverterreadyforoperation*)
	tScavFanOp : HALioDi_Type; (*DIexhaustgasscavengingfanoperating*)
	tScavFan_Sp : HALioAo_Type; (*AOscavengingfansetpoint*)
	tScavVaClosed : HALioDi_Type; (*DIscavengingvalveclosed*)
	tScavVaCoClose : HALioDo_Type; (*DOscavengingvalvecommandclose*)
	tScavVaCoOpen : HALioDo_Type; (*DOscavengingvalvecommandopen*)
	tScavVaFailure : HALioDi_Type; (*DIscavengingvalvefailure*)
	tScavVaOpened : HALioDi_Type; (*DIscavengingvalveopened*)
	tSelGasTyp : HALioDi_Type; (*DI:Selectiongastype-general*)
	tSelGasTyp2 : HALioDi_Type; (*DI:Selectiongastype2*)
	tSelGasTyp3 : HALioDi_Type; (*DI:Selectiongastype3*)
	tSelGasTyp4 : HALioDi_Type; (*DI:Selectiongastype4*)
	tSet_ER_Fan_Min : HALioDo_Type; (*DOdemandVEmin.speed*)
	tSGM_DirStepper1 : HALioDo_Type; (*DO SGM direction stepper 1 *)
	tSGM_DirStepper2 : HALioDo_Type; (*DO SGM direction stepper 2 *)
	tSGM_DirStepper3 : HALioDo_Type; (*DO SGM direction stepper 3 *)
	tSGM_EnabStepper1 : HALioDo_Type; (*DO SGM enable stepper 1 *)
	tSGM_EnabStepper2 : HALioDo_Type; (*DO SGM enable stepper 2 *)
	tSGM_EnabStepper3 : HALioDo_Type; (*DO SGM enable stepper 3 *)
	tSignal1R1 : HALioDo_Type; (*DOsignallamp1redcontinuouslight*)
	tSignal1R2 : HALioDo_Type; (*DOsignallamp2redcontinuouslight*)
	tSignalG1 : HALioDo_Type; (*DOsignallamp1greencontinuouslight*)
	tSignalG2 : HALioDo_Type; (*DOsignallamp2greencontinuouslight*)
	tSignalR1 : HALioDo_Type; (*DOsignallamp1redflashing*)
	tSignalR2 : HALioDo_Type; (*DOsignallamp2redflashing*)
	tSignalY1 : HALioDo_Type; (*DOsignallamp1yellowcontinuouslight*)
	tSignalY2 : HALioDo_Type; (*DOsignallamp2yellowcontinuouslight*)
	tStUpSpeed : HALioDo_Type; (*DOstartupspeed*)
	tSys_Run : HALioDo_Type; (*RUNDigitaOutbittoHAL*)
	tSys_Run1 : HALioDo_Type; (*RUNDigitaOutbittoHAL*)
	tSys_Run2 : HALioDo_Type; (*RUNDigitaOutbittoHAL*)
	tSys_Run3 : HALioDo_Type; (*RUNDigitaOutbittoHAL*)
	tSys_Run4 : HALioDo_Type; (*RUNDigitaOutbittoHAL*)
	tSys_Run5 : HALioDo_Type; (*RUNDigitaOutbittoHAL*)
	tSys_Run6 : HALioDo_Type; (*RUNDigitaOutbittoHAL*)
	tSy_N_Down : HALioDi_Type; (*DIexternalspeedmatchingDOWN*)
	tSy_N_Up : HALioDi_Type; (*DIexternalspeedmatchingUP*)
	tS_Act : ARRAY[0..2] OF HALioAi_Type; (* appearent power [kV] *)
	tTBMode : HALioDi_Type; (*DItestbenchmode*)
	tTCOP_CB_On : HALioDi_Type; (*Failure Pump Turbocharger pressure*)
	tTCOP_Grid : HALioDi_Type; (*turbo charger oil pump mains voltage ok*)
	tTCOP_GridOk : HALioDo_Type; (*turbo charger oil pump mains voltage ok*)
	tTCOP_Op : HALioDi_Type; (*DIturbochargeroilpumpoperating*)
	tTCOP_UPS_CB_On : HALioDi_Type; (*Circuit breaker tripped Prelubrication oil pump / Cool down oilpump*)
	tTC_EOP_On : HALioDo_Type; (*DO:Engineoilpump,NPO601*)
	tTC_EOP_OnUSV : HALioDo_Type; (*DO:Engineoilpump,NPO601viaUSV*)
	tThR_Contactor : HALioDo_Type; (*DOthermalreactorcontactor*)
	tThR_CV_CDec : HALioDo_Type; (*DOthermalreactorgascontrolvalvecommanddecrease*)
	tThR_CV_CInc : HALioDo_Type; (*DOthermalreactorgascontrolvalvecommandincrease*)
	tThR_EH11 : HALioDo_Type; (*DOthermalreactorelectricalheatingelementgroup1output1*)
	tThR_EH12 : HALioDo_Type; (*DOthermalreactorelectricalheatingelementgroup1output2*)
	tThR_EH13 : HALioDo_Type; (*DOthermalreactorelectricalheatingelementgroup1output3*)
	tThR_EH21 : HALioDo_Type; (*DOthermalreactorelectricalheatingelementgroup2output1*)
	tThR_EH22 : HALioDo_Type; (*DOthermalreactorelectricalheatingelementgroup2output2*)
	tThR_EH23 : HALioDo_Type; (*DOthermalreactorelectricalheatingelementgroup2output3*)
	tThR_EH31 : HALioDo_Type; (*DOthermalreactorelectricalheatingelementgroup3output1*)
	tThR_EH32 : HALioDo_Type; (*DOthermalreactorelectricalheatingelementgroup3output2*)
	tThR_EH33 : HALioDo_Type; (*DOthermalreactorelectricalheatingelementgroup3output3*)
	tThR_ErrLamp : HALioDo_Type; (*DOthermalreactorfailurelamp*)
	tThR_GT_COn1 : HALioDo_Type; (*DO1thermalreactorgasinjectioncommandon*)
	tThR_GT_COn2 : HALioDo_Type; (*DO2thermalreactorgasinjectioncommandon*)
	tThR_LampTest : HALioDi_Type; (*DIthermalreactorlamptest*)
	tThR_RunLamp : HALioDo_Type; (*DOthermalreactoroperatinglamp*)
	tThR_SL : HALioDi_Type; (*DIthermalreactorsafetyloop*)
	tThR_Swth_On : HALioDi_Type; (*DIthermalreactoroperationswitchon*)
	tThR_Val_Air : HALioDo_Type; (*DOthermalreactorpurgeairvalve*)
	tThR_Val_CCylIn : HALioDo_Type; (*DOthermalreactorflapcommandmoveincylinder*)
	tThR_Val_CCylOut : HALioDo_Type; (*DOthermalreactorflapcommandmoveoutcylinder*)
	tTransformerTrip : HALioDi_Type; (*DItransformerfailure*)
	tTransformerWarning : HALioDi_Type; (*DItransformerfailure*)
	tTurnRel : HALioDo_Type; (*DOcrankshaftturningdevicerelease*)
	tT_AirER : HALioAi_Type; (*AIairengineroomtemperature[C]*)
	tT_AirER_Ext_Hi : HALioDi_Type; (*DIairengineroomtemperatureexternalhigh*)
	tT_AirER_Ext_Hi1 : HALioDi_Type; (*DIroomtemperaturelimit*)
	tT_AirER_Ext_Hi2 : HALioDi_Type; (*DIroomtemperaturelimit*)
	tT_AirER_Ext_Hi3 : HALioDi_Type; (*DIroomtemperaturelimit*)
	tT_AirIFCP_Hi : HALioDi_Type; (*DIairtemperatureinterfacecontrolpanelhigh*)
	tT_AirIn : HALioAi_Type;
	tT_AirOutdoor : HALioAi_Type; (*AItemperatureairoutdoor*)
	tT_AO_Gen_T_In : HALioAo_Type; (*Generatorairinlettemperatureforgen.controler*)
	tT_Cat : HALioAi_Type; (*AIcatalysttemperature*)
	tT_CBearing_Hi : HALioDi_Type; (*Warning Temperature conrod bearing*)
	tT_CBearing_HiHi : HALioDi_Type; (*Shut down Temperature conrod bearing*)
	tT_ChCW_Hi : HALioDi_Type; (*DIchargecoolingwatertemperaturehigh*)
	tT_Ch_T1HP : HALioAi_Type; (*chargetemperaturebeforehighpressureTC[°C]*)
	tT_Ch_T1HP_A : HALioAi_Type; (*chargetemperaturebeforehighpressureTCA[°C]*)
	tT_Ch_T1HP_B : HALioAi_Type; (*chargetemperaturebeforehighpressureTCB[°C]*)
	tT_Ch_T1LP : HALioAi_Type; (*AI charge temperature before low-pressure turbocharger (= intake air) [°C]*)
	tT_Ch_T1LP_A : HALioAi_Type; (*AI charge temperature before low-pressure turbocharger bank A (= intake air) [°C]*)
	tT_Ch_T1LP_B : HALioAi_Type; (*AI charge temperature before low-pressure turbocharger bank B (= intake air) [°C]*)
	tT_Ch_T2HP : HALioAi_Type; (*AI charge temperature after high-pressure turbocharger [°C]*)
	tT_Ch_T2HP_A : HALioAi_Type; (*AI charge temperature after high-pressure turbocharger bank A [°C]*)
	tT_Ch_T2HP_B : HALioAi_Type; (*AI charge temperature after high-pressure turbocharger bank B [°C]*)
	tT_Ch_T2LP : HALioAi_Type; (*AI charge temperature after low-pressure turbocharger [°C]*)
	tT_Ch_T2LP_A : HALioAi_Type; (*AI charge temperature after low-pressure turbocharger bank A [°C]*)
	tT_Ch_T2LP_B : HALioAi_Type; (*AI charge temperature after low-pressure turbocharger bank B [°C]*)
	tT_Ch_T2s : HALioAi_Type; (*AItemperaturechargeafterthrottlevalve*)
	tT_Ch_T2s_A : HALioAi_Type; (*chargetemperaturet2'afterthrottlevalveA[°C]*)
	tT_Ch_T2s_B : HALioAi_Type; (*chargetemperaturet2'afterthrottlevalveB[°C]*)
	tT_CO2_Hi : HALioDi_Type; (*DICO2temperaturereactorchamberhigh*)
	tT_DAI : HALioAi_Type; (*AI Air temperature before DAI shut off valve[°C]*)
	tT_ECW : HALioAi_Type; (*AItemperatureenginecoolingwater*)
	tT_ECWbEng : HALioAi_Type; (*Engine jacket water temperature befor Engine*)
	tT_ECW_AfEng : HALioAi_Type; (*AItemperatureenginecoolingwaterafterengine[°C]*)
	tT_ECW_Ext_Hi : HALioDi_Type; (*DItemperatureenginecoolingwaterhighexternal*)
	tT_ECW_PreH_Hi : HALioDi_Type; (*DItemperatureenginecoolingwaterpreheatinghigh*)
	tT_ECW_PreH_HiHi : HALioDi_Type; (*DItemperatureenginecoolingwaterpreheatinghighhigh*)
	tT_EGafHeEx1 : HALioAi_Type; (*IF660exh.gastemp.aft.heatexch.1*)
	tT_EGafHeEx2 : HALioAi_Type; (*IF661exh.gastemp.aft.heatexch.2*)
	tT_EGaHE : HALioAi_Type; (*AIexhaustgastemperatureafterheatexchanger*)
	tT_EGaHE1 : HALioAi_Type; (*AIexhaustgastemperatureafterheatexchanger1*)
	tT_EGaHE2 : HALioAi_Type; (*AIexhaustgastemperatureafterheatexchanger2*)
	tT_EGaHPTC_A : HALioAi_Type; (* AI: Exhaust gas temperatur after high-pressure turbocharger A  (M.02-TI-167) *) (* OldName: AI_M_02_TI_167	; Cyclic: 5; *)
	tT_EGaHPTC_B : HALioAi_Type; (* AI: Exhaust gas temperatur after high-pressure turbocharger A  (M.02-TI-267) *) (* OldName: AI_M_02_TI_267	; Cyclic: 5; *)
	tT_EGaLPTC_A : HALioAi_Type; (*AIexhaustgastemperatureafterlowpressureturbochargerA*)
	tT_EGaLPTC_B : HALioAi_Type; (*AIexhaustgastemperatureafterlowpressureturbochargerB*)
	tT_EGaTC : HALioAi_Type; (*AIexhaustgastemperatureafterturbocharger*)
	tT_EGbHPTC_A : HALioAi_Type; (* AI: Exhaust gas temperature before high-pressure turbocharger A  (M.02-TI-166) *) (* OldName: AI_M_02_TI_166	; Cyclic: 5; *)
	tT_EGbHPTC_B : HALioAi_Type; (* AI: Exhaust gas temperature before high-pressure turbocharger B  (M.02-TI-266) *) (* OldName: AI_M_02_TI_266	; Cyclic: 5; *)
	tT_EGbTC : HALioAi_Type; (*AIexhaustgastemperaturebeforeturbocharger*)
	tT_EG_Cyl : ARRAY[0..24] OF HALioAi_Type; (*cylinder exhaust gas temperature*)
	tT_EO : HALioAi_Type; (*AItemperatureengineoil*)
	tT_EOP_After : HALioAi_Type; (*AI:Oiltemperatureafteroilpump,NUT71/AI_M_03_TI_071*)
	tT_EO_Gear_Max : HALioDi_Type; (*DI:Oiltemperaturehightransmission*)
	tT_EO_Preheating : HALioAi_Type; (*AI:Oiltemperaturepreheating,NUT78/AI_M_03_TI_078*)
	tT_EO_PreH_Hi : HALioDi_Type; (*Temperaturbegrenzer Vorwärmung Motoröl (Warnung)*)
	tT_EO_PreH_HiHi : HALioDi_Type; (*Temperaturbegrenzer Vorwärmung Motoröl*)
	tT_GenAirOut : HALioAi_Type; (*Exhaust air Temperature*)
	tT_Gen_Bear_A_Act : HALioAi_Type; (*generatorbearingAtemperaturesignal*)
	tT_Gen_Bear_B_Act : HALioAi_Type; (*generatorbearingBtemperaturesignal*)
	tT_Gen_Wind : HALioAi_Type; (*actualgeneratorwindingtemperaturesignal*)
	tT_Gen_Wind_Act_L1 : HALioAi_Type; (*generatorwindingtemperaturesignal,windingphase1*)
	tT_Gen_Wind_Act_L2 : HALioAi_Type; (*generatorwindingtemperaturesignal,windingphase2*)
	tT_Gen_Wind_Act_L3 : HALioAi_Type; (*generatorwindingtemperaturesignal,windingphase3*)
	tT_GT : HALioAi_Type; (*IF657gastemperature	*)
	tT_GT_Ok : HALioDi_Type; (*DI	GastemperatureOK*)
	tT_HW_Hi : HALioDi_Type; (*DIheatwatertemperaturehigh*)
	tT_HW_Hi1 : HALioDi_Type; (*DIheatwatertemperaturehigh*)
	tT_HW_Re : HALioAi_Type; (*AItemperatureheatwaterreturn*)
	tT_HW_ReAfEC : HALioAi_Type; (*AItemperatureheatwaterreturnafteremergencycooler*)
	tT_HW_ReBeEng : HALioAi_Type; (*AItemperatureheatwaterreturnbeforeengine*)
	tT_HW_Re_LT : HALioAi_Type; (*AItemperatureheatwaterreturnlowtemp.circuit[°C]*)
	tT_HW_Su : HALioAi_Type; (*AItemperatureheatwatersupply*)
	tT_Su_PriCirc : HALioAi_Type; (*AI supply water temperature primary circuit [°C]*) (*STM*)
	tT_Re_PriCirc : HALioAi_Type; (*AI return water temperature primary circuit [°C]*) (*STM*)
	tT_Su_SecCirc : HALioAi_Type; (*AI supply water temperature secondary circuit [°C]*) (*STM*)
	tT_Re_SecCirc : HALioAi_Type; (*AI return water temperature secondary circuit [°C]*) (*STM*)
	tP_Heat : HALioAi_Type; (*AI heating power engine heat water circuit [kW]*) (*STM 2*)
	tT_HW_Su_LT : HALioAi_Type; (*AItemperatureheatwatersupplylowtemp.circuit[°C]*)
	tT_OilSkid_Supply : HALioAi_Type; (*AI OilSkid supply temperature*)
	tT_OilSkid_Tank : HALioAi_Type; (*AI OilSkid tank temperature*)
	tT_PCGAfCo : HALioAi_Type; (*AItemperatureprechambergasaftercooler*)
	tT_PCGAfComp_Hi : HALioDi_Type; (*DItemperatureprechambergascompressoroutlethigh*)
	tT_PCGT : HALioAi_Type; (*AI	Prechambergastemperature*)
	tT_PlateHE : HALioAi_Type; (*AIplatetemperatureheatexchanger*)
	tT_ThR_Chamber1_1 : HALioAi_Type; (*thermalreactorchambertemperature1_1*)
	tT_ThR_Chamber1_2 : HALioAi_Type; (*thermalreactorchambertemperature1_2*)
	tT_ThR_Chamber2_1 : HALioAi_Type; (*thermalreactorchambertemperature2_1*)
	tT_ThR_Chamber2_2 : HALioAi_Type; (*thermalreactorchambertemperature2_2*)
	tT_ThR_ChamberLo : HALioDi_Type; (*DIthermalreactorchambertemperaturelow*)
	tT_ThR_Comp : HALioAi_Type; (*thermalreactorcompensationtemperature*)
	tT_ThR_In : HALioAi_Type; (*thermalreactorinlettemperature*)
	tT_ThR_Out : HALioAi_Type; (*thermalreactoroutlettemperature*)
	tT_ThR_Swg_Hi : HALioDi_Type; (*DIthermalreactorswitchgeartemperaturehigh*)
	tUPS_CB_On : HALioDi_Type; (*Circuit breaker tripped supply UPS*)
	tUPS_Ok : HALioDi_Type; (*failureuninterruptedpowersupply*)
	TurnRel : BOOL; (*DOcrankshaftturningdevicerelease*)
	tU_Adj_Minus : HALioDi_Type; (*VoltageadjustmentMinus*)
	tU_Adj_Plus : HALioDi_Type; (*VoltageadjustmentPlus*)
	tU_Avg : ARRAY[0..2] OF HALioAi_Type; (*actualgeneratoraveragevoltage*)
	tU_GenC_SetCUST : HALioAi_Type; (*costumiz:scalingvalueforgeneratorvoltageforreactivepowerfromEU*)
	tU_GenDiode_Fail : HALioDi_Type; (*generatordiodealarm*)
	tU_GenOverVolt : HALioDi_Type; (*failuregeneratorovervoltageprotection*)
	tU_Gen_Contr_Fail : HALioDi_Type; (*generatorvoltageregulatorfailure*)
	tU_Gen_Dec : HALioDi_Type; (*digitalinputforvoltageadjustmentbyMMU(decreasing*)
	tU_Gen_Exc : HALioAi_Type; (*actualexcitationvoltagesignal,filteredandscaled*)
	tU_Gen_Inc : HALioDi_Type; (*digitalinputforvoltageadjustmentbyMMU(increasing*)
	tU_Gen_LimHi : ARRAY[0..2] OF HALioDi_Type; (*generatorvoltagetoohigh*)
	tU_Gen_LimLo : ARRAY[0..2] OF HALioDi_Type; (*generatorvoltagetoolow*)
	tU_Gen_LimLo2 : ARRAY[0..2] OF HALioDi_Type; (*generatorvoltagetoolow2*)
	tU_L1L2 : ARRAY[0..2] OF HALioAi_Type; (* generator voltage phase 1_2 [V] *)
	tU_L1N : ARRAY[0..2] OF HALioAi_Type; (* generator voltage phase 1_N [V] *)
	tU_L2L3 : ARRAY[0..2] OF HALioAi_Type; (* generator voltage phase 2_3 [V] *)
	tU_L2N : ARRAY[0..2] OF HALioAi_Type; (* generator voltage phase 2_N [V] *)
	tU_L3L1 : ARRAY[0..2] OF HALioAi_Type; (* generator voltage phase 3_1 [V] *)
	tU_L3N : ARRAY[0..2] OF HALioAi_Type; (* generator voltage phase 3_N [V] *)
	tU_MidPos : HALioDo_Type; (*Voltagemiddleposition*)
	tU_Minus : HALioDo_Type; (*Voltageminus*)
	tU_MMD_Asy : ARRAY[0..2] OF HALioDi_Type; (*generatorvoltagenegativesequencetoohigh*)
	tU_MMD_Synch1 : ARRAY[0..2] OF HALioAi_Type; (*synchronization voltage 1*)
	tU_MMD_Synch2 : ARRAY[0..2] OF HALioAi_Type; (*synchronization voltage 2*)
	tU_Plus : HALioDo_Type; (*Voltageplus*)
	tU_StarterBat_Lo : HALioDi_Type; (*DIvoltagestarterbatterylow*)
	tU_Starter_engage1 : HALioAi_Type; (*Start motor 1 voltage*)
	tU_Starter_engage2 : HALioAi_Type; (*Start motor 2 voltage*)
	tU_Starter_engage3 : HALioAi_Type; (*Start motor 3 voltage*)
	tVol_GT : HALioAi_Type; (*IF658gasquantity	*)
	tWG_Dem : HALioDo_Type; (*wastegateposition*)
	tWG_A_Dem : HALioDo_Type; (*wastegatepositionA*)
	tWG_B_Dem : HALioDo_Type; (*wastegatepositionB*)
	T_AirER : INT; (*AIairengineroomtemperature[C]*)
	T_AirER_Ext_Hi : BOOL; (*DIairengineroomtemperatureexternalhigh*)
	T_AirER_Ext_Hi1 : BOOL; (*DIroomtemperaturelimit*)
	T_AirER_Ext_Hi2 : BOOL; (*DIroomtemperaturelimit*)
	T_AirER_Ext_Hi3 : BOOL; (*DIroomtemperaturelimit*)
	T_AirIFCP_Hi : BOOL; (*DIairtemperatureinterfacecontrolpanelhigh*)
	T_AirIn : INT;
	T_AirOutdoor : INT; (*AItemperatureairoutdoor*)
	T_AO_Gen_T_In : INT; (*Generatorairinlettemperatureforgen.controler*)
	T_Cat : INT; (*AIcatalysttemperature*)
	T_CBearing_Hi : BOOL; (*Warning Temperature conrod bearing*)
	T_CBearing_HiHi : BOOL; (*Shut down Temperature conrod bearing*)
	T_ChCW_Hi : BOOL; (*DIchargecoolingwatertemperaturehigh*)
	T_Ch_T1HP : INT; (*chargetemperaturebeforehighpressureTC[°C]*)
	T_Ch_T1HP_A : INT; (*chargetemperaturebeforehighpressureTCA[°C]*)
	T_Ch_T1HP_B : INT; (*chargetemperaturebeforehighpressureTCB[°C]*)
	T_Ch_T2s : INT; (*AItemperaturechargeafterthrottlevalve*)
	T_Ch_T2s_A : INT; (*chargetemperaturet2'afterthrottlevalveA[°C]*)
	T_Ch_T2s_B : INT; (*chargetemperaturet2'afterthrottlevalveB[°C]*)
	T_CO2_Hi : BOOL; (*DICO2temperaturereactorchamberhigh*)
	T_DAI : INT; (*air temperature before DAI shut off valve[°C]*)
	T_ECW : INT; (*AItemperatureenginecoolingwater*)
	T_ECWbEng : INT; (*Engine jacket water temperature befor Engine*)
	T_ECW_AfEng : INT; (*AItemperatureenginecoolingwaterafterengine[°C]*)
	T_ECW_Ext_Hi : BOOL; (*DItemperatureenginecoolingwaterhighexternal*)
	T_ECW_PreH_Hi : BOOL; (*DItemperatureenginecoolingwaterpreheatinghigh*)
	T_ECW_PreH_HiHi : BOOL; (*DItemperatureenginecoolingwaterpreheatinghighhigh*)
	T_EGafHeEx1 : INT; (*IF660exh.gastemp.aft.heatexch.1*)
	T_EGafHeEx2 : INT; (*IF661exh.gastemp.aft.heatexch.2*)
	T_EGaHE : INT; (*AIexhaustgastemperatureafterheatexchanger*)
	T_EGaHE1 : INT; (*AIexhaustgastemperatureafterheatexchanger1*)
	T_EGaHE2 : INT; (*AIexhaustgastemperatureafterheatexchanger2*)
	T_EGaHPTC_A : INT; (* AI: Exhaust gas temperatur after high-pressure turbocharger A  (M.02-TI-167) *) (* OldName: AI_M_02_TI_167	; Cyclic: 5; *)
	T_EGaHPTC_B : INT; (* AI: Exhaust gas temperatur after high-pressure turbocharger A  (M.02-TI-267) *) (* OldName: AI_M_02_TI_267	; Cyclic: 5; *)
	T_EGaLPTC_A : INT; (*AIexhaustgastemperatureafterlowpressureturbochargerA*)
	T_EGaLPTC_B : INT; (*AIexhaustgastemperatureafterlowpressureturbochargerB*)
	T_EGaTC : INT; (*AIexhaustgastemperatureafterturbocharger*)
	T_EGbHPTC_A : INT; (* AI: Exhaust gas temperature before high-pressure turbocharger A  (M.02-TI-166) *) (* OldName: AI_M_02_TI_166	; Cyclic: 5; *)
	T_EGbHPTC_B : INT; (* AI: Exhaust gas temperature before high-pressure turbocharger B  (M.02-TI-266) *) (* OldName: AI_M_02_TI_266	; Cyclic: 5; *)
	T_EGbTC : INT; (*AIexhaustgastemperaturebeforeturbocharger*)
	T_EG_Cyl : ARRAY[0..24] OF INT; (*cylinder exhaust gas temperature*)
	T_EO : INT; (*AItemperatureengineoil*)
	T_EOP_After : INT; (*AI:Oiltemperatureafteroilpump,NUT71/AI_M_03_TI_071*)
	T_EO_Gear_Max : BOOL; (*DI:Oiltemperaturehightransmission*)
	T_EO_Preheating : INT; (*AI:Oiltemperaturepreheating,NUT78/AI_M_03_TI_078*)
	T_EO_PreH_Hi : BOOL; (*Temperaturbegrenzer Vorwärmung Motoröl (Warnung)*)
	T_EO_PreH_HiHi : BOOL; (*Temperaturbegrenzer Vorwärmung Motoröl*)
	T_GenAirOut : INT; (*Exhaust air Temperature*)
	T_Gen_Bear_A_Act : INT; (*generatorbearingAtemperaturesignal*)
	T_Gen_Bear_B_Act : INT; (*generatorbearingBtemperaturesignal*)
	T_Gen_Wind : INT; (*actualgeneratorwindingtemperaturesignal*)
	T_Gen_Wind_Act_L1 : INT; (*generatorwindingtemperaturesignal,windingphase1*)
	T_Gen_Wind_Act_L2 : INT; (*generatorwindingtemperaturesignal,windingphase2*)
	T_Gen_Wind_Act_L3 : INT; (*generatorwindingtemperaturesignal,windingphase3*)
	T_GT : INT; (*IF657gastemperature	*)
	T_GT_Ok : BOOL; (*DI	GastemperatureOK*)
	T_HW_Hi : BOOL; (*DIheatwatertemperaturehigh*)
	T_HW_Hi1 : BOOL; (*DIheatwatertemperaturehigh*)
	T_HW_Re : INT; (*AItemperatureheatwaterreturn*)
	T_HW_ReAfEC : INT; (*AItemperatureheatwaterreturnafteremergencycooler*)
	T_HW_ReBeEng : INT; (*AItemperatureheatwaterreturnbeforeengine*)
	T_HW_Re_LT : INT; (*AItemperatureheatwaterreturnlowtemp.circuit[°C]*)
	T_HW_Su : INT; (*AItemperatureheatwatersupply*)
	T_HW_Su_LT : INT; (*AItemperatureheatwatersupplylowtemp.circuit[°C]*)
	T_Su_PriCirc : INT; (*AI supply water temperature primary circuit [°C]*) (*STM*)
	T_Re_PriCirc : INT; (*AI return water temperature primary circuit [°C]*) (*STM*)
	T_Su_SecCirc : INT; (*AI supply water temperature secondary circuit [°C]*) (*STM*)
	T_Re_SecCirc : INT; (*AI return water temperature secondary circuit [°C]*) (*STM*)
	T_Ch_T1LP : INT; (*AI charge temperature before low-pressure turbocharger (= intake air) [°C]*)
	T_Ch_T1LP_A : INT; (*AI charge temperature before low-pressure turbocharger bank A (= intake air) [°C]*)
	T_Ch_T1LP_B : INT; (*AI charge temperature before low-pressure turbocharger bank B (= intake air) [°C]*)
	T_Ch_T2LP : INT; (*AI charge temperature after low-pressure turbocharger [°C]*)
	T_Ch_T2LP_A : INT; (*AI charge temperature after low-pressure turbocharger bank A [°C]*)
	T_Ch_T2LP_B : INT; (*AI charge temperature after low-pressure turbocharger bank B [°C]*)
	T_Ch_T2HP : INT; (*AI charge temperature after high-pressure turbocharger [°C]*)
	T_Ch_T2HP_A : INT; (*AI charge temperature after high-pressure turbocharger bank A [°C]*)
	T_Ch_T2HP_B : INT; (*AI charge temperature after high-pressure turbocharger bank B [°C]*)
	T_OilSkid_Supply : INT; (*AI OilSkid supply temperature*)
	T_OilSkid_Tank : INT; (*AI OilSkid tank temperature*)
	T_PCGAfCo : INT; (*AItemperatureprechambergasaftercooler*)
	T_PCGAfComp_Hi : BOOL; (*DItemperatureprechambergascompressoroutlethigh*)
	T_PCGT : INT; (*AI	Prechambergastemperature*)
	T_PlateHE : INT; (*AIplatetemperatureheatexchanger*)
	T_ThR_Chamber1_1 : INT; (*thermalreactorchambertemperature1_1*)
	T_ThR_Chamber1_2 : INT; (*thermalreactorchambertemperature1_2*)
	T_ThR_Chamber2_1 : INT; (*thermalreactorchambertemperature2_1*)
	T_ThR_Chamber2_2 : INT; (*thermalreactorchambertemperature2_2*)
	T_ThR_ChamberLo : BOOL; (*DIthermalreactorchambertemperaturelow*)
	T_ThR_Comp : INT; (*thermalreactorcompensationtemperature*)
	T_ThR_In : INT; (*thermalreactorinlettemperature*)
	T_ThR_Out : INT; (*thermalreactoroutlettemperature*)
	T_ThR_Swg_Hi : BOOL; (*DIthermalreactorswitchgeartemperaturehigh*)
	ulMMDSerialNumber : ARRAY[0..2] OF UDINT; (*Serial number MMD*)
	UPS_CB_On : BOOL; (*Circuit breaker tripped supply UPS*)
	UPS_Ok : BOOL; (*failureuninterruptedpowersupply*)
	usCAsymDel : ARRAY[0..2] OF UINT; (* delay current asymetrie monitoring *)
	usCNMax : ARRAY[0..2] OF UINT; (* monitoring limit neutral current *)
	usCNMaxDel : ARRAY[0..2] OF UINT; (* delay neutral current monitoring *)
	usCTherm : ARRAY[0..2] OF UINT; (* monitoring limit thermal overload *)
	usFreqDiffMax : ARRAY[0..2] OF UINT; (*maximum frequence difference (positive) [0,02..0,49Hz]*)
	usFreqNenn : ARRAY[0..2] OF UINT; (*nominal frequency [48..62Hz]*)
	usIDyn : ARRAY[0..2] OF UINT; (* dynamic generator current [A] *)
	usImpDO4Min : ARRAY[0..2] OF UINT; (*minimum impulse width of DO4 [0,04..0,5s]*)
	usImpVal : ARRAY[0..2] OF UINT; (* work impulse factor [kW/imp] *)
	usINennGen : ARRAY[0..2] OF UINT; (*nominal current generator [0..65kA]*)
	usIntValue : ARRAY[0..2] OF UINT; (* integrator thermal overload monit. *)
	usMMDModuleID : ARRAY[0..2] OF UINT; (*Module ID MMD*)
	usMMDSynchHWVariant : ARRAY[0..2] OF UINT; (*Hardware variant MMDsynch*)
	usMulIL1L3 : ARRAY[0..2] OF UINT; (* current input multiplikator *)
	usMulUBus : ARRAY[0..2] OF UINT; (*voltage input multiplikator bus*)
	usMulUL1L3 : ARRAY[0..2] OF UINT; (* voltage input multiplikator *)
	usMulUSync1 : ARRAY[0..2] OF UINT; (* voltage input multiplikator synch 1*)
	usMulUSync2 : ARRAY[0..2] OF UINT; (* voltage input multiplikator synch 2*)
	usOFreq : ARRAY[0..2] OF UINT; (* monitoring limit over frequency *)
	usOFreqDel : ARRAY[0..2] OF UINT; (* delay over frequency monitoring *)
	usOVolt : ARRAY[0..2] OF UINT; (* monitoring limit over voltage *)
	usOVoltDel : ARRAY[0..2] OF UINT; (* delay over voltage monitoring *)
	usPhiDiffMax : ARRAY[0..2] OF UINT; (*maximum phase shift [0..60°]*)
	usPhiSync1 : ARRAY[0..2] OF UINT; (*phase shift of sync1*)
	usPsumFiltDel : ARRAY[0..2] OF UINT; (*low pass filter time of power calculation [0-300ms]*)
	usReactDel : ARRAY[0..2] OF UINT; (* delay reactive power monitoring *)
	usShort : ARRAY[0..2] OF UINT; (* monitoring limit short circuit *)
	usShortDel : ARRAY[0..2] OF UINT; (* delay short current monitoring *)
	usSwitchDelDO4 : ARRAY[0..2] OF UINT; (*switching delay of the relay switched with DO4 [40..300ms]*)
	usSyncCfg : ARRAY[0..2] OF UINT; (* sync selector configuration*)
	usUdeadBus : ARRAY[0..2] OF UINT; (*maximum voltage for dead bus detection DO3*)
	usUdeadSync : ARRAY[0..2] OF UINT; (*maximum voltage for sync mode 'dead bus' detection*)
	usUDiffMax : ARRAY[0..2] OF UINT; (*maximum voltage difference [0,1% - 30% usUNennSync]*)
	usUFreq : ARRAY[0..2] OF UINT; (* monitoring limit under frequency *)
	usUFreqDel : ARRAY[0..2] OF UINT; (* delay under frequncy monitoring *)
	usUNennBus : ARRAY[0..2] OF UINT; (*nominal voltage bus [70V..65kV]*)
	usUNennGen : ARRAY[0..2] OF UINT; (*nominal voltage generator [70V..65kV]*)
	usUNennSync : ARRAY[0..2] OF UINT; (*nominal voltage sync1 & sync2 [70V..65kV]*)
	usUVolt : ARRAY[0..2] OF UINT; (* monitoring limit under voltage *)
	usUVolt2 : ARRAY[0..2] OF UINT; (* monitoring limit under voltage *)
	usUVolt2Del : ARRAY[0..2] OF UINT; (* delay under voltage monitoring *)
	usUVoltDel : ARRAY[0..2] OF UINT; (* delay under voltage monitoring *)
	usVAsym : ARRAY[0..2] OF UINT; (* monitoring limit volt. asymetrie *)
	usVAsymDel : ARRAY[0..2] OF UINT; (* last monit. limit. volt. asymetrie *)
	usCAsym : ARRAY[0..2] OF UINT; (* monitoring current asymetry value [p.u.] *)
	usP_ThermOverChar : ARRAY[0..2] OF UINT; (* Thermic overload protection characteristic *)
	usOutput21Cfg : ARRAY[0..2] OF UINT; (* configuration Output 21 - generator mains monitoring functions *)
	U_Adj_Minus : BOOL; (*VoltageadjustmentMinus*)
	U_Adj_Plus : BOOL; (*VoltageadjustmentPlus*)
	U_Avg : ARRAY[0..2] OF INT; (*actualgeneratoraveragevoltage*)
	U_GenC_SetCUST : INT; (*costumiz:scalingvalueforgeneratorvoltageforreactivepowerfromEU*)
	U_GenDiode_Fail : BOOL; (*generatordiodealarm*)
	U_GenOverVolt : BOOL; (*failuregeneratorovervoltageprotection*)
	U_Gen_Contr_Fail : BOOL; (*generatorvoltageregulatorfailure*)
	U_Gen_Dec : BOOL; (*digitalinputforvoltageadjustmentbyMMU(decreasing*)
	U_Gen_Exc : INT; (*actualexcitationvoltagesignal,filteredandscaled*)
	U_Gen_Inc : BOOL; (*digitalinputforvoltageadjustmentbyMMU(increasing*)
	U_Gen_LimHi : ARRAY[0..2] OF BOOL; (*generatorvoltagetoohigh*)
	U_Gen_LimLo : ARRAY[0..2] OF BOOL; (*generatorvoltagetoolow*)
	U_Gen_LimLo2 : ARRAY[0..2] OF BOOL; (*generatorvoltagetoolow2*)
	U_L1L2 : ARRAY[0..2] OF INT; (* generator voltage phase 1_2 [V] *)
	U_L1N : ARRAY[0..2] OF INT; (* generator voltage phase 1_N [V] *)
	U_L2L3 : ARRAY[0..2] OF INT; (* generator voltage phase 2_3 [V] *)
	U_L2N : ARRAY[0..2] OF INT; (* generator voltage phase 2_N [V] *)
	U_L3L1 : ARRAY[0..2] OF INT; (* generator voltage phase 3_1 [V] *)
	U_L3N : ARRAY[0..2] OF INT; (* generator voltage phase 3_N [V] *)
	U_MidPos : BOOL; (*Voltagemiddleposition*)
	U_Minus : BOOL; (*Voltageminus*)
	U_MMD_Asy : ARRAY[0..2] OF BOOL; (*generatorvoltagenegativesequencetoohigh*)
	U_MMD_Synch1 : ARRAY[0..2] OF INT; (*synchronization voltage 1*)
	U_MMD_Synch2 : ARRAY[0..2] OF INT; (*synchronization voltage 2*)
	U_Plus : BOOL; (*Voltageplus*)
	U_StarterBat_Lo : BOOL; (*DIvoltagestarterbatterylow*)
	U_Starter_engage1 : INT; (*Start motor 1 voltage*)
	U_Starter_engage2 : INT; (*Start motor 2 voltage*)
	U_Starter_engage3 : INT; (*Start motor 3 voltage*)
	Vol_GT : INT; (*IF658gasquantity	*)
	WG_Dem : BOOL; (*wastegateposition*)
	WG_A_Dem : BOOL; (*wastegatepositionA*)
	WG_B_Dem : BOOL; (*wastegatepositionB*)
	tT_EO_Pan : HALioAi_Type; (*engine oil temperature oil pan, M.03-TI-002*) (*OldName:AI_t_OilPan; Cycle:5*)
	T_EO_Pan : INT; (*engine oil temperature oil pan, M.03-TI-002*) (*OldName:AI_t_OilPan; Cycle:5*)
	tGenHeat_CB_On : HALioDi_Type; (*Generator heater circuit breaker tripped*) (*Oldname:newPv;Cycle:5;*)
	GenHeat_CB_On : BOOL; (*Generator heater circuit breaker tripped*) (*Oldname:newPv;Cycle:5;*)
	tT_GR : HALioAi_Type; (*AI Gas rail temperature*) (*OldName: AI_GRTP; Cyclic: 2; *)
	T_GR : INT; (*AI Gas rail temperature*) (*OldName: AI_GRTP; Cyclic: 2; *)
	tGV1_line1_Open : HALioDo_Type; (*DO open gas valve 1 line 1 *) (* OldName: DO_GASV1_1_TC1; Cyclic:2; *)
	GV1_line1_Open : BOOL; (*DO open gas valve 1 line 1 *) (* OldName: DO_GASV1_1_TC1; Cyclic:2; *)
	tGV1_line2_Open : HALioDo_Type; (*DO open gas valve 1 line 2 *) (* OldName: DO_GASV1_2_TC1; Cyclic:2; *)
	GV1_line2_Open : BOOL; (*DO open gas valve 1 line 2 *) (* OldName: DO_GASV1_2_TC1; Cyclic:2; *)
	tGV1_line3_Open : HALioDo_Type; (*DO open gas valve 1 line 3*) (* OldName: DO_GASV1_3_TC1; Cyclic:2; *)
	GV1_line3_Open : BOOL; (*DO open gas valve 1 line 3*) (* OldName: DO_GASV1_3_TC1; Cyclic:2; *)
	tGV1_line4_Open : HALioDo_Type; (*DO open gas valve 1 line 4*) (* OldName: DO_GASV1_4_TC1; Cyclic:2; *)
	GV1_line4_Open : BOOL; (*DO open gas valve 1 line 4*) (* OldName: DO_GASV1_4_TC1; Cyclic:2; *)
	tPS_EI_CB_On : HALioDi_Type; (*power supply engine interface panel circuit breaker on*) (*OldName:PS_EI_CB_trip; Cycle:5;*)
	PS_EI_CB_On : BOOL; (*power supply engine interface panel circuit breaker on*) (*OldName:PS_EI_CB_trip; Cycle:5;*)
	tSTT_CB_On : HALioDi_Type; (*control voltage transformer circuit breaker on*) (*OldName:STT_CB_trip; Cycle:5;*)
	STT_CB_On : BOOL; (*control voltage transformer circuit breaker on*) (*OldName:STT_CB_trip; Cycle:5;*)
	tCV_MCP_Low : HALioDi_Type; (*control voltage low - module control panel*) (*OldName:DI_CV_MCP_low; Cycle:5;*)
	CV_MCP_Low : BOOL; (*control voltage low - module control panel*) (*OldName:DI_CV_MCP_low; Cycle:5;*)
	tENGIA_CB_On : HALioDi_Type; (*power supply engine interface panel circuit breaker on*) (*OldName:DI_ENGIA_CB_On; Cycle:5;*)
	ENGIA_CB_On : BOOL; (*power supply engine interface panel circuit breaker on*) (*OldName:DI_ENGIA_CB_On; Cycle:5;*)
	tFastStartReq : HALioDi_Type; (* DI: Fast Start Required *) (* OldName: DI_FastStartReq; Cycle:2; *)
	FastStartReq : BOOL; (* DI: Fast Start Required *) (* OldName: DI_FastStartReq; Cycle:2; *)
	tVeryFastStartReq : HALioDi_Type; (* DI: Very Fast Start Required *) (* OldName: DI_FastStartReq; Cycle:2; *)
	VeryFastStartReq : BOOL; (* DI: Very Fast Start Required *) (* OldName: DI_FastStartReq; Cycle:2; *)
	tU_GenDiode_Trip : HALioDi_Type; (*generator diode trip*) (*OldName:DI_GEN_D_Tr ;Cycle:5*)
	U_GenDiode_Trip : BOOL; (*generator diode trip*) (*OldName:DI_GEN_D_Tr ;Cycle:5*)
	tPr_AirStarter_Tank : HALioAi_Type; (*AI air starter tank pressure [bar] (P.31-PI-001)*)
	Pr_AirStarter_Tank : INT; (*AI air starter tank pressure [bar] (P.31-PI-001)*)
	tPr_AirStarter_Supply : HALioAi_Type; (*AI Air starter supply pressure [bar] (E.31-PI-001)*)
	Pr_AirStarter_Supply : INT; (*AI Air starter supply pressure [bar] (E.31-PI-001)*)
	tCnt_N_AirStarter : HALioAi_INT_Type; (*AI air starter speed [rpm] (E.00-SI-006)*)
	Cnt_N_AirStarter : UINT; (*AI air starter speed [rpm] (E.00-SI-006)*)
	T_MBearing : ARRAY[0..11] OF INT; (*AI Main bearing temperature *) (*  *)
	tT_MBearing : ARRAY[0..11] OF HALioAi_Type; (*AI Main bearing temperature *) (*  *)
	Actuator_Ok_CBV_A : BOOL; (* DI: Actuator okay compressor by pass valve 1A *) (* OldName: DI_F_ACT_TBV_A; Cycle:2; *)
	tActuator_Ok_CBV_A : HALioDi_Type; (* DI: Actuator okay compressor by pass valve 1A *) (* OldName: DI_F_ACT_TBV_A; Cycle:2; *)
	Actuator_Ok_CBV_B : BOOL; (* DI: Actuator okay compressor by pass valve 1B *) (* OldName: DI_F_ACT_TBV_B; Cycle:2; *)
	tActuator_Ok_CBV_B : HALioDi_Type; (* DI: Actuator okay compressor by pass valve 1B *) (* OldName: DI_F_ACT_TBV_B; Cycle:2; *)
	MnsOk_ClosCond_Ok : BOOL; (*closing condition from external facility*) (* OldName: newPV; Cycle:2; *)
	tMnsOk_ClosCond_Ok : HALioDi_Type; (*closing condition from external facility*) (* OldName: newPV; Cycle:2; *)
	P_GenRev_Ext : BOOL; (*Generator reverse power*) (* OldName: newPV; Cycle:2; *)
	tP_GenRev_Ext : HALioDi_Type; (*Generator reverse power*) (* OldName: newPV; Cycle:2; *)
	GenLossExc_Ext : BOOL; (*Generator loss of excitation*) (* OldName: newPV; Cycle:2; *)
	tGenLossExc_Ext : HALioDi_Type; (*Generator loss of excitation*) (* OldName: newPV; Cycle:2; *)
	U_GenAsy_Ext : BOOL; (*Voltage negative sequence*) (* OldName: newPV; Cycle:2; *)
	tU_GenAsy_Ext : HALioDi_Type; (*Voltage negative sequence*) (* OldName: newPV; Cycle:2; *)
	I_GenAsy_Ext : BOOL; (*Current negative sequence*) (* OldName: newPV; Cycle:2; *)
	tI_GenAsy_Ext : HALioDi_Type; (*Current negative sequence*) (* OldName: newPV; Cycle:2; *)
	GenOverExc : BOOL; (*generator overexcitation*) (*OldName:newPV; Cycle:5*)
	tGenOverExc : HALioDi_Type; (*generator overexcitation*) (*OldName:newPV; Cycle:5*)
	GenRotorEarthFault : BOOL; (*rotor earth fault*) (*OldName:newPV; Cycle:5*)
	tGenRotorEarthFault : HALioDi_Type; (*rotor earth fault*) (*OldName:newPV; Cycle:5*)
	Q_GenUnderVoltProt : BOOL; (*reactive power/undervoltage protection (Q-U-protection)*) (*OldName:newPV; Cycle:5*)
	tQ_GenUnderVoltProt : HALioDi_Type; (*reactive power/undervoltage protection (Q-U-protection)*) (*OldName:newPV; Cycle:5*)
	MCB_OpF_Ext : BOOL; (*generator circuit breaker opening failure*) (*OldName:newPV; Cycle:5*)
	tMCB_OpF_Ext : HALioDi_Type; (*generator circuit breaker opening failure*) (*OldName:newPV; Cycle:5*)
	GCB_OpF_Ext : BOOL; (*generator circuit breaker opening failure*) (*OldName:newPV; Cycle:5*)
	tGCB_OpF_Ext : HALioDi_Type; (*generator circuit breaker opening failure*) (*OldName:newPV; Cycle:5*)
	tTempMax_GenCB : HALioDi_Type; (*DI: Temperatur max Generatorschalter*)
	TempMax_GenCB : BOOL; (*DI: Temperatur max Generatorschalter*)
	tCDP_Dem : HALioDo_Type; (*DO: Demand condensor pump*)
	CDP_Dem : BOOL; (*DO: Demand condensor pump*)
	tCDP_Op : HALioDi_Type; (*DI: Failure condensor pump*)
	CDP_Op : BOOL; (*DI: Failure condensor pump*)
	tCtr_CDSu_Set : HALioAo_Type; (*AO: Set point FC condensor pump*)
	Ctr_CDSu_Set : INT; (*AO: Set point FC condensor pump*)
	tT_CD_Su : HALioAi_Type; (*AI: Supply temperature condensor circuit*)
	T_CD_Su : INT; (*AI: Supply temperature condensor circuit*)
	tT_CD_Re : HALioAi_Type; (*AI: Return temperature condensor circuit*)
	T_CD_Re : INT; (*AI: Return temperature condensor circuit*)
	tDemnd_BHV : HALioDi_Type; (*DI: Demand boiler house ventilation*)
	Demnd_BHV : BOOL; (*DI: Demand boiler house ventilation*)
	tBHV_Op : HALioDi_Type; (*DI: Failure boiler house ventilation*)
	BHV_Op : BOOL; (*DI: Failure boiler house ventilation*)
	tBHV_Dem : HALioDo_Type; (*DO: Demand boiler house ventilation*)
	BHV_Dem : BOOL; (*DO: Demand boiler house ventilation*)
	tAuxV_ModIf_ok : HALioDi_Type; (*DI: Auxiliaries voltage module interface OK*)
	AuxV_ModIf_ok : BOOL; (*DI: Auxiliaries voltage module interface OK*)
	tAuxV_Aux_ok : HALioDi_Type; (*DI: Auxiliaries voltage auxiliaries panel OK*)
	AuxV_Aux_ok : BOOL; (*DI: Auxiliaries voltage auxiliaries panel OK*)
	tEmStop_CoolRun : HALioDi_Type; (*DI: Emergency stop with cool down run*)
	EmStop_CoolRun : BOOL; (*DI: Emergency stop with cool down run*)
	tL_DayOilTank_Hi : HALioDi_Type; (*DI: Day oil tank high*)
	L_DayOilTank_Hi : BOOL; (*DI: Day oil tank high*)
	tDayOilTank_Leck : HALioDi_Type; (*DI: Leck day oil tank*)
	DayOilTank_Leck : BOOL; (*DI: Leck day oil tank*)
	tL_DayOilSump_Hi : HALioDi_Type; (*DI: Day tank oil collector pan high*)
	L_DayOilSump_Hi : BOOL; (*DI: Day tank oil collector pan high*)
	tFOP_Op : HALioDi_Type; (*DI: Fresh oil pump operation*)
	FOP_Op : BOOL; (*DI: Fresh oil pump operation*)
	tMCB_COf_GCB_OpF : HALioDo_Type; (*DO: open mcb cause of gcb open failure*)
	MCB_COf_GCB_OpF : BOOL; (*DO: open mcb cause of gcb open failure*)
	tPr_Diff_ExGFilter : HALioAi_Type; (*AI: Differential pressure exhaust gas filter*)
	Pr_Diff_ExGFilter : INT; (*AI: Differential pressure exhaust gas filter*)
	tPr_Diff_ExGCooler : HALioAi_Type; (*AI: Differential pressure exhaust gas cooler*)
	Pr_Diff_ExGCooler : INT; (*AI: Differential pressure exhaust gas cooler*)
	tHWF_Fail : HALioDi_Type; (*DI: Failure heat water flap*)
	HWF_Fail : BOOL; (*DI: Failure heat water flap*)
	tHWF_Dem : HALioDo_Type; (*DO: Demand heat water flap*)
	HWF_Dem : BOOL; (*DO: Demand heat water flap*)
	tT_HW_HC_Re : HALioAi_Type; (*AI: Heating circuit return temperature*)
	T_HW_HC_Re : INT; (*AI: Heating circuit return temperature*)
	tPos_InlLou1 : HALioAi_Type; (*AI: position air inlet louver 1*) (*STM*)
	Pos_InlLou1 : INT; (*AI: position air inlet louver 1*) (*STM*)
	tPos_InlLou2 : HALioAi_Type; (*AI: position air inlet louver 2*) (*STM*)
	Pos_InlLou2 : INT; (*AI: position air inlet louver 2*) (*STM*)
	tPos_OutlLou1 : HALioAi_Type; (*AI: position air outlet louver 1) (*STM*)
	Pos_OutlLou1 : INT; (*AI: position air outlet louver 1*) (*STM*)
	tPos_OutlLou2 : HALioAi_Type; (*AI: position air outlet louver 2*) (*STM*)
	Pos_OutlLou2 : INT; (*AI: position air outlet louver 2*) (*STM*)
	tPos_CircLou1 : HALioAi_Type; (*AI: position air circulation louver 1*) (*STM*)
	Pos_CircLou1 : INT; (*AI: position air circulation louver 1*) (*STM*)
	tPos_CircLou2 : HALioAi_Type; (*AI: position air circulation louver 2*) (*STM*)
	Pos_CircLou2 : INT; (*AI: position air circulation louver 2*) (*STM*)
	tPos_HW_ReValve : HALioAi_Type; (*AI: position heating water return temperature regulation valve*) (*STM*)
	Pos_HW_ReValve : INT; (*AI: position heating water return temperature regulation valve*) (*STM*)
	tPos_HW_EC_ReValve : HALioAi_Type; (*AI: position heating water return temperature after cooler regulation valve*) (*STM*)
	Pos_HW_EC_ReValve : INT; (*AI: position heating water return temperature after cooler regulation valve*) (*STM*)
	tPos_ChC_Valve : HALioAi_Type; (*AI: position charge temperature regulation valve*) (*STM*)
	Pos_ChC_Valve : INT; (*AI: position charge temperature regulation valve*) (*STM*)
	tCtr_InlLou_Set : HALioAo_Type; (*AO: setpoint inlet louver(s)*) (*STM*)
	Ctr_InlLou_Set : INT; (*AO: setpoint inlet louvre(s)*) (*STM*)
	tCtr_OutlLou_RT_Set : HALioAo_Type; (*AO: setpoint outlet louver(s) regarding engine room temperature*) (*STM 2*)
	Ctr_OutlLou_RT_Set : INT; (*AO: setpoint outlet louvre(s) regarding engine room temperature*) (*STM 2*)
	tCtr_OutlLou_RDP_Set : HALioAo_Type; (*AO: setpoint outlet louver(s) regarding engine room differential pressure*) (*STM 2*)
	Ctr_OutlLou_RDP_Set : INT; (*AO: setpoint outlet louver(s) regarding engine room differential pressure*) (*STM 2*)
	tCtr_CircLou_Set : HALioAo_Type; (*AO: setpoint circulation louver(s)*) (*STM*)
	Ctr_CircLou_Set : INT; (*AO: setpoint circulation louver(s)*) (*STM*)
	tPrDiff_ER : HALioAi_Type; (*AI: engine room difference pressure*) (*STM 2*)
	PrDiff_ER : INT; (*AI: engine room difference pressure*) (*STM 2*)
	P_max_LSL : INT; (*AO:  power reduction *)
	tP_max_LSL : HALioAo_Type; (*AO:  power reduction *)
	tPCGT_SafeDevOK : HALioDi_Type; (*DI Gassafety device Prechamber*) (*STM 2*)
	PCGT_SafeDevOK : BOOL; (*DI Gassafety device Prechamber*) (*STM 2*)
	tPCGT_SafeDevice : HALioDo_Type; (*DO Gas safety device Prechamber *) (*STM 2*)
	PCGT_SafeDevice : BOOL; (*DO Gas safety device Prechamber *) (*STM 2*)
	tP_LimitSon_Gh : ARRAY[0..4] OF HALioDo_Type; (*Loadstep feedback*) (* Oldname: new PV; Cycle: 2 *)
	P_LimitSon_Gh : ARRAY[0..4] OF BOOL; (*Loadstep feedback*) (* Oldname: new PV; Cycle: 2 *)
	tPr_HW_Re_LT : HALioAi_Type; (*pressure heat water return low temp.circuit M.07-PI-002*)
	Pr_HW_Re_LT : INT; (*pressure heat water return low temp.circuit M.07-PI-002*)
	tPr_HW_Re_HT : HALioAi_Type; (*pressure heat water return high temp.circuit M.06-PI-002*)
	Pr_HW_Re_HT : INT; (*pressure heat water return high temp.circuit M.06-PI-002*)
	tPr_HW_Re_PreH_ECW : HALioAi_Type; (*pressure heat water return preheating engine cooling water M.04-PI-005*)
	Pr_HW_Re_PreH_ECW : INT; (*pressure heat water return preheating engine cooling water M.04-PI-005*)
	tPr_HW_Re_PreH_EO : HALioAi_Type; (*pressure heat water return preheating engine oil M.03-PI-005*)
	Pr_HW_Re_PreH_EO : INT; (*pressure heat water return preheating engine oil M.03-PI-005*)
	tPr_EO_Mod_Out : HALioAi_Type; (*pressure engine oil module outlet M.03-PI-006*)
	Pr_EO_Mod_Out : INT; (*pressure engine oil module outlet M.03-PI-006*)
	tT_ECW_Mod_In : HALioAi_Type; (*temperature engine cooling water, engine cooling water module inlet M.04-TI-003*)
	T_ECW_Mod_In : INT; (*temperature engine cooling water, engine cooling water module inlet M.04-TI-003*)
	tT_ECW_Mod_Out : HALioAi_Type; (*temperature engine cooling water, engine cooling water module outlet M.04-TI-004*)
	T_ECW_Mod_Out : INT; (*temperature engine cooling water, engine cooling water module outlet M.04-TI-004*)
	tT_EO_Mod_In : HALioAi_Type; (*temperature engine oil, oil module inlet M.03-TI-004*)
	T_EO_Mod_In : INT; (*temperature engine oil, oil module inlet M.03-TI-004*)
	tT_EO_Mod_Out : HALioAi_Type; (*temperature engine oil, oil module outlet M.03-TI-003*)
	T_EO_Mod_Out : INT; (*temperature engine oil, oil module outlet M.03-TI-003*)
	tT_HW_Su_PreH_ECW : HALioAi_Type; (*temperature heat water supply preheating engine cooling water M.04-TI-005*)
	T_HW_Su_PreH_ECW : INT; (*temperature heat water supply preheating engine cooling water M.04-TI-005*)
	tT_HW_Re_PreH_ECW : HALioAi_Type; (*temperature heat water return preheating engine cooling water M.04-TI-006*)
	T_HW_Re_PreH_ECW : INT; (*temperature heat water return preheating engine cooling water M.04-TI-006*)
	tT_HW_Su_PreH_EO : HALioAi_Type; (*temperature heat water supply preheating engine oil M.03-TI-005*)
	T_HW_Su_PreH_EO : INT; (*temperature heat water supply preheating engine oil M.03-TI-005*)
	tT_HW_Re_PreH_EO : HALioAi_Type; (*temperature heat water return preheating engine oil M.03-TI-006*)
	T_HW_Re_PreH_EO : INT; (*temperature heat water return preheating engine oil M.03-TI-006*)
	tActuator_Ok_WG : HALioDi_Type; (* DI: Actuator okay wastegate valve *)
	Actuator_Ok_WG : BOOL; (* DI: Actuator okay wastegate valve *)
	tActuator_Ok_WG_A : HALioDi_Type; (* DI: Actuator okay wastegate valve A *) (* OldName: DI_F_ACT_EGBV_A; Cycle:2; *)
	Actuator_Ok_WG_A : BOOL; (* DI: Actuator okay wastegate valve A *) (* OldName: DI_F_ACT_EGBV_A; Cycle:2; *)
	tActuator_Ok_WG_B : HALioDi_Type; (* DI: Actuator okay wastegate valve B *) (* OldName: DI_F_ACT_EGBV_B; Cycle:2; *)
	Actuator_Ok_WG_B : BOOL; (* DI: Actuator okay wastegate valve B *) (* OldName: DI_F_ACT_EGBV_B; Cycle:2; *)
	tGearPump_Dem : HALioDo_Type; (*gear pump demand*)
	GearPump_Dem : BOOL; (*gear pump demand*)
	F_MMD_BusBar : ARRAY[0..2] OF UINT; (* bus bar frequency multi measure device*)
	tF_MMD_BusBar : ARRAY[0..2] OF HALioAi_Type; (* bus bar actual generator frequency*)
	FreshOilPump_RTC : BOOL; (*fresh oil pump run time exceeded*)
	tFreshOilPump_RTC : HALioDo_Type; (*fresh oil pump run time exceeded*)
	tPr_Ch_P2bFA : HALioAi_Type; (*charge pressure before flame arrester [bar]*) (*OldName: new PV; Cycle: 5;*) (*V04.04.00.00*)
	Pr_Ch_P2bFA : INT; (*charge pressure before flame arrester [bar]*) (*OldName: new PV; Cycle: 5;*) (*V04.04.00.00*)
	tPr_Ch_P2HP : HALioAi_Type; (*charge pressure after high pressure turbocharger [bar]*) (*OldName: new PV; Cycle: 5;*) (*V04.04.00.00*)
	Pr_Ch_P2HP : INT; (*charge pressure after high pressure turbocharger [bar]*) (*OldName: new PV; Cycle: 5;*) (*V04.04.00.00*)
	tPr_Ch_P2HP_A : HALioAi_Type; (*charge pressure after high pressure turbocharger A [bar]*) (*OldName: new PV; Cycle: 5;*) (*V04.04.00.00*)
	Pr_Ch_P2HP_A : INT; (*charge pressure after high pressure turbocharger A [bar]*) (*OldName: new PV; Cycle: 5;*) (*V04.04.00.00*)
	tPr_Ch_P2HP_B : HALioAi_Type; (*charge pressure after high pressure turbocharger B [bar]*) (*OldName: new PV; Cycle: 5;*) (*V04.04.00.00*)
	Pr_Ch_P2HP_B : INT; (*charge pressure after high pressure turbocharger B [bar]*) (*OldName: new PV; Cycle: 5;*) (*V04.04.00.00*)
	tPr_Ch_P2LP : HALioAi_Type; (*charge pressure after low pressure turbocharger [bar]*) (*OldName: new PV; Cycle: 5;*) (*V04.04.00.00*)
	Pr_Ch_P2LP : INT; (*charge pressure after low pressure turbocharger [bar]*) (*OldName: new PV; Cycle: 5;*) (*V04.04.00.00*)
	tPr_Ch_P2LP_A : HALioAi_Type; (*charge pressure after low pressure turbocharger A [bar]*) (*OldName: new PV; Cycle: 5;*) (*V04.04.00.00*)
	Pr_Ch_P2LP_A : INT; (*charge pressure after low pressure turbocharger A [bar]*) (*OldName: new PV; Cycle: 5;*) (*V04.04.00.00*)
	tPr_Ch_P2LP_B : HALioAi_Type; (*charge pressure after low pressure turbocharger B [bar]*) (*OldName: new PV; Cycle: 5;*) (*V04.04.00.00*)
	Pr_Ch_P2LP_B : INT; (*charge pressure after low pressure turbocharger B [bar]*) (*OldName: new PV; Cycle: 5;*) (*V04.04.00.00*)
	tT_ECW_bChC_HT : HALioAi_Type; (*temperature engine cooling water before charge cooler high temp.circ. M.06-TI-014*)
	T_ECW_bChC_HT : INT; (*temperature engine cooling water before charge cooler high temp.circ. M.06-TI-014*)
	tT_ECW_bOilC : HALioAi_Type; (*temperature engine cooling water before oil cooler M.06-TI-020*)
	T_ECW_bOilC : INT; (*temperature engine cooling water before oil cooler M.06-TI-020*)
	tT_ECW_bECWC : HALioAi_Type; (*temperature engine cooling water before engine cooling water cooler M.06-TI-030*)
	T_ECW_bECWC : INT; (*temperature engine cooling water before engine cooling water cooler M.06-TI-030*)
	tCV_GENI_Ok : HALioDi_Type; (*control voltage missing generator interface*)
	CV_GENI_Ok : BOOL; (*control voltage missing generator interface*)
	tCV_ENGIB_Ok : HALioDi_Type; (*control voltage missing engine interface bank B*)
	CV_ENGIB_Ok : BOOL; (*control voltage missing engine interface bank B*)
	tCV_TCMI_Ok : HALioDi_Type; (*control voltage missing turbo charger module interface *)
	CV_TCMI_Ok : BOOL; (*control voltage missing turbo charger module interface *)
	tCV_TCUS_Ok : HALioDi_Type; (*control voltage missing turbo charger unit sensor cabinet *)
	CV_TCUS_Ok : BOOL; (*control voltage missing turbo charger unit sensor cabinet *)
	tCV_JWMI_Ok : HALioDi_Type; (*control voltage missing jacket water module interface *)
	CV_JWMI_Ok : BOOL; (*control voltage missing jacket water module interface *)
	tCV_OILMI_Ok : HALioDi_Type; (*control voltage missing oil module interface *)
	CV_OILMI_Ok : BOOL; (*control voltage missing oil module interface *)
	tCV_M_Ok : HALioDi_Type; (*control voltage missing module interface cabinet*)
	CV_M_Ok : BOOL; (*control voltage missing module interface cabinet*)
	tCV_A_Ok : HALioDi_Type; (*control voltage missing module control cabinet *)
	CV_A_Ok : BOOL; (*control voltage missing module control cabinet *)
	tCV_AUX_Ok : ARRAY[0..5] OF HALioDi_Type; (*control voltage missing auxiliaries control cabinet*)
	CV_AUX_Ok : ARRAY[0..5] OF BOOL; (*control voltage missing auxiliaries control cabinet*)
	tPr_EOaP : HALioAi_Type; (*engine oil pressure after pump M.03-PI-007*)
	Pr_EOaP : INT; (*engine oil pressure after pump M.03-PI-007*)
	tPS_EOaP_HiHi : HALioDi_Type; (*engine oil pressure after pump high safety pressure switch M.03-PS-001*)
	PS_EOaP_HiHi : BOOL; (*engine oil pressure after pump high safety pressure switch M.03-PS-001*)
	tPr_OFUbFilt : HALioAi_Type; (*pressure oil filter unit before filter M.03-PI-011*)
	Pr_OFUbFilt : INT; (*pressure oil filter unit before filter M.03-PI-011*)
	tPr_OFUaFilt : HALioAi_Type; (*pressure oil filter unit after filter M.03-PI-012*)
	Pr_OFUaFilt : INT; (*pressure oil filter unit after filter M.03-PI-012*)
	tOFUP_Centrifuge : HALioDo_Type; (*oil filter unit pump centrifuge M.03-P-006*)
	OFUP_Centrifuge : BOOL; (*oil filter unit pump centrifuge M.03-P-006*)
	tOFUP_Filter : HALioDo_Type; (*oil filter unit pump filter M.03-P-007*)
	OFUP_Filter : BOOL; (*oil filter unit pump filter M.03-P-007*)
	tPr_OFUbCentrifuge : HALioAi_Type; (*pressure oil filter unit before centrifuge M.03-PI-008*)
	Pr_OFUbCentrifuge : INT; (*pressure oil filter unit before centrifuge M.03-PI-008*)
	tOFUP_Centrifuge_CB : HALioDi_Type; (*oil filter unit pump centrifuge M.03-P-006 - circuit breaker*)
	OFUP_Centrifuge_CB : BOOL; (*oil filter unit pump centrifuge M.03-P-006 - circuit breaker*)
	tOFUP_Filter_CB : HALioDi_Type; (*oil filter unit pump filter M.03-P-007 - circuit breaker*)
	OFUP_Filter_CB : BOOL; (*oil filter unit pump filter M.03-P-007 - circuit breaker*)
	tSIFA_BOV : HALioDi_Type; (*Blow-off system supply circuit breaker tripped*)
	SIFA_BOV : BOOL; (*Blow-off system supply circuit breaker tripped*)
	tLockEng_ClosCond : HALioDo_Type; (*lockout engine due to closing conditions*)
	LockEng_ClosCond : BOOL; (*lockout engine due to closing conditions*)
	tQ_AVR_Set_U : HALioAo_Type; (*reactive power setpoint to AVR*)
	Q_AVR_Set_U : INT; (*reactive power setpoint to AVR*)
	tCtr_OutlVE_RT_Set : HALioAo_Type; (*AO: setpoint outlet air ventilation regarding engine room temperature*)
	Ctr_OutlVE_RT_Set : INT; (*AO: setpoint outlet air ventilation regarding engine room temperature*)
	tCtr_OutlVE_RDP_Set : HALioAo_Type; (*AO: setpoint outlet air ventilation regarding engine room differential pressure*)
	Ctr_OutlVE_RDP_Set : INT; (*AO: setpoint outlet air ventilation regarding engine room differential pressure*)
	FireProtFlap1_InlAir_Closed : BOOL; (*fireprotectionflap 1 inlet-air closed*)
	tFireProtFlap1_InlAir_Closed : HALioDi_Type; (*fireprotectionflap 1 inlet-air closed*)
	FireProtFlap2_InlAir_Closed : BOOL; (*fireprotectionflap 2 inlet-air closed*)
	tFireProtFlap2_InlAir_Closed : HALioDi_Type; (*fireprotectionflap 2 inlet-air closed*)
	FireProtFlap1_InlAir_Opened : BOOL; (*fireprotectionflap 1 inlet-air opened*)
	tFireProtFlap1_InlAir_Opened : HALioDi_Type; (*fireprotectionflap 1 inlet-air opened*)
	FireProtFlap2_InlAir_Opened : BOOL; (*fireprotectionflap 2 inlet-air opened*)
	tFireProtFlap2_InlAir_Opened : HALioDi_Type; (*fireprotectionflap 2 inlet-air opened*)
	FireProtFlap1_OutlAir_Closed : BOOL; (*fireprotectionflap 1 outlet-air closed*)
	tFireProtFlap1_OutlAir_Closed : HALioDi_Type; (*fireprotectionflap 1 outlet-air closed*)
	FireProtFlap2_OutlAir_Closed : BOOL; (*fireprotectionflap 2 outlet-air closed*)
	tFireProtFlap2_OutlAir_Closed : HALioDi_Type; (*fireprotectionflap 2 outlet-air closed*)
	FireProtFlap1_OutlAir_Opened : BOOL; (*fireprotectionflap 1 outlet-air opened*)
	tFireProtFlap1_OutlAir_Opened : HALioDi_Type; (*fireprotectionflap 1 outlet-air opened*)
	FireProtFlap2_OutlAir_Opened : BOOL; (*fireprotectionflap 2 outlet-air opened*)
	tFireProtFlap2_OutlAir_Opened : HALioDi_Type; (*fireprotectionflap 2 outlet-air opened*)
	P_DEIE : INT;
	tP_DEIE : HALioAi_Type;
	P_FC_RMC_pos : INT; (*AI: positive margin power for FC*)
	tP_FC_RMC_pos : HALioAi_Type; (*AI: positive margin power for FC*)
	P_FC_RMC_neg : INT; (*AI: negative margin power for FC*)
	tP_FC_RMC_neg : HALioAi_Type; (*AI: negative margin power for FC*)
	P_Set_FC : INT; (*AI: power setpoint FC*)
	tP_Set_FC : HALioAi_Type; (*AI: power setpoint FC*)
	Set_ILF_COn : BOOL; (*DI: set ILF command on*)
	tSet_ILF_COn : HALioDi_Type; (*DI: set ILF command on*)
	Set_ILF_COf : BOOL; (*DI: set ILF command off*)
	tSet_ILF_COf : HALioDi_Type; (*DI: set ILF command off*)
	Set_FC_COn : BOOL; (*DI: set frequency command on*)
	tSet_FC_COn : HALioDi_Type; (*DI: set frequency command on*)
	Set_FC_COf : BOOL; (*DI: set frequency command off*)
	tSet_FC_COf : HALioDi_Type; (*DI: set frequency command off*)
	ILF_SOn : BOOL; (*DO: ILF switched on*)
	tILF_SOn : HALioDo_Type; (*DO: ILF switched on*)
	ILF_SOf : BOOL; (*DO: ILF switched off*)
	tILF_SOf : HALioDo_Type; (*DO: ILF switched off*)
	FC_SOn : BOOL; (*DO: frequency control switched on*)
	tFC_SOn : HALioDo_Type; (*DO: frequency control switched on*)
	FC_SOf : BOOL; (*DO: frequency control switched off*)
	tFC_SOf : HALioDo_Type; (*DO: frequency control switched off*)
	tSet_PU_COn : HALioDi_Type; (*DI: set P(U) command on*)
	Set_PU_COn : BOOL; (*DI: set P(U) command on*)
	tSet_PU_COf : HALioDi_Type; (*DI: set P(U) command on*)
	Set_PU_COf : BOOL; (*DI: set P(U) command off*)
	PU_SOn : BOOL; (*DO: P(U) switched on*)
	tPU_SOn : HALioDo_Type; (*DO: P(U) switched on*)
	PU_SOf : BOOL; (*DO: P(U) switched off*)
	tPU_SOf : HALioDo_Type; (*DO: P(U) switched off*)
	F_Act_FC : INT; (*AO: actual frequency FC*)
	tF_Act_FC : HALioAo_Type; (*AO: actual frequency FC*)
	F_Set_FC : INT; (*AO: nominal frequency set FC*)
	tF_Set_FC : HALioAo_Type; (*AO: nominal frequency set FC*)
	P_Act_FC : INT; (*AO: actual power FC*)
	tP_Act_FC : HALioAo_Type; (*AO: actual power FC*)
	P_PRLCont_FC : INT; (*AO: PRL controller power output FC*)
	tP_PRLCont_FC : HALioAo_Type; (*AO: PRL controller power output FC*)
	Pr_TCO : INT; (*oil pressure before turbocharger*)
	tPr_TCO : HALioAi_Type; (*oil pressure before turbocharger*)
	TCOV_CoClose : BOOL; (*turbo charger oil valve command open*)
	tTCOV_CoClose : HALioDo_Type; (*turbo charger oil valve command open*)
	Pr_PCGT_a_Filt : INT; (*AI	Gaspressureprechambergastrainafterfilter*)
	tPr_PCGT_a_Filt : HALioAi_Type; (*AI	Gaspressureprechambergastrainafterfilter*)
	Dem_Ctr_Mns : BOOL; (*V4.4 Netzbezugsregler 01*)
	tDem_Ctr_Mns : HALioDi_Type; (*V4.4 Netzbezugsregler 01*)
	P_Mns_AnaIn : INT; (*V4.4 Netzbezugsregler 01*)
	tP_Mns_AnaIn : HALioAi_Type; (*V4.4 Netzbezugsregler 01*)
	Ctr_Mns_Anain_Setp_W_ext : INT; (*V4.4 Netzbezugsregler 01*)
	tCtr_Mns_Anain_Setp_W_ext : HALioAi_Type; (*V4.4 Netzbezugsregler 01*)
	T_bScavValve : INT; (*air temperature before exhaust gas scavening valve*)
	tT_bScavValve : HALioAi_Type; (*air temperature before exhaust gas scavening valve*)
	U_StarterBat : INT; (*AI starter battery voltage monitoring*)
	tU_StarterBat : HALioAi_Type; (*AI starter battery voltage monitoring*)
	EOP_BWS : BOOL; (*DI pre-lubrication engine oil pump brush wear signal*)
	tEOP_BWS : HALioDi_Type; (*DI pre-lubrication engine oil pump brush wear signal*)
	EOP_BWS2 : BOOL; (*DI pre-lubrication engine oil pump brush wear signal 2*)
	tEOP_BWS2 : HALioDi_Type; (*DI pre-lubrication engine oil pump brush wear signal 2*)
	ACP_AirER_Dem : BOOL; (*Active Cooling Program - Room Air Ventilation demanded*)
	tACP_AirER_Dem : HALioDo_Type; (*Active Cooling Program - Room Air Ventilation demanded*)
	ACP_HT_Dem : BOOL; (*Active Cooling Program - Heat Water demanded*)
	tACP_HT_Dem : HALioDo_Type; (*Active Cooling Program - Heat Water demanded*)
	T_EGbCat : INT; (*OXIcat Inlet temperature (P.02-TI-046)*) (*OldName: ; Cycle: 5*)
	tT_EGbCat : HALioAi_Type; (*OXIcat Inlet temperature (P.02-TI-046)*) (*OldName: VKAT_WE; Cycle: 5*)
	T_EGaCat : INT; (*OXIcat Outlet temperature (P.02-TI-047)*) (*OldName: ; Cycle: 5*)
	tT_EGaCat : HALioAi_Type; (*OXIcat Outlet temperature (P.02-TI-047)*) (*OldName: ; Cycle: 5*)
	Pr_OXIcat_In : INT; (*OXIcat Inlet pressure (P.02-PI-003)*) (*OldName: newPV; Cycle: 5*)
	tPr_OXIcat_In : HALioAi_Type; (*OXIcat Inlet pressure (P.02-PI-003)*) (*OldName: newPV; Cycle: 5*)
	Pr_OXIcat_Out : INT; (*OXIcat Outlet pressure (P.02-PI-004)*) (*OldName: newPV; Cycle: 5*)
	tPr_OXIcat_Out : HALioAi_Type; (*OXIcat Outlet pressure (P.02-PI-004)*) (*OldName: newPV; Cycle: 5*)
	DI_OMS_Auto : BOOL;
	tDI_OMS_Auto : HALioDi_Type;
	DI_OMS_Man : BOOL;
	tDI_OMS_Man : HALioDi_Type;
	DI_RMS_On : BOOL;
	tDI_RMS_On : HALioDi_Type;
	DI_RMS_Remote : BOOL;
	tDI_RMS_Remote : HALioDi_Type;
	DI_SyOMS_Auto : BOOL;
	tDI_SyOMS_Auto : HALioDi_Type;
	DI_SyOMS_Man : BOOL;
	tDI_SyOMS_Man : HALioDi_Type;
	SPAx_CamDev : BOOL; (* DI: SPAx CAM deviation monitoring *)
	tSPAx_CamDev : HALioDi_Type; (* DI: SPAx CAM deviation monitoring *)
	CO_SCR_EMLine1 : INT; (*SCR Emission measurement line 1 - CO sensor [ppm] (P.02-JI-105)*) (*OldName: tCO_SCR; Cycle: 5;*) (*V04.05.00.00*)
	Flow_SCR_UreaDosingOut : INT; (*SCR Urea flow rate after dosing [l/h] (P.29-FI-001)*) (*OldName: tFlow_Urea; Cycle: 5;*) (*V04.05.00.00*)
	FS_SCR_EMLine1_Lo : BOOL; (*SCR Emission measurement line 1 - flow rate minimum (P.02-FS-101)*) (*OldName: tFS_SampleGas1_Rdy; Cycle: 5;*) (*V04.05.00.00*)
	FS_SCR_EMLine2_Lo : BOOL; (*SCR Emission measurement line 2 - flow rate minimum (P.02-FS-102)*) (*OldName: tFS_SampleGas2_Rdy; Cycle: 5;*) (*V04.05.00.00*)
	Lev_SCR_EMLine1_Hi : BOOL; (*SCR Emission measurement line 1 - moisture maximum (P.02-LS-101)*) (*OldName: tSampleGas_Moisture1; Cycle: 5;*) (*V04.05.00.00*)
	Lev_SCR_EMLine2_Hi : BOOL; (*SCR Emission measurement line 2 - moisture maximum (P.02-LS-102)*) (*OldName: tSampleGas_Moisture2; Cycle: 5;*) (*V04.05.00.00*)
	Lev_SCR_EMAir_Hi : BOOL; (*SCR Emission measurement air line - moisture maximum (P.02-LS-103)*) (*OldName: tSampleGas_Moisture2; Cycle: 5;*) (*V04.14.00.00*)
	Lev_SCR_UreaDosingCabinet_Hi : BOOL; (*SCR Leakage in urea dosing cabinet (P.29-LS-002)*) (*OldName: new PV; Cycle: 5;*) (*V04.05.00.00*)
	Lev_SCR_UreaTank_Lo : BOOL; (*SCR Urea tank level minimum (P.29-LS-001)*) (*OldName: tL_UreaTank; Cycle: 5;*) (*V04.05.00.00*)
	NO2_SCR_EMLine1 : INT; (*SCR Emission measurement line 1 - NO2 sensor [ppm] (P.02-JI-103)*) (*OldName: tNO2_SCR; Cycle: 5;*) (*V04.05.00.00*)
	NO2_SCR_EMLine2 : INT; (*SCR Emission measurement line 2 - NO2 sensor [ppm] (P.02-JI-104)*) (*OldName: new PV; Cycle: 5;*) (*V04.05.00.00*)
	NO_SCR_EMLine1 : INT; (*SCR Emission measurement line 1 - NO sensor [ppm] (P.02-JI-101)*) (*OldName: tNO_SCR; Cycle: 5;*) (*V04.05.00.00*)
	NO_SCR_EMLine2 : INT; (*SCR Emission measurement line 2 - NO sensor [ppm] (P.02-JI-102)*) (*OldName: tNO_Ctrl_SCR; Cycle: 5;*) (*V04.05.00.00*)
	O2_SCR_EMLine1 : INT; (*SCR Emission measurement line 1 - O2 sensor [Vol-%] (P.02-JI-107)*) (*OldName: new PV; Cycle: 5;*) (*V04.05.00.00*)
	Pc_SCR_UreaDosingPump_Set : INT; (*SCR Urea dosing pump - set point [%] (P.29-P-001 / P.29-P-003)*) (*OldName: tFlow_Urea_Set; Cycle: 5;*) (*V04.05.00.00*)
	Pos_SCR_UreaDosingValve2_Set : INT; (*SCR Urea dosing valve redundant - set position [%] (P.29-YCI-002)*) (*OldName: new PV; Cycle: 5;*) (*V04.05.00.00*)
	Pos_SCR_UreaDosingValve_Set : INT; (*SCR Urea dosing valve - set position [%] (P.29-YCI-001)*) (*OldName: new PV; Cycle: 5;*) (*V04.05.00.00*)
	Pr_SCR_CatIn : INT; (*SCR Exhaust pressure CAT inlet [bar] (P.02-PI-101)*) (*OldName: tPr_SCR_In; Cycle: 5;*) (*V04.05.00.00*)
	Pr_SCR_CatOut : INT; (*SCR Exhaust pressure CAT outlet [bar] (P.02-PI-102)*) (*OldName: tPr_SCR_Out; Cycle: 5;*) (*V04.05.00.00*)
	Pr_SCR_ComprAirSupply : INT; (*SCR Compressed air supply pressure urea injection [bar] (P.32-PI-010)*) (*OldName: tPr_AirSupply; Cycle: 5;*) (*V04.05.00.00*)
	Pr_SCR_UreaDosingIn : INT; (*SCR Urea pressure before dosing [bar] (P.29-PI-002)*) (*OldName: new PV; Cycle: 5;*) (*V04.05.00.00*)
	Pr_SCR_UreaDosingOut : INT; (*SCR Urea pressure after dosing [bar] (P.29-PI-001)*) (*OldName: tPr_Urea; Cycle: 5;*) (*V04.05.00.00*)
	SCR_AirCompressor_Dem : BOOL; (*SCR Air compressor demand (P.32-VT-010)*) (*OldName: new PV; Cycle: 5;*) (*V04.05.00.00*)
	SCR_AirCompressor_Rdy : BOOL; (*SCR Air compressor urea injection - power supply ready(= TRUE) (P.32-VT-010)*) (*OldName: new PV; Cycle: 5;*) (*V04.05.00.00*)
	SCR_Aux_Dem : BOOL; (*SCR Auxiliaries demand*) (*OldName: tSCR_AC_PS_Dem; Cycle: 5;*) (*V04.05.00.00*)
	SCR_ComprAirValve_Dem : BOOL; (*SCR Compressed air valve urea injection - demand (P.32-YCS-010)*) (*OldName: tAirCompressed_Dem; Cycle: 5;*) (*V04.05.00.00*)
	SCR_ComprAirValve_Rdy : BOOL; (*SCR Compressed air valve urea injection - power supply ready (P.32-YCS-010)*) (*OldName: tAirCompressed_Rdy; Cycle: 5;*) (*V04.05.00.00*)
	SCR_DosingExt_On : BOOL; (*SCR External dosing on - from customer (TRUE = On)*) (*OldName: new PV; Cycle: 5;*) (*V04.09.00.00*)
	SCR_EMCooler_Rdy : BOOL; (*SCR Emission measurement sample gas cooler - ready (P.02-TS-101)*) (*OldName: tSampleGasCooler_Rdy; Cycle: 5;*) (*V04.05.00.00*)
	SCR_EMPump1_Dem : BOOL; (*SCR Emission measurement line 1 - sample gas pump demand (P.02-P-101)*) (*OldName: tSampleGasPump1_Dem; Cycle: 5;*) (*V04.05.00.00*)
	SCR_EMPump1_Rdy : BOOL; (*SCR Emission measurement line 1 - sample gas pump ready (P.02-P-101)*) (*OldName: tSampleGasPump1_Rdy; Cycle: 5;*) (*V04.05.00.00*)
	SCR_EMPump2_Dem : BOOL; (*SCR Emission measurement line 2 - sample gas pump demand (P.02-P-102)*) (*OldName: tSampleGasPump2_Dem; Cycle: 5;*) (*V04.05.00.00*)
	SCR_EMPump2_Rdy : BOOL; (*SCR Emission measurement line 2 - sample gas pump ready (P.02-P-102)*) (*OldName: tSampleGasPump2_Rdy; Cycle: 5;*) (*V04.05.00.00*)
	SCR_EMValve1_CG_Dem : BOOL; (*SCR Emission measurement line 1 - calibration/sample gas switch valve (P.02-YCS-105)*) (*OldName: tCalGas_Val1_Dem; Cycle: 5;*) (*V04.05.00.00*)
	SCR_EMValve1_SGbCat_Dem : BOOL; (*SCR Emission measurement line 1 - bevor/after CAT sample gas switch valve (P.02-YCS-101)*) (*OldName: tSampleGasVal_Dem; Cycle: 5;*) (*V04.05.00.00*)
	SCR_EMValve1_SGbOxi_Dem : BOOL; (*SCR Emission measurement line 1 - before/after OXI sample gas switch valve (P.02-YCS-102)*) (*OldName: new PV; Cycle: 5;*) (*V04.05.00.00*)
	SCR_EMValve1_SG_Dem : BOOL; (*SCR Emission measurement line 1 - air/sample gas switch valve (P.02-YCS-103)*) (*OldName: tAir_SampleGas_Val1_Dem; Cycle: 5;*) (*V04.05.00.00*)
	SCR_EMValve2_CG_Dem : BOOL; (*SCR Emission measurement line 2 - calibration/sample gas switch valve (P.02-YCS-106)*) (*OldName: tCalGas_Val2_Dem; Cycle: 5;*) (*V04.05.00.00*)
	SCR_EMValve2_SG_Dem : BOOL; (*SCR Emission measurement line 2 - air/sample gas switch valve (P.02-YCS-104)*) (*OldName: tAir_SampleGas_Val2_Dem; Cycle: 5;*) (*V04.05.00.00*)
	SCR_IndicatorLight : BOOL; (*SCR Indicator light demand*) (*OldName: tSCR_Err; Cycle: 5;*) (*V04.05.00.00*)
	SCR_InjectValve_Air : BOOL; (*SCR Urea-air injection valve - air opened (P.29-YCS-001)*) (*OldName: tUreaAirVal_AirOpened; Cycle: 5;*) (*V04.05.00.00*)
	SCR_InjectValve_Opened : BOOL; (*SCR Urea-air injection valve - opened (P.29-YCS-001)*) (*OldName: tUreaAirVal_Opened; Cycle: 5;*) (*V04.05.00.00*)
	SCR_InjectValve_Open_Dem : BOOL; (*SCR Urea-air injection valve - open demand (P.29-YCS-001)*) (*OldName: tUreaAirVal_Open_Dem; Cycle: 5;*) (*V04.05.00.00*)
	SCR_InjectValve_Urea : BOOL; (*SCR Urea-air injection valve - urea opened (P.29-YCS-001)*) (*OldName: tUreaAirVal_UreaOpened; Cycle: 5;*) (*V04.05.00.00*)
	SCR_InjectValve_Urea_Dem : BOOL; (*SCR Urea-air injection valve - urea demand (P.29-YCS-001)*) (*OldName: tUreaAirVal_Dem; Cycle: 5;*) (*V04.05.00.00*)
	SCR_UreaDosingPump2_Dem : BOOL; (*SCR Urea dosing pump redundant - demand (P.29-P-003)*) (*OldName: new PV; Cycle: 5;*) (*V04.05.00.00*)
	SCR_UreaDosingPump2_Rdy : BOOL; (*SCR Urea dosing pump redundant - ready (P.29-P-003)*) (*OldName: new PV; Cycle: 5;*) (*V04.05.00.00*)
	SCR_UreaDosingPump_Dem : BOOL; (*SCR Urea dosing pump - demand (P.29-P-001)*) (*OldName: tUreaPump_Dem; Cycle: 5;*) (*V04.05.00.00*)
	SCR_UreaDosingPump_Rdy : BOOL; (*SCR Urea dosing pump - ready (P.29-P-001)*) (*OldName: tUreaPump_Rdy; Cycle: 5;*) (*V04.05.00.00*)
	SCR_UreaDosingPump_Reset : BOOL; (*SCR Urea dosing pump - FC reset demand (P.29-P-001)*) (*OldName: tUreaPumpFC_Reset; Cycle: 5;*) (*V04.05.00.00*)
	SCR_UreaDosingValve_Dem : BOOL; (*SCR Urea dosing valve - demand (P.29-YCI-001)*) (*OldName: new PV; Cycle: 5;*) (*V04.05.00.00*)
	SCR_UreaDosingValve2_Dem : BOOL; (*SCR Urea dosing valve redundant - demand (P.29-YCI-002)*) (*OldName: new PV; Cycle: 5;*) (*V04.05.00.00*)
	SCR_UreaSupplyPump_Dem : BOOL; (*SCR Urea supply pump demand (P.29-P-002)*) (*OldName: tUreaCircPump_Dem; Cycle: 5;*) (*V04.05.00.00*)
	SCR_UreaSupplyPump_Op : BOOL; (*SCR Urea supply pump operating (P.29-P-002)*) (*OldName: tUreaCircPump_Rdy; Cycle: 5;*) (*V04.05.00.00*)
	SCR_ValvePowerSupply_Ok : BOOL; (*SCR Power supply to the valves on*) (*OldName: tSCR_Val_PS_On; Cycle: 5;*) (*V04.05.00.00*)
	tCO_SCR_EMLine1 : HALioAi_Type; (*SCR Emission measurement line 1 - CO sensor [ppm] (P.02-JI-105)*) (*OldName: tCO_SCR; Cycle: 5;*) (*V04.05.00.00*)
	tFlow_SCR_UreaDosingOut : HALioAi_Type; (*SCR Urea flow rate after dosing [l/h] (P.29-FI-001)*) (*OldName: tFlow_Urea; Cycle: 5;*) (*V04.05.00.00*)
	tFS_SCR_EMLine1_Lo : HALioDi_Type; (*SCR Emission measurement line 1 - flow rate minimum (P.02-FS-101)*) (*OldName: tFS_SampleGas1_Rdy; Cycle: 5;*) (*V04.05.00.00*)
	tFS_SCR_EMLine2_Lo : HALioDi_Type; (*SCR Emission measurement line 2 - flow rate minimum (P.02-FS-102)*) (*OldName: tFS_SampleGas2_Rdy; Cycle: 5;*) (*V04.05.00.00*)
	tLev_SCR_EMLine1_Hi : HALioDi_Type; (*SCR Emission measurement line 1 - moisture maximum (P.02-LS-101)*) (*OldName: tSampleGas_Moisture1; Cycle: 5;*) (*V04.05.00.00*)
	tLev_SCR_EMLine2_Hi : HALioDi_Type; (*SCR Emission measurement line 2 - moisture maximum (P.02-LS-102)*) (*OldName: tSampleGas_Moisture2; Cycle: 5;*) (*V04.05.00.00*)
	tLev_SCR_EMAir_Hi : HALioDi_Type; (*SCR Emission measurement air line - moisture maximum (P.02-LS-103)*) (*OldName: tSampleGas_Moisture2; Cycle: 5;*) (*V04.14.00.00*)
	tLev_SCR_UreaDosingCabinet_Hi : HALioDi_Type; (*SCR Leakage in urea dosing cabinet (P.29-LS-002)*) (*OldName: new PV; Cycle: 5;*) (*V04.05.00.00*)
	tLev_SCR_UreaTank_Lo : HALioDi_Type; (*SCR Urea tank level minimum (P.29-LS-001)*) (*OldName: tL_UreaTank; Cycle: 5;*) (*V04.05.00.00*)
	tNO2_SCR_EMLine1 : HALioAi_Type; (*SCR Emission measurement line 1 - NO2 sensor [ppm] (P.02-JI-103)*) (*OldName: tNO2_SCR; Cycle: 5;*) (*V04.05.00.00*)
	tNO2_SCR_EMLine2 : HALioAi_Type; (*SCR Emission measurement line 2 - NO2 sensor [ppm] (P.02-JI-104)*) (*OldName: new PV; Cycle: 5;*) (*V04.05.00.00*)
	tNO_SCR_EMLine1 : HALioAi_Type; (*SCR Emission measurement line 1 - NO sensor [ppm] (P.02-JI-101)*) (*OldName: tNO_SCR; Cycle: 5;*) (*V04.05.00.00*)
	tNO_SCR_EMLine2 : HALioAi_Type; (*SCR Emission measurement line 2 - NO sensor [ppm] (P.02-JI-102)*) (*OldName: tNO_Ctrl_SCR; Cycle: 5;*) (*V04.05.00.00*)
	tO2_SCR_EMLine1 : HALioAi_Type; (*SCR Emission measurement line 1 - O2 sensor [Vol-%] (P.02-JI-107)*) (*OldName: new PV; Cycle: 5;*) (*V04.05.00.00*)
	tPc_SCR_UreaDosingPump_Set : HALioAo_Type; (*SCR Urea dosing pump - set point [%] (P.29-P-001 / P.29-P-003)*) (*OldName: tFlow_Urea_Set; Cycle: 5;*) (*V04.05.00.00*)
	tPos_SCR_UreaDosingValve2_Set : HALioAo_Type; (*SCR Urea dosing valve redundant - set position [%] (P.29-YCI-002)*) (*OldName: new PV; Cycle: 5;*) (*V04.05.00.00*)
	tPos_SCR_UreaDosingValve_Set : HALioAo_Type; (*SCR Urea dosing valve - set position [%] (P.29-YCI-001)*) (*OldName: new PV; Cycle: 5;*) (*V04.05.00.00*)
	tPr_SCR_CatIn : HALioAi_Type; (*SCR Exhaust pressure CAT inlet [bar] (P.02-PI-101)*) (*OldName: tPr_SCR_In; Cycle: 5;*) (*V04.05.00.00*)
	tPr_SCR_CatOut : HALioAi_Type; (*SCR Exhaust pressure CAT outlet [bar] (P.02-PI-102)*) (*OldName: tPr_SCR_Out; Cycle: 5;*) (*V04.05.00.00*)
	tPr_SCR_ComprAirSupply : HALioAi_Type; (*SCR Compressed air supply pressure urea injection [bar] (P.32-PI-010)*) (*OldName: tPr_AirSupply; Cycle: 5;*) (*V04.05.00.00*)
	tPr_SCR_UreaDosingIn : HALioAi_Type; (*SCR Urea pressure before dosing [bar] (P.29-PI-002)*) (*OldName: new PV; Cycle: 5;*) (*V04.05.00.00*)
	tPr_SCR_UreaDosingOut : HALioAi_Type; (*SCR Urea pressure after dosing [bar] (P.29-PI-001)*) (*OldName: tPr_Urea; Cycle: 5;*) (*V04.05.00.00*)
	tSCR_AirCompressor_Dem : HALioDo_Type; (*SCR Air compressor demand (P.32-VT-010)*) (*OldName: new PV; Cycle: 5;*) (*V04.05.00.00*)
	tSCR_AirCompressor_Rdy : HALioDi_Type; (*SCR Air compressor urea injection - power supply ready(= TRUE) (P.32-VT-010)*) (*OldName: new PV; Cycle: 5;*) (*V04.05.00.00*)
	tSCR_Aux_Dem : HALioDo_Type; (*SCR Auxiliaries demand*) (*OldName: tSCR_AC_PS_Dem; Cycle: 5;*) (*V04.05.00.00*)
	tSCR_ComprAirValve_Dem : HALioDo_Type; (*SCR Compressed air valve urea injection - demand (P.32-YCS-010)*) (*OldName: tAirCompressed_Dem; Cycle: 5;*) (*V04.05.00.00*)
	tSCR_ComprAirValve_Rdy : HALioDi_Type; (*SCR Compressed air valve urea injection - power supply ready (P.32-YCS-010)*) (*OldName: tAirCompressed_Rdy; Cycle: 5;*) (*V04.05.00.00*)
	tSCR_DosingExt_On : HALioDi_Type; (*SCR External dosing on - from customer (TRUE = On)*) (*OldName: new PV; Cycle: 5;*) (*V04.09.00.00*)
	tSCR_EMCooler_Rdy : HALioDi_Type; (*SCR Emission measurement sample gas cooler - ready (P.02-TS-101)*) (*OldName: tSampleGasCooler_Rdy; Cycle: 5;*) (*V04.05.00.00*)
	tSCR_EMPump1_Dem : HALioDo_Type; (*SCR Emission measurement line 1 - sample gas pump demand (P.02-P-101)*) (*OldName: tSampleGasPump1_Dem; Cycle: 5;*) (*V04.05.00.00*)
	tSCR_EMPump1_Rdy : HALioDi_Type; (*SCR Emission measurement line 1 - sample gas pump ready (P.02-P-101)*) (*OldName: tSampleGasPump1_Rdy; Cycle: 5;*) (*V04.05.00.00*)
	tSCR_EMPump2_Dem : HALioDo_Type; (*SCR Emission measurement line 2 - sample gas pump demand (P.02-P-102)*) (*OldName: tSampleGasPump2_Dem; Cycle: 5;*) (*V04.05.00.00*)
	tSCR_EMPump2_Rdy : HALioDi_Type; (*SCR Emission measurement line 2 - sample gas pump ready (P.02-P-102)*) (*OldName: tSampleGasPump2_Rdy; Cycle: 5;*) (*V04.05.00.00*)
	tSCR_EMValve1_CG_Dem : HALioDo_Type; (*SCR Emission measurement line 1 - calibration/sample gas switch valve (P.02-YCS-105)*) (*OldName: tCalGas_Val1_Dem; Cycle: 5;*) (*V04.05.00.00*)
	tSCR_EMValve1_SGbCat_Dem : HALioDo_Type; (*SCR Emission measurement line 1 - bevor/after CAT sample gas switch valve (P.02-YCS-101)*) (*OldName: tSampleGasVal_Dem; Cycle: 5;*) (*V04.05.00.00*)
	tSCR_EMValve1_SGbOxi_Dem : HALioDo_Type; (*SCR Emission measurement line 1 - before/after OXI sample gas switch valve (P.02-YCS-102)*) (*OldName: new PV; Cycle: 5;*) (*V04.05.00.00*)
	tSCR_EMValve1_SG_Dem : HALioDo_Type; (*SCR Emission measurement line 1 - air/sample gas switch valve (P.02-YCS-103)*) (*OldName: tAir_SampleGas_Val1_Dem; Cycle: 5;*) (*V04.05.00.00*)
	tSCR_EMValve2_CG_Dem : HALioDo_Type; (*SCR Emission measurement line 2 - calibration/sample gas switch valve (P.02-YCS-106)*) (*OldName: tCalGas_Val2_Dem; Cycle: 5;*) (*V04.05.00.00*)
	tSCR_EMValve2_SG_Dem : HALioDo_Type; (*SCR Emission measurement line 2 - air/sample gas switch valve (P.02-YCS-104)*) (*OldName: tAir_SampleGas_Val2_Dem; Cycle: 5;*) (*V04.05.00.00*)
	tSCR_IndicatorLight : HALioDo_Type; (*SCR Indicator light demand*) (*OldName: tSCR_Err; Cycle: 5;*) (*V04.05.00.00*)
	tSCR_InjectValve_Air : HALioDi_Type; (*SCR Urea-air injection valve - air opened (P.29-YCS-001)*) (*OldName: tUreaAirVal_AirOpened; Cycle: 5;*) (*V04.05.00.00*)
	tSCR_InjectValve_Opened : HALioDi_Type; (*SCR Urea-air injection valve - opened (P.29-YCS-001)*) (*OldName: tUreaAirVal_Opened; Cycle: 5;*) (*V04.05.00.00*)
	tSCR_InjectValve_Open_Dem : HALioDo_Type; (*SCR Urea-air injection valve - open demand (P.29-YCS-001)*) (*OldName: tUreaAirVal_Open_Dem; Cycle: 5;*) (*V04.05.00.00*)
	tSCR_InjectValve_Urea : HALioDi_Type; (*SCR Urea-air injection valve - urea opened (P.29-YCS-001)*) (*OldName: tUreaAirVal_UreaOpened; Cycle: 5;*) (*V04.05.00.00*)
	tSCR_InjectValve_Urea_Dem : HALioDo_Type; (*SCR Urea-air injection valve - urea demand (P.29-YCS-001)*) (*OldName: tUreaAirVal_Dem; Cycle: 5;*) (*V04.05.00.00*)
	tSCR_UreaDosingPump2_Dem : HALioDo_Type; (*SCR Urea dosing pump redundant - demand (P.29-P-003)*) (*OldName: new PV; Cycle: 5;*) (*V04.05.00.00*)
	tSCR_UreaDosingPump2_Rdy : HALioDi_Type; (*SCR Urea dosing pump redundant - ready (P.29-P-003)*) (*OldName: new PV; Cycle: 5;*) (*V04.05.00.00*)
	tSCR_UreaDosingPump_Dem : HALioDo_Type; (*SCR Urea dosing pump - demand (P.29-P-001)*) (*OldName: tUreaPump_Dem; Cycle: 5;*) (*V04.05.00.00*)
	tSCR_UreaDosingPump_Rdy : HALioDi_Type; (*SCR Urea dosing pump - ready (P.29-P-001)*) (*OldName: tUreaPump_Rdy; Cycle: 5;*) (*V04.05.00.00*)
	tSCR_UreaDosingPump_Reset : HALioDo_Type; (*SCR Urea dosing pump - FC reset demand (P.29-P-001)*) (*OldName: tUreaPumpFC_Reset; Cycle: 5;*) (*V04.05.00.00*)
	tSCR_UreaDosingValve_Dem : HALioDo_Type; (*SCR Urea dosing valve - demand (P.29-YCI-001)*) (*OldName: new PV; Cycle: 5;*) (*V04.05.00.00*)
	tSCR_UreaDosingValve2_Dem : HALioDo_Type; (*SCR Urea dosing valve redundant - demand (P.29-YCI-002)*) (*OldName: new PV; Cycle: 5;*) (*V04.05.00.00*)
	tSCR_UreaSupplyPump_Dem : HALioDo_Type; (*SCR Urea supply pump demand (P.29-P-002)*) (*OldName: tUreaCircPump_Dem; Cycle: 5;*) (*V04.05.00.00*)
	tSCR_UreaSupplyPump_Op : HALioDi_Type; (*SCR Urea supply pump operating (P.29-P-002)*) (*OldName: tUreaCircPump_Rdy; Cycle: 5;*) (*V04.05.00.00*)
	tSCR_ValvePowerSupply_Ok : HALioDi_Type; (*SCR Power supply to the valves on*) (*OldName: tSCR_Val_PS_On; Cycle: 5;*) (*V04.05.00.00*)
	tT_SCR_CatIn : HALioAi_Type; (*SCR exhaust temperature CAT inlet [°C] (P.02-TI-101)*) (*OldName: tT_SCR_In; Cycle: 5;*) (*V04.05.00.00*)
	tT_SCR_CatOut : HALioAi_Type; (*SCR exhaust temperature CAT outlet [°C] (P.02-TI-102)*) (*OldName: tT_SCR_Out; Cycle: 5;*) (*V04.05.00.00*)
	T_SCR_CatIn : INT; (*SCR exhaust temperature CAT inlet [°C] (P.02-TI-101)*) (*OldName: tT_SCR_In; Cycle: 5;*) (*V04.05.00.00*)
	T_SCR_CatOut : INT; (*SCR exhaust temperature CAT outlet [°C] (P.02-TI-102)*) (*OldName: tT_SCR_Out; Cycle: 5;*) (*V04.05.00.00*)
	AfMnsF_ClosCond_Ok : BOOL; (*closing condition from external facility after mains failure*) (* OldName: newPV; Cycle:2; *)
	tAfMnsF_ClosCond_Ok : HALioDi_Type; (*closing condition from external facility after mains failure*) (* OldName: newPV; Cycle:2; *)
	MnsOk_ClosCond_Skip : BOOL; (*skip closing condition from external facility*) (* OldName: newPV; Cycle:2; *)
	tMnsOk_ClosCond_Skip : HALioDi_Type; (*skip closing condition from external facility*) (* OldName: newPV; Cycle:2; *)
	AfMnsF_ClosCond_Skip : BOOL; (*skip closing condition from external facility after mains failure*) (* OldName: newPV; Cycle:2; *)
	tAfMnsF_ClosCond_Skip : HALioDi_Type; (*skip closing condition from external facility after mains failure*) (* OldName: newPV; Cycle:2; *)
	AfMnsF_LockEng_ClosCond : BOOL; (*lockout engine due to closing conditions after mains failure*) (* OldName: newPV; Cycle:2; *)
	tAfMnsF_LockEng_ClosCond : HALioDo_Type; (*DO lockout engine due to closing conditions after mains failure*) (* OldName: newPV; Cycle:2; *)
	ClosCond : BOOL; (*DO closing condition ok from external facility*) (* OldName: newPV; Cycle:2; *)
	tClosCond : HALioDo_Type; (*DO closing condition ok from external facility*) (* OldName: newPV; Cycle:2; *)
	AfMnsF_ClosCond : BOOL; (*DO closing condition ok from external facility after mains failure*) (* OldName: newPV; Cycle:2; *)
	tAfMnsF_ClosCond : HALioDo_Type; (*DO closing condition ok from external facility after mains failure*) (* OldName: newPV; Cycle:2; *)
	ProtectionTest : ARRAY[0..3] OF BOOL; (*DO protection test custom*) (* OldName: newPV; Cycle:2; *)
	tProtectionTest : ARRAY[0..3] OF HALioDo_Type; (*DO protection test custom*) (* OldName: newPV; Cycle:2; *)
	U_Bus_L1_2 : ARRAY[0..2] OF INT; (* bus bar voltage phase 1_2 [V] *)
	tU_Bus_L1_2 : ARRAY[0..2] OF HALioAi_Type; (* bus bar voltage phase 1_2 [V] *)
	U_Bus_L2_3 : ARRAY[0..2] OF INT; (* bus bar voltage phase 2_3 [V] *)
	tU_Bus_L2_3 : ARRAY[0..2] OF HALioAi_Type; (* bus bar voltage phase 2_3 [V] *)
	U_Bus_L3_1 : ARRAY[0..2] OF INT; (* bus bar voltage phase 3_1 [V] *)
	tU_Bus_L3_1 : ARRAY[0..2] OF HALioAi_Type; (* bus bar voltage phase 3_1 [V] *)
	U_Bus_L1N : ARRAY[0..2] OF INT; (* bus bar voltage phase 1 [V] *)
	tU_Bus_L1N : ARRAY[0..2] OF HALioAi_Type; (* bus bar voltage phase 1 [V] *)
	U_Bus_L2N : ARRAY[0..2] OF INT; (* bus bar voltage phase 2 [V] *)
	tU_Bus_L2N : ARRAY[0..2] OF HALioAi_Type; (* bus bar voltage phase 2 [V] *)
	U_Bus_L3N : ARRAY[0..2] OF INT; (* bus bar voltage phase 3 [V] *)
	tU_Bus_L3N : ARRAY[0..2] OF HALioAi_Type; (* bus bar voltage phase 3 [V] *)
	tReady4FastStart : HALioDo_Type; (* Engine ready for fast start *)
	Ready4FastStart : BOOL; (* DO: Engine ready for fast start *)
	tReady4VeryFastStart : HALioDo_Type; (* Engine ready for very fast start *)
	Ready4VeryFastStart : BOOL; (* DO: Engine ready for very fast start *)
	InAirER_Lou1Closed : BOOL; (*DIintakeairengineroomlouver1Closed*)
	InAirER_Lou2Closed : BOOL; (*DIintakeairengineroomlouver2Closed*)
	tInAirER_Lou1Closed : HALioDi_Type; (*DIintakeairengineroomlouver1Closed*)
	tInAirER_Lou2Closed : HALioDi_Type; (*DIintakeairengineroomlouver2Closed*)
	OutAirER_LouClosed : BOOL; (*DIoutletairengineroomlouverClosed*)
	tOutAirER_LouClosed : HALioDi_Type; (*DIoutletairengineroomlouverClosed*)
	ChC2_DemPump : BOOL; (*DO charge cooler 2 demand pump*)
	tChC2_DemPump : HALioDo_Type; (*DO charge cooler 2 demand pump*)
	ChC2_DemFan1 : BOOL; (*DO charge cooler 2 demand fan 1*)
	ChC2_DemFan2 : BOOL; (*DO charge cooler 2 demand fan 2*)
	ChC2_DemFan3 : BOOL; (*DO charge cooler 2 demand fan 3*)
	ChC2_DemFan4 : BOOL; (*DO charge cooler 2 demand fan 4*)
	ChC2_DemFan5 : BOOL; (*DO charge cooler 2 demand fan 5*)
	ChC2_DemFan6 : BOOL; (*DO charge cooler 2 demand fan 6*)
	ChC2_DemFan7 : BOOL; (*DO charge cooler 2 demand fan 7*)
	ChC2_DemFan8 : BOOL; (*DO charge cooler 2 demand fan 8*)
	ChC2_DemFan9 : BOOL; (*DO charge cooler 2 demand fan 9*)
	ChC2_DemFan10 : BOOL; (*DO charge cooler 2 demand fan 10*)
	ChC2_DemFan11 : BOOL; (*DO charge cooler 2 demand fan 11*)
	ChC2_DemFan12 : BOOL; (*DO charge cooler 2 demand fan 12*)
	ChC2_DemFan13 : BOOL; (*DO charge cooler 2 demand fan 13*)
	ChC2_DemFan14 : BOOL; (*DO charge cooler 2 demand fan 14*)
	ChC2_DemFan15 : BOOL; (*DO charge cooler 2 demand fan 15*)
	ChC2_DemFan16 : BOOL; (*DO charge cooler 2 demand fan 16*)
	tChC2_DemFan1 : HALioDo_Type; (*DO charge cooler 2 demand fan 1*)
	tChC2_DemFan2 : HALioDo_Type; (*DO charge cooler 2 demand fan 2*)
	tChC2_DemFan3 : HALioDo_Type; (*DO charge cooler 2 demand fan 3*)
	tChC2_DemFan4 : HALioDo_Type; (*DO charge cooler 2 demand fan 4*)
	tChC2_DemFan5 : HALioDo_Type; (*DO charge cooler 2 demand fan 5*)
	tChC2_DemFan6 : HALioDo_Type; (*DO charge cooler 2 demand fan 6*)
	tChC2_DemFan7 : HALioDo_Type; (*DO charge cooler 2 demand fan 7*)
	tChC2_DemFan8 : HALioDo_Type; (*DO charge cooler 2 demand fan 8*)
	tChC2_DemFan9 : HALioDo_Type; (*DO charge cooler 2 demand fan 9*)
	tChC2_DemFan10 : HALioDo_Type; (*DO charge cooler 2 demand fan 10*)
	tChC2_DemFan11 : HALioDo_Type; (*DO charge cooler 2 demand fan 11*)
	tChC2_DemFan12 : HALioDo_Type; (*DO charge cooler 2 demand fan 12*)
	tChC2_DemFan13 : HALioDo_Type; (*DO charge cooler 2 demand fan 13*)
	tChC2_DemFan14 : HALioDo_Type; (*DO charge cooler 2 demand fan 14*)
	tChC2_DemFan15 : HALioDo_Type; (*DO charge cooler 2 demand fan 15*)
	tChC2_DemFan16 : HALioDo_Type; (*DO charge cooler 2 demand fan 16*)
	Pos_ChC2_Valve : INT; (*AI: Position temperature-regulation-valve 2nd LT charge cooler circuit (T1-HP) (P.07-YTC-007)*)
	tPos_ChC2_Valve : HALioAi_Type; (*AI: Position temperature-regulation-valve 2nd LT charge cooler circuit (T1-HP) (P.07-YTC-007)*)
	Ctr_ChC2_Valve_Set : INT; (*AO: Control temperature-regulation-valve 2nd LT charge cooler circuit (T1-HP) (P.07-YTC-007)*)
	tCtr_ChC2_Valve_Set : HALioAo_Type; (*AO: Control temperature-regulation-valve 2nd LT charge cooler circuit (T1-HP) (P.07-YTC-007)*)
	Pr_ChC2_Lo : BOOL; (*DI charge cooler 2 water pressure low (P.07-PS-101)*)
	tPr_ChC2_Lo : HALioDi_Type; (*DI charge cooler 2 water pressure low (P.07-PS-101)*)
	ChC2_FanRdy : BOOL; (*DI charge cooler 2 fan ready*)
	tChC2_FanRdy : HALioDi_Type; (*DI charge cooler 2 fan ready*)
	ChC2_Failure : BOOL; (*DI charge cooler 2 failure*)
	tChC2_Failure : HALioDi_Type; (*DI charge cooler 2 failure*)
	CC2WP_Op : BOOL; (*DI charge cooler 2 water pump operating (P.07-M-007)*)
	tCC2WP_Op : HALioDi_Type; (*DI charge cooler 2 water pump operating (P.07-M-007)*)
	T_ChC2_Re_LT : INT; (*AI return water temperature 2nd LT charge cooler circuit (T1-HP) [°C] (P.07-TI-006)*)
	tT_ChC2_Re_LT : HALioAi_Type; (*AI return water temperature 2nd LT charge cooler circuit (T1-HP) [°C] (P.07-TI-006)*)
	T_ChC2_Su_LT : INT; (*AI supply water temperature 2nd LT charge cooler circuit (T1-HP) [°C] (P.07-TI-004)*)
	tT_ChC2_Su_LT : HALioAi_Type; (*AI supply water temperature 2nd LT charge cooler circuit (T1-HP) [°C] (P.07-TI-004)*)
	T_ChC2W_Hi : BOOL; (*DI charge cooler 2 water temperature high*)
	tT_ChC2W_Hi : HALioDi_Type; (*DI charge cooler 2 water temperature high*)
	ChC2_Heating : BOOL; (*DO Demand charge cooler 2 pre heating*)
	tChC2_Heating : HALioDo_Type; (*DO Demand charge cooler 2 pre heating*)
	MidVoltCB_Failure : BOOL; (*mid voltage CB failure*)
	tMidVoltCB_Failure : HALioDi_Type; (*mid voltage CB failure*)
	P_Red_EU_Norm : INT; (* AO Power reduction from EU (feedback) *)
	tP_Red_EU_Norm : HALioAo_Type; (* AO Power reduction from EU (feedback) *)
	P_Avail_Norm : INT; (* AO Available power *)
	tP_Avail_Norm : HALioAo_Type; (* AO Available power *)
	OpMode_NetP : BOOL; (* DO Operating mode is net parallel *)
	tOpMode_NetP : HALioDo_Type; (* DO Operating mode is net parallel *)
	OpMode_Island : BOOL; (* DO Operating mode is island *)
	tOpMode_Island : HALioDo_Type; (* DO Operating mode is island *)
	OpMode_Idle : BOOL; (* DO Operating mode is idle *)
	tOpMode_Idle : HALioDo_Type; (* DO Operating mode is idle *)
	tHA2CU : HALIO2CUSTOM_Struct; (* Data exchange structure to Custom *)
	tHA2GR : HALIO2GRID_Struct; (* Data exchange structure to Grid *)
	Set_LFSMO_DB_COn : BOOL; (*DI:request LFSMO Deadband from EU-on(activate*)
	tSet_LFSMO_DB_COn : HALioDi_Type; (*DI:request LFSMO Deadband from EU-on(activate*)
	Set_LFSMO_DB_COf : BOOL; (*DI:request LFSMO Deadband from EU-off(deactivate*)
	tSet_LFSMO_DB_COf : HALioDi_Type; (*DI:request LFSMO Deadband from EU-off(deactivate*)
	F_LFSMO_DB : INT; (*AI:LFSMO Deadband reference from EU [Hz]*)
	tF_LFSMO_DB : HALioAi_Type; (*AI:LFSMO Deadband reference from EU [Hz]*)
	Set_LFSMU_DB_COn : BOOL; (*DI:request LFSMU Deadband from EU-on(activate*)
	tSet_LFSMU_DB_COn : HALioDi_Type; (*DI:request LFSMU Deadband from EU-on(activate*)
	Set_LFSMU_DB_COf : BOOL; (*DI:request LFSMU Deadband from EU-off(deactivate*)
	tSet_LFSMU_DB_COf : HALioDi_Type; (*DI:request LFSM Deadband from EU-off(deactivate*)
	F_LFSMU_DB : INT; (*AI:LFSMU Deadband reference from EU [Hz]*)
	tF_LFSMU_DB : HALioAi_Type; (*AI:LFSMU Deadband reference from EU [Hz]*)
	Set_LFSMO_Droop_COn : BOOL; (*DI:request LFSMO Droop from EU-on(activate*)
	tSet_LFSMO_Droop_COn : HALioDi_Type; (*DI:request LFSMO Droop from EU-on(activate*)
	Set_LFSMO_Droop_COf : BOOL; (*DI:request LFSMO Droop from EU-off(deactivate*)
	tSet_LFSMO_Droop_COf : HALioDi_Type; (*DI:request LFSM Droop from EU-off(deactivate*)
	F_LFSMO_Droop : INT; (*AI:LFSMO Droop reference from EU [Hz]*)
	tF_LFSMO_Droop : HALioAi_Type; (*AI:LFSMO Droop reference from EU [Hz]*)
	Set_LFSMU_Droop_COn : BOOL; (*DI:request LFSMU Droop from EU-on(activate*)
	tSet_LFSMU_Droop_COn : HALioDi_Type; (*DI:request LFSMU Droop from EU-on(activate*)
	Set_LFSMU_Droop_COf : BOOL; (*DI:request LFSMU Droop from EU-off(deactivate*)
	tSet_LFSMU_Droop_COf : HALioDi_Type; (*DI:request LFSMU Droop from EU-off(deactivate*)
	F_LFSMU_Droop : INT; (*AI:LFSMU Droop reference from EU [Hz]*)
	tF_LFSMU_Droop : HALioAi_Type; (*AI:LFSMU Droop reference from EU [Hz]*)
	Set_FSMU_Droop_COn : BOOL; (*DI:request FSMU Droop from EU-on(activate*)
	tSet_FSMU_Droop_COn : HALioDi_Type; (*DI:request FSMU Droop from EU-on(activate*)
	Set_FSMU_Droop_COf : BOOL; (*DI:request FSMU Droop from EU-off(deactivate*)
	tSet_FSMU_Droop_COf : HALioDi_Type; (*DI:request FSMU Droop from EU-off(deactivate*)
	F_FSMU_Droop : INT; (*AI:FSMU Droop reference from EU [Hz]*)
	tF_FSMU_Droop : HALioAi_Type; (*AI:FSMU Droop reference from EU [Hz]*)
	Set_FSMO_Droop_COn : BOOL; (*DI:request FSMO Droop from EU-on(activate*)
	tSet_FSMO_Droop_COn : HALioDi_Type; (*DI:request FSMO Droop from EU-on(activate*)
	Set_FSMO_Droop_COf : BOOL; (*DI:request FSMO Droop from EU-off(deactivate*)
	tSet_FSMO_Droop_COf : HALioDi_Type; (*DI:request FSMO Droop from EU-off(deactivate*)
	F_FSMO_Droop : INT; (*AI:FSMO Droop reference from EU [Hz]*)
	tF_FSMO_Droop : HALioAi_Type; (*AI:FSMO Droop reference from EU [Hz]*)
	Set_FSMU_DB_COn : BOOL; (*DI:request FSMU Deadband from EU-on(activate*)
	tSet_FSMU_DB_COn : HALioDi_Type; (*DI:request FSMU Deadband from EU-on(activate*)
	Set_FSMU_DB_COf : BOOL; (*DI:request FSMU Deadband from EU-off(deactivate*)
	tSet_FSMU_DB_COf : HALioDi_Type; (*DI:request FSMU Deadband from EU-off(deactivate*)
	F_FSMU_DB : INT; (*AI:FSMU Deadband reference from EU [Hz]*)
	tF_FSMU_DB : HALioAi_Type; (*AI:FSMU Deadband reference from EU [Hz]*)
	Set_FSMO_DB_COn : BOOL; (*DI:request FSMO Deadband from EU-on(activate*)
	tSet_FSMO_DB_COn : HALioDi_Type; (*DI:request FSMO Deadband from EU-on(activate*)
	Set_FSMO_DB_COf : BOOL; (*DI:request FSMO Deadband from EU-off(deactivate*)
	tSet_FSMO_DB_COf : HALioDi_Type; (*DI:request FSMO Deadband from EU-off(deactivate*)
	F_FSMO_DB : INT; (*AI:FSMO Deadband reference from EU [Hz]*)
	tF_FSMO_DB : HALioAi_Type; (*AI:FSMO Deadband reference from EU [Hz]*)
	Set_FSM_RMC_Up_COn : BOOL; (*DI:request positive Margin from EU-on(activate*)
	tSet_FSM_RMC_Up_COn : HALioDi_Type; (*DI:request positive Margin from EU-on(activate*)
	Set_FSM_RMC_Up_COf : BOOL; (*DI:request positive Margin from EU-off(deactivate*)
	tSet_FSM_RMC_Up_COf : HALioDi_Type; (*DI:request positive Margin from EU-off(deactivate*)
	P_FSM_RMC_Up : INT; (*AI:positive Margin reference from EU [%Pnom]*)
	tP_FSM_RMC_Up : HALioAi_Type; (*AI:positive Margin reference from EU [%Pnom]*)
	Set_FSM_RMC_Down_COn : BOOL; (*DI:request negative Margin from EU-on(activate*)
	tSet_FSM_RMC_Down_COn : HALioDi_Type; (*DI:request negative Margin from EU-on(activate*)
	Set_FSM_RMC_Down_COf : BOOL; (*DI:request negative Margin from EU-off(deactivate*)
	tSet_FSM_RMC_Down_COf : HALioDi_Type; (*DI:request negative Margin from EU-off(deactivate*)
	P_FSM_RMC_Down : INT; (*AI:Negative Margin reference from EU [%Pnom]*)
	tP_FSM_RMC_Down : HALioAi_Type; (*AI:Negative Margin reference from EU [%Pnom]*)
	Set_U_Droop_COn : BOOL; (*DI:request U Droop from EU-on(activate*)
	tSet_U_Droop_COn : HALioDi_Type; (*DI:request U Droop from EU-on(activate*)
	Set_U_Droop_COf : BOOL; (*DI:request U Droop from EU-off(deactivate*)
	tSet_U_Droop_COf : HALioDi_Type; (*DI:request U Droop from EU-off(deactivate*)
	U_Droop : INT; (*AI:U Droop reference from EU [%]*)
	tU_Droop : HALioAi_Type; (*AI:U Droop reference from EU [%]*)
	Set_FSM_Rmp_COn : BOOL; (*DI:request ramp rate from EU-on(activate*)
	tSet_FSM_Rmp_COn : HALioDi_Type; (*DI:request ramp rate from EU-on(activate*)
	Set_FSM_Rmp_COf : BOOL; (*DI:request ramp rate from EU-off(deactivate*)
	tSet_FSM_Rmp_COf : HALioDi_Type; (*DI:request ramp rate from EU-off(deactivate*)
	FSM_Rmp_Up : INT; (*AI:Ramp rate UP reference from EU [%Pnom/s]*)
	tFSM_Rmp_Up : HALioAi_Type; (*AI:Ramp rate UP reference from EU [%Pnom/s]*)
	FSM_Rmp_Down : INT; (*AI:Ramp rate UP reference from EU [%Pnom/s]*)
	tFSM_Rmp_Down : HALioAi_Type; (*AI:Ramp rate UP reference from EU [%Pnom/s]*)
	Set_F_Ref_FSM_COn : BOOL; (*DI:request reference frequency for FSM/LFSM from EU-on(activate*)
	tSet_F_Ref_FSM_COn : HALioDi_Type; (*DI:request reference frequency for FSM/LFSM from EU-on(activate*)
	Set_F_Ref_FSM_COf : BOOL; (*DI:request reference frequency for FSM/LFSM from EU-off(deactivate*)
	tSet_F_Ref_FSM_COf : HALioDi_Type; (*DI:request reference frequency for FSM/LFSM from EU-off(deactivate*)
	F_Ref_FSM : INT; (*AI:Reference frequency for FSM/LFSM reference from EU [Hz]*)
	tF_Ref_FSM : HALioAi_Type; (*AI:Reference frequency for FSM/LFSM reference from EU [Hz]*)
	ECW_HydrPreH_Pump_Dem : BOOL; (*DO Hydraulic ECW pre-heating pump demand*)
	tECW_HydrPreH_Pump_Dem : HALioDo_Type; (*DO Hydraulic ECW pre-heating pump demand*)
	ECW_HydrPreH_Val_DemOpen : BOOL; (*DO Hydraulic ECW pre-heating valve demand open*)
	tECW_HydrPreH_Val_DemOpen : HALioDo_Type; (*DO Hydraulic ECW pre-heating valve demand open*)
	GV1_Opened : BOOL; (* 	DI Gasvalve position status	 *) (*OldName: NewPV  V4.07*)
	GV1_Closed : BOOL; (* 	DI Gasvalve position status	 *) (*OldName: NewPV  V4.07*)
	GV2_Opened : BOOL; (* 	DI Gasvalve position status	 *) (*OldName: NewPV  V4.07*)
	GV2_Closed : BOOL; (*	DI Gasvalve position status	 *) (*OldName: NewPV  V4.07*)
	tGV1_Opened : HALioDi_Type; (* 	DI Gasvalve position status	 *) (*OldName: NewPV  V4.07*)
	tGV1_Closed : HALioDi_Type; (* 	DI Gasvalve position status	 *) (*OldName: NewPV  V4.07*)
	tGV2_Opened : HALioDi_Type; (* 	DI Gasvalve position status	 *) (*OldName: NewPV  V4.07*)
	tGV2_Closed : HALioDi_Type; (*	DI Gasvalve position status	 *) (*OldName: NewPV  V4.07 *)
	GV_Upstream_Opened : BOOL; (*	DI Gasvalve position status	 *) (*OldName: NewPV  V4.07 *)
	GV_Upstream_Closed : BOOL; (*	DI Gasvalve position status	 *) (*OldName: NewPV  V4.07 *)
	tGV_Upstream_Opened : HALioDi_Type; (*	DI Gasvalve position status	 *) (*OldName: NewPV  V4.07 *)
	tGV_Upstream_Closed : HALioDi_Type; (*	DI Gasvalve position status	 *) (*OldName: NewPV  V4.07 *)
	GV_Upstream_Open : BOOL; (*	DI open External Customer Gasvalve	 *) (*OldName: NewPV  V4.07 *)
	GV_Upstream_Release : BOOL; (*	DI release External Customer Gasvalve	 *) (*OldName: NewPV  V4.07 *)
	tGV_Upstream_Open : HALioDo_Type; (*	Do open External Customer Gasvalve 	 *) (*OldName: NewPV  V4.07 *)
	tGV_Upstream_Release : HALioDo_Type; (*	DO release External Customer Gasvalve	 *) (*OldName: NewPV  V4.07 *)
	U_Set_Norm : INT; (* voltage output for island mode [%Unom] *) (*OldName:new pv V4.07 ;Cycle:5*)
	tU_Set_Norm : HALioAo_Type; (* voltage output for island mode [%Unom] *) (*OldName:new pv V4.07 ;Cycle:5*)
	U_SetExtAI_Norm : INT; (* External voltage set point [%Unom] *)
	tU_SetExtAI_Norm : HALioAi_Type; (* External voltage set point [%Unom] *)
	HWP1_Dem : BOOL; (*DO Redundant heating water pump 1 demand*)
	tHWP1_Dem : HALioDo_Type; (*DO Redundant heating water pump 1 demand*)
	HWP2_Dem : BOOL; (*DO Redundant heating water pump 2 demand*)
	tHWP2_Dem : HALioDo_Type; (*DO Redundant heating water pump 2 demand*)
	HWP1_Op : BOOL; (*DI Redundant heating water pump 1 operating*)
	tHWP1_Op : HALioDi_Type; (*DI Redundant heating water pump 1 operating*)
	HWP2_Op : BOOL; (*DI Redundant heating water pump 2 operating*)
	tHWP2_Op : HALioDi_Type; (*DI Redundant heating water pump 2 operating*)
	CCWP1_Dem : BOOL; (*DO Redundant charge cooler water pump 1 demand*)
	tCCWP1_Dem : HALioDo_Type; (*DO Redundant charge cooler water pump 1 demand*)
	CCWP2_Dem : BOOL; (*DO Redundant charge cooler water pump 2 demand*)
	tCCWP2_Dem : HALioDo_Type; (*DO Redundant charge cooler water pump 2 demand*)
	CCWP1_Op : BOOL; (*DI Redundant charge cooler water pump 1 operating*)
	tCCWP1_Op : HALioDi_Type; (*DI Redundant charge cooler water pump 1 operating*)
	CCWP2_Op : BOOL; (*DI Redundant charge cooler water pump 2 operating*)
	tCCWP2_Op : HALioDi_Type; (*DI Redundant charge cooler water pump 2 operating*)
	CC2WP1_Dem : BOOL; (*DO Redundant charge cooler 2 water pump 1 demand*)
	tCC2WP1_Dem : HALioDo_Type; (*DO Redundant charge cooler 2 water pump 1 demand*)
	CC2WP2_Dem : BOOL; (*DO Redundant charge cooler 2 water pump 2 demand*)
	tCC2WP2_Dem : HALioDo_Type; (*DO Redundant charge cooler 2 water pump 2 demand*)
	CC2WP1_Op : BOOL; (*DI Redundant charge cooler 2 water pump 1 operating*)
	tCC2WP1_Op : HALioDi_Type; (*DI Redundant charge cooler 2 water pump 1 operating*)
	CC2WP2_Op : BOOL; (*DI Redundant charge cooler 2 water pump 2 operating*)
	tCC2WP2_Op : HALioDi_Type; (*DI Redundant charge cooler 2 water pump 2 operating*)
	EmCWP_Op : BOOL; (*DI Emergency cooler water pump operating*)
	tEmCWP_Op : HALioDi_Type; (*DI Emergency cooler water pump operating*)
	EmCWP1_Dem : BOOL; (*DO Redundant emergency cooler water pump 1 demand*)
	tEmCWP1_Dem : HALioDo_Type; (*DO Redundant emergency cooler water pump 1 demand*)
	EmCWP2_Dem : BOOL; (*DO Redundant emergency cooler water pump 2 demand*)
	tEmCWP2_Dem : HALioDo_Type; (*DO Redundant emergency cooler water pump 2 demand*)
	EmCWP1_Op : BOOL; (*DI Redundant emergency cooler water pump 1 operating*)
	tEmCWP1_Op : HALioDi_Type; (*DI Redundant emergency cooler water pump 1 operating*)
	EmCWP2_Op : BOOL; (*DI Redundant emergency cooler water pump 2 operating*)
	tEmCWP2_Op : HALioDi_Type; (*DI Redundant emergency cooler water pump 2 operating*)
	BoilerFailure : BOOL; (*DI Boiler failure*)
	tBoilerFailure : HALioDi_Type; (*DI Boiler failure*)
	SeismicAlarm : BOOL; (*DI Seismic alarm (M.00-AI-100)*)
	tSeismicAlarm : HALioDi_Type; (*DI Seismic alarm (M.00-AI-100)*)
	Pr_EG_Deflag_Fast : INT; (*AI: Exhaust gas pressure fast (P.02-PI-010)*) (*OldName: Pr_OXIcat_In_Fast  V4.07*)
	tPr_EG_Deflag_Fast : HALioAi_Type; (*AI: Exhaust gas pressure fast (P.02-PI-010)*) (*OldName: Pr_OXIcat_In_Fast  V4.07*)
	T_SCR_Cat_HiHi : BOOL; (*SCR Exhaust temperatures CAT maximum - from customer (OK = TRUE)*) (*OldName: new PV; Cycle: 5;*) (*V04.07.00.00*)
	SCR_Catalyst_Rdy : BOOL; (*SCR Catalyst ready - from customer (Ready = TRUE)*) (*OldName: new PV; Cycle: 5;*) (*V04.07.00.00*)
	tT_SCR_Cat_HiHi : HALioDi_Type; (*SCR Exhaust temperatures CAT maximum - from customer (OK = TRUE)*) (*OldName: new PV; Cycle: 5;*) (*V04.07.00.00*)
	tSCR_Catalyst_Rdy : HALioDi_Type; (*SCR Catalyst ready - from customer (Ready = TRUE)*) (*OldName: new PV; Cycle: 5;*) (*V04.07.00.00*)
	P_Droop_Set : INT; (*Active power setpoint in frequency droop*)
	tP_Droop_Set : HALioAi_Type; (*Active power setpoint in frequency droop*)
	ExtCtrOk : BOOL; (* DI: External speed / voltage controller okay *)
	tExtCtrOk : HALioDi_Type; (* DI: External speed / voltage controller okay *)
	JunctionBox_GnlAlm : BOOL; (* General Alarm from junction box *)
	tJunctionBox_GnlAlm : HALioDi_Type; (* DI: General Alarm from junction box *)
	Execute_BS : BOOL; (* DO: Execute black out start *)
	tExecute_BS : HALioDo_Type; (* DO: Execute black out start *)
	EngBlock_PlantCtr : BOOL; (* DI: Module blocked by plant control *)
	tEngBlock_PlantCtr : HALioDi_Type; (* DI: Module blocked by plant control *)
	T_GT_NG : INT; (*AI Natural gas temperature mA Signal from customer via interface*)
	tT_GT_NG : HALioAi_Type; (*AI Natural gas temperature mA Signal from customer via interface*)
	Pr_GT_NG : INT; (*AI Natural gas pressure mA Signal from customer via interface*)
	tPr_GT_NG : HALioAi_Type; (*AI Natural gas pressure mA Signal from customer via interface*)
	Vol_GT_NG : INT; (*AI Natural gas volume mA Signal from customer via interface*)
	tVol_GT_NG : HALioAi_Type; (*AI Natural gas volume mA Signal from customer via interface*)
	T_EG_PrReliefVa1 : INT; (*AI temperature exhaust gas pressure relief valve 1 (P.02-TI-039)*)
	tT_EG_PrReliefVa1 : HALioAi_Type; (*AI temperature exhaust gas pressure relief valve 1 (P.02-TI-039)*)
	T_EG_PrReliefVa2 : INT; (*AI temperature exhaust gas pressure relief valve 2 (P.02-TI-040)*)
	tT_EG_PrReliefVa2 : HALioAi_Type; (*AI temperature exhaust gas pressure relief valve 2 (P.02-TI-040)*)
	GndFaultW : BOOL; (* DI earth fault warning *)
	tGndFaultW : HALioDi_Type; (* DI earth fault warning *)
	AirST_ValEngage : BOOL; (*DO: Air starter valve engage (E.31-YCS-001)*)
	AirST_ValStart : BOOL; (*DO: Air starter valve start (E.31-YCS-002)*)
	Pr_AirST_Engage : INT; (*AI: Pressure air starter engagement [bar] (E.31-PI-004)*)
	tAirST_ValEngage : HALioDo_Type; (*DO: Air starter valve engage (E.31-YCS-001)*)
	tAirST_ValStart : HALioDo_Type; (*DO: Air starter valve start (E.31-YCS-002)*)
	tPr_AirST_Engage : HALioAi_Type; (*AI: Pressure air starter engagement [bar] (E.31-PI-004)*)
	Pr_ECWaP1 : INT; (*AI Engine cooling water pressure after ECW pump 1 (M.04-PI-010)*)
	tPr_ECWaP1 : HALioAi_Type; (*AI Engine cooling water pressure after ECW pump 1 (M.04-PI-010)*)
	Pr_ECWaP2 : INT; (*AI Engine cooling water pressure after ECW pump 2 (M.04-PI-011)*)
	tPr_ECWaP2 : HALioAi_Type; (*AI Engine cooling water pressure after ECW pump 2 (M.04-PI-011)*)
	L_FreshOilTank_LoLo : BOOL; (*DI Fresh oil tank level low (2nd level switch)*)
	tL_FreshOilTank_LoLo : HALioDi_Type; (*DI Fresh oil tank level low (2nd level switch)*)
	L_DayOilTank_Lo : BOOL; (*DI Fresh oil day tank level low*)
	tL_DayOilTank_Lo : HALioDi_Type; (*DI Fresh oil day tank level low*)
	L_DayOilTank_LoLo : BOOL; (*DI Fresh oil day tank level low (2nd level switch)*)
	tL_DayOilTank_LoLo : HALioDi_Type; (*DI Fresh oil day tank level low (2nd level switch)*)
	OF_DayOilTank : BOOL; (*DI Overfill prevention device fresh oil day tank*)
	tOF_DayOilTank : HALioDi_Type; (*DI Overfill prevention device fresh oil day tank*)
	L_WasteOilDayTank_Hi : BOOL; (*DI Waste oil day tank level high*)
	tL_WasteOilDayTank_Hi : HALioDi_Type; (*DI Waste oil day tank level high*)
	OF_WasteOilDayTank : BOOL; (*DI Overfill prevention device waste oil day tank*)
	tOF_WasteOilDayTank : HALioDi_Type; (*DI Overfill prevention device waste oil day tank*)
	PS_FreshOilPump_Hi : BOOL; (*DI Fresh oil pump oil pressure maximum*)
	tPS_FreshOilPump_Hi : HALioDi_Type; (*DI Fresh oil pump oil pressure maximum*)
	FreshOilPump_Block : BOOL; (*DO Oil pressure max. Block fresh oil pump*)
	tFreshOilPump_Block : HALioDo_Type; (*DO Oil pressure max. Block fresh oil pump*)
	T_HW_EGHE_Hi : BOOL; (*DI Heating water temperature max. exhaust gas cooler*)
	tT_HW_EGHE_Hi : HALioDi_Type; (*DI Heating water temperature max. exhaust gas cooler*)
	T_HW_EGCD_Hi : BOOL; (*DI Heating water temperature max. exhaust gas condenser*)
	tT_HW_EGCD_Hi : HALioDi_Type; (*DI Heating water temperature max. exhaust gas condenser*)
	Cust_HW_Ext_Trip : BOOL; (*DI External heating water circuit monitoring*)
	tCust_HW_Ext_Trip : HALioDi_Type; (*DI External heating water circuit monitoring*)
	Dem_EU_Block2 : BOOL; (*DI module blocked from grid operator - shutdown*)
	tDem_EU_Block2 : HALioDi_Type; (*DI module blocked from grid operator - shutdown*)
	Dem_EU_Block3 : BOOL; (*DI module blocked from grid operator - demand off*)
	tDem_EU_Block3 : HALioDi_Type; (*DI module blocked from grid operator - demand off*)
	EU_RM_BLOCK2 : BOOL; (*module blocked from grid operator - shutdown*)
	tEU_RM_BLOCK2 : HALioDo_Type; (*module blocked from grid operator - shutdown*)
	EU_RM_BLOCK3 : BOOL; (*module blocked from grid operator - demand off*)
	tEU_RM_BLOCK3 : HALioDo_Type; (*module blocked from grid operator - demand off*)
	MCP_AuxPS_CB_Trip : BOOL; (*auxiliaries power supply circuit breaker module control panel tripped*)
	tMCP_AuxPS_CB_Trip : HALioDi_Type; (*auxiliaries power supply circuit breaker module control panel tripped*)
	MCP_AuxPS_CB_On : BOOL; (*auxiliaries power supply circuit breaker module control panel opened*)
	tMCP_AuxPS_CB_On : HALioDi_Type; (*auxiliaries power supply circuit breaker module control panel opened*)
	MCP_AuxPS_GndFault : BOOL; (*earth fault auxiliaries power supply module control panel*)
	tMCP_AuxPS_GndFault : HALioDi_Type; (*earth fault auxiliaries power supply module control panel*)
	MCP_FC_GndFault : BOOL; (*earth fault frequency converter module control panel*)
	tMCP_FC_GndFault : HALioDi_Type; (*earth fault frequency converter module control panel*)
	MIP_FC_GndFault : BOOL; (*earth fault frequency converter module interface panel*)
	tMIP_FC_GndFault : HALioDi_Type; (*earth fault frequency converter module interface panel*)
	AuxCP_FC_GndFault : BOOL; (*earth fault frequency converter auxiliaries control panel*)
	tAuxCP_FC_GndFault : HALioDi_Type; (*earth fault frequency converter auxiliaries control panel*)
	AuxCP_AuxPS_GndFault : BOOL; (*earth fault auxiliaries power supply auxiliaries control panel*)
	tAuxCP_AuxPS_GndFault : HALioDi_Type; (*earth fault auxiliaries power supply auxiliaries control panel*)
	AuxCP_AuxPS_CB_Trip : BOOL; (*auxiliaries power supply circuit breaker auxiliaries control panel tripped*)
	tAuxCP_AuxPS_CB_Trip : HALioDi_Type; (*auxiliaries power supply circuit breaker auxiliaries control panel tripped*)
	AuxCP_AuxPS_CB_On : BOOL; (*auxiliaries power supply circuit breaker auxiliaries control panel opened*)
	tAuxCP_AuxPS_CB_On : HALioDi_Type; (*auxiliaries power supply circuit breaker auxiliaries control panel opened*)
	GndFault_BB : BOOL; (*earth fault bus bar*)
	tGndFault_BB : HALioDi_Type; (*earth fault bus bar*)
	TR_AuxPS_GndFault : BOOL; (*earth fault auxiliaries power supply thermal reactor panel*)
	tTR_AuxPS_GndFault : HALioDi_Type; (*earth fault auxiliaries power supply thermal reactor panel*)
	TR_AuxPS_CB_Trip : BOOL; (*auxiliaries power supply circuit breaker thermal reactor panel tripped*)
	tTR_AuxPS_CB_Trip : HALioDi_Type; (*auxiliaries power supply circuit breaker thermal reactor panel tripped*)
	TR_AuxPS_CB_On : BOOL; (*auxiliaries power supply circuit breaker thermal reactor panel opened*)
	tTR_AuxPS_CB_On : HALioDi_Type; (*auxiliaries power supply circuit breaker thermal reactor panel opened*)
	ECWP_CB_On : BOOL; (*DI engine cooling water pump circuit breaker on*)
	tECWP_CB_On : HALioDi_Type; (*DI engine cooling water pump circuit breaker on*)
	U_BufferBat1 : INT; (*AI Buffer battery 1 voltage [V]*)
	tU_BufferBat1 : HALioAi_Type; (*AI Buffer battery 1 voltage [V]*)
	U_BufferBat2 : INT; (*AI Buffer battery 2 voltage [V]*)
	tU_BufferBat2 : HALioAi_Type; (*AI Buffer battery 2 voltage [V]*)
	BufferBat1_Disconnect : BOOL; (*DO Disconnect buffer battery 1*)
	tBufferBat1_Disconnect : HALioDo_Type; (*DO Disconnect buffer battery 1*)
	BufferBat2_Disconnect : BOOL; (*DO Disconnect buffer battery 2*)
	tBufferBat2_Disconnect : HALioDo_Type; (*DO Disconnect buffer battery 2*)
	BufferBat1_ConnectLoad : BOOL; (*DO Connect load resistor buffer battery 1*)
	tBufferBat1_ConnectLoad : HALioDo_Type; (*DO Connect load resistor buffer battery 1*)
	BufferBat2_ConnectLoad : BOOL; (*DO Connect load resistor buffer battery 2*)
	tBufferBat2_ConnectLoad : HALioDo_Type; (*DO Connect load resistor buffer battery 2*)
	StarterBat_ConnectLoad : BOOL; (*DO Connect load resistor starter battery*)
	tStarterBat_ConnectLoad : HALioDo_Type; (*DO Connect load resistor starter battery*)
	BatChargeDev_Ok : BOOL; (*DO Status battery charging devices*)
	tBatChargeDev_Ok : HALioDi_Type; (*DO Status battery charging devices*)
	Leak_OilExtensionTank1 : BOOL; (*DI Oil leakage detection additional oil tank 1 (P.03-LS-021)*)
	tLeak_OilExtensionTank1 : HALioDi_Type; (*DI Oil leakage detection additional oil tank 1 (P.03-LS-021)*)
	Leak_OilExtensionTank2 : BOOL; (*DI Oil leakage detection additional oil tank 2 (P.03-LS-031)*)
	tLeak_OilExtensionTank2 : HALioDi_Type; (*DI Oil leakage detection additional oil tank 2 (P.03-LS-031)*)
	Leak_OilExtensionTank3 : BOOL; (*DI Oil leakage detection additional oil tank 3 (P.03-LS-041)*)
	tLeak_OilExtensionTank3 : HALioDi_Type; (*DI Oil leakage detection additional oil tank 3 (P.03-LS-041)*)
	F_FSM_Simulated : INT; (*simulated test frequency in FSM/LFSM test mode[Hz]*)
	tF_FSM_Simulated : HALioAo_Type; (*simulated test frequency in FSM/LFSM test mode[Hz]*)
	U_CtrlBat : ARRAY[1..iNum_CtrlBatMon] OF INT; (*AI Control battery voltage [V]*)
	tU_CtrlBat : ARRAY[1..iNum_CtrlBatMon] OF HALioAi_Type; (*AI Control battery voltage [V]*)
	CtrlBat_Disconnect : ARRAY[1..iNum_CtrlBatMon] OF BOOL; (*DO Disconnect control battery set X*)
	tCtrlBat_Disconnect : ARRAY[1..iNum_CtrlBatMon] OF HALioDo_Type; (*DO Disconnect control battery set X*)
	CtrlBat_ConnectLoad : ARRAY[1..iNum_CtrlBatMon] OF BOOL; (*DO Connect load resistor control battery set X*)
	tCtrlBat_ConnectLoad : ARRAY[1..iNum_CtrlBatMon] OF HALioDo_Type; (*DO Connect load resistor control battery set X*)
	CtrlBat_ChargeDev_Ok : ARRAY[1..iNum_CtrlBatMon] OF BOOL; (*DO Status control battery charging devices*)
	tCtrlBat_ChargeDev_Ok : ARRAY[1..iNum_CtrlBatMon] OF HALioDi_Type; (*DO Status control battery charging devices*)
	Q_Droop_Set : INT; (*reactive power setpoint for voltage droop mode*)
	tQ_Droop_Set : HALioAi_Type; (*reactive power setpoint for voltage droop mode*)
	DemGenExcOff : BOOL; (*demand generator excitation off*)
	tDemGenExcOff : HALioDi_Type; (*demand generator excitation off*)
	GenExcOff : BOOL; (*generator de-energized(excitation off)*)
	tGenExcOff : HALioDo_Type; (*generator de-energized(excitation off)*)
	SyOMSS_Man : BOOL; (*synchronization operating mode selection MANUAL*)
	tSyOMSS_Man : HALioDo_Type; (*synchronization operating mode selection MANUAL*)
	SyOMSS_Aut : BOOL; (*synchronization operating mode selection AUTO*)
	tSyOMSS_Aut : HALioDo_Type; (*synchronization operating mode selection AUTO*)
	GenBearGreasSys2DE : BOOL; (*INNIO STAR CONTROL SYSTEM Pin2 drive end DE bearing*)
	tGenBearGreasSys2DE : HALioDi_Type; (*INNIO STAR CONTROL SYSTEM Pin2 drive end DE bearing*)
	GenBearGreasSys4DE : BOOL; (*INNIO STAR CONTROL SYSTEM Pin4 drive end DE bearing*)
	tGenBearGreasSys4DE : HALioDi_Type; (*INNIO STAR CONTROL SYSTEM Pin4 drive end DE bearing*)
	GenBearGreasSys2NDE : BOOL; (*INNIO STAR CONTROL SYSTEM Pin2 non-drive end NDE bearing*)
	tGenBearGreasSys2NDE : HALioDi_Type; (*INNIO STAR CONTROL SYSTEM Pin2 non-drive end NDE bearing*)
	GenBearGreasSys4NDE : BOOL; (*INNIO STAR CONTROL SYSTEM Pin4 non-drive end NDE bearing*)
	tGenBearGreasSys4NDE : HALioDi_Type; (*INNIO STAR CONTROL SYSTEM Pin4 non-drive end NDE bearing*)
	L_FreshOilTank : INT := 0; (*V4.12 Spec 2022-112*)
	tL_FreshOilTank : HALioAi_Type := (0); (*V4.12 Spec 2022-112*)
	L_WasteOilTank : INT := 0; (*V4.12 Spec 2022-112*)
	tL_WasteOilTank : HALioAi_Type := (0); (*V4.12 Spec 2022-112*)
	L_DayOilTank : INT := 0; (*V4.12 Spec 2022-112*)
	tL_DayOilTank : HALioAi_Type := (0); (*V4.12 Spec 2022-112*)
	DI_TestBench_TripPrio2 : BOOL := TRUE; (*A2399 - Shut down test bench priority 2*)
	tDI_TestBench_TripPrio2 : HALioDi_Type; (*A2399 - Shut down test bench priority 2*)
	DI_TestBench_TripPrio3 : BOOL := TRUE; (*A2400 - Shut down test bench priority 3*)
	tDI_TestBench_TripPrio3 : HALioDi_Type; (*A2400 - Shut down test bench priority 3*)
	DI_TestBench_Warning : BOOL := TRUE; (* W9400 - Warning test bench *)
	tDI_TestBench_Warning : HALioDi_Type; (* W9400 - Warning test bench *)
	GT_H2 : INT; (* H2 content [%] *)
	tGT_H2 : HALioAi_Type; (* H2 content [%] *)
	GT_RatioMix_Set : INT; (* Gas mixing ratio in percent. 1.0 = 100% *)
	tGT_RatioMix_Set : HALioAi_Type; (* Gas mixing ratio in percent. 1.0 = 100% *)
	iTimeStamp_PosZeroCrossing_UGen1 : DINT; (*TimeStamp of last positive zero crossing UGen1 [ 1 / 4096microseconds]*)
	iTimeStamp_PosZeroCrossing_UGen2 : DINT; (*TimeStamp of last positive zero crossing UGen2 [ 1 / 4096microseconds]*)
	iTimeStamp_PosZeroCrossing_UGen3 : DINT; (*TimeStamp of last positive zero crossing UGen3 [ 1 / 4096microseconds]*)
	BurstingDisk1_Ok : BOOL; (*DI exhaust Monitoring bursting disc 1 (P.02-GS-001)*)
	tBurstingDisk1_Ok : HALioDi_Type; (*DI exhaust Monitoring bursting disc 1 (P.02-GS-001)*)
	BurstingDisk2_Ok : BOOL; (*DI exhaust Monitoring bursting disc 2 (P.02-GS-002)*)
	tBurstingDisk2_Ok : HALioDi_Type; (*DI exhaust Monitoring bursting disc 2 (P.02-GS-002)*)
	Pos_ThR_AuxGasCV_Act : INT; (* Thermal reactor - auxiliary gas injection control valve position [%] (P.16-S-001) *)
	tPos_ThR_AuxGasCV_Act : HALioAi_Type; (* Thermal reactor - auxiliary gas injection control valve position [%] (P.16-S-001) *)
	Pr_ThR_AuxGasBeforeCV : INT; (* Thermal reactor - auxiliary gas pressure before control valve [mbar] (P.16-PI-010) *)
	tPr_ThR_AuxGasBeforeCV : HALioAi_Type; (* Thermal reactor - auxiliary gas pressure before control valve [mbar] (P.16-PI-010) *)
	Pr_ThR_AuxGasAfterCV : INT; (* Thermal reactor - auxiliary gas pressure after control valve [mbar] (P.16-PI-020) *)
	tPr_ThR_AuxGasAfterCV : HALioAi_Type; (* Thermal reactor - auxiliary gas pressure after control valve [mbar] (P.16-PI-020) *)
	Lev_SCR_UreaTank : INT; (*SCR Urea tank level [%] (P.29-LI-001)*) (*OldName: new PV; Cycle: 5;*) (*V04.13.00.00*)
	tLev_SCR_UreaTank : HALioAi_Type; (*SCR Urea tank level [%] (P.29-LI-001)*) (*OldName: new PV; Cycle: 5;*) (*V04.13.00.00*)
	tReq_PowMod : HALioDi_Type; (*DI request power mode*)
	tECW_ShutOffVal_Dem : HALioDo_Type; (*DO: Demand 2-way shut off valve engine jacket water circuit*)
	ECW_ShutOffVal_Dem : BOOL; (*DO: Demand 2-way shut off valve engine jacket water circuit*)
	tValHeater_Dem : HALioDo_Type; (*DO: Demand 3-way valve heater*)
	ValHeater_Dem : BOOL; (*DO: Demand 3-way valve heater*)
	tFanRingHeater_Dem : HALioDo_Type; (*DO: Demand fan ring heater*)
	FanRingHeater_Dem : BOOL; (*DO: Demand fan ring heater*)
	ThR2_EH_group1_Dem : BOOL; (* Thermal reactor 2 - electrical heating group 1 - command On (P.16-W-101,102,103,104,105) *)
	tThR2_EH_group1_Dem : HALioDo_Type; (* Thermal reactor 2 - electrical heating group 1 - command On (P.16-W-101,102,103,104,105) *)
	ThR2_EH_group2_Dem : BOOL; (* Thermal reactor 2 - electrical heating group 2 - command On (P.16-W-201,202,203) *)
	tThR2_EH_group2_Dem : HALioDo_Type; (* Thermal reactor 2 - electrical heating group 2 - command On (P.16-W-201,202,203) *)
	ThR2_EH_group3_Dem : BOOL; (* Thermal reactor 2 - electrical heating group 3 - command On (P.16-W-301,302,303,304,305) *)
	tThR2_EH_group3_Dem : HALioDo_Type; (* Thermal reactor 2 - electrical heating group 3 - command On (P.16-W-301,302,303,304,305) *)
	ThR2_EH_group4_Dem : BOOL; (* Thermal reactor 2 - electrical heating group 4 - command On (P.16-W-401,402,403) *)
	tThR2_EH_group4_Dem : HALioDo_Type; (* Thermal reactor 2 - electrical heating group 4 - command On (P.16-W-401,402,403) *)
	ThR2_EH_group5_Dem : BOOL; (* Thermal reactor 2 - electrical heating group 5 - command On (P.16-W-501,502,503,504,505) *)
	tThR2_EH_group5_Dem : HALioDo_Type; (* Thermal reactor 2 - electrical heating group 5 - command On (P.16-W-501,502,503,504,505) *)
	ThR2_AuxGasShutOffValve_Dem : BOOL; (* Thermal reactor 2 - solenoid valve gas injection - command Open (P.16-YCS-009) *)
	tThR2_AuxGasShutOffValve_Dem : HALioDo_Type; (* Thermal reactor 2 - solenoid valve gas injection - command Open (P.16-YCS-009) *)
	Pr_ThR2_Inlet : INT; (* Thermal reactor 2 - inlet pressure [mbar] (P.02-PI-201) *)
	tPr_ThR2_Inlet : HALioAi_Type; (* Thermal reactor 2 - inlet pressure [mbar] (P.02-PI-201) *)
	Pr_ThR2_Outlet : INT; (* Thermal reactor 2 - outlet pressure [mbar] (P.02-PI-202) *)
	tPr_ThR2_Outlet : HALioAi_Type; (* Thermal reactor 2 - outlet pressure [mbar] (P.02-PI-202) *)
	T_ThR2_EH_group1 : INT; (* Thermal reactor 2 - electrical heating group 1 - temperature [degC] (P.16-TI-101) *)
	tT_ThR2_EH_group1 : HALioAi_Type; (* Thermal reactor 2 - electrical heating group 1 - temperature [degC] (P.16-TI-101) *)
	T_ThR2_EH_group2 : INT; (* Thermal reactor 2 - electrical heating group 2 - temperature [degC] (P.16-TI-201) *)
	tT_ThR2_EH_group2 : HALioAi_Type; (* Thermal reactor 2 - electrical heating group 2 - temperature [degC] (P.16-TI-201) *)
	T_ThR2_EH_group3 : INT; (* Thermal reactor 2 - electrical heating group 3 - temperature [degC] (P.16-TI-301) *)
	tT_ThR2_EH_group3 : HALioAi_Type; (* Thermal reactor 2 - electrical heating group 3 - temperature [degC] (P.16-TI-301) *)
	T_ThR2_EH_group4 : INT; (* Thermal reactor 2 - electrical heating group 4 - temperature [degC] (P.16-TI-401) *)
	tT_ThR2_EH_group4 : HALioAi_Type; (* Thermal reactor 2 - electrical heating group 4 - temperature [degC] (P.16-TI-401) *)
	T_ThR2_EH_group5 : INT; (* Thermal reactor 2 - electrical heating group 5 - temperature [degC] (P.16-TI-501) *)
	tT_ThR2_EH_group5 : HALioAi_Type; (* Thermal reactor 2 - electrical heating group 5 - temperature [degC] (P.16-TI-501) *)
	T_ThR2_LeftChamber : INT; (* Thermal reactor 2 - chamber temperature left side [degC] (P.16-TI-018) *)
	tT_ThR2_LeftChamber : HALioAi_Type; (* Thermal reactor 2 - chamber temperature left side [degC] (P.16-TI-018) *)
	T_ThR2_RightChamber : INT; (* Thermal reactor 2 - chamber temperature right side [degC] (P.16-TI-017) *)
	tT_ThR2_RightChamber : HALioAi_Type; (* Thermal reactor 2 - chamber temperature right side [degC] (P.16-TI-017) *)
	T_ThR2_Downstream : INT; (* Thermal reactor 2 - downstream temperature [degC] (P.16-TI-021) *)
	tT_ThR2_Downstream : HALioAi_Type; (* Thermal reactor 2 - downstream temperature [degC] (P.16-TI-021) *)
	ThR2_T_UnitOk_LeftCh : BOOL; (* Thermal reactor 2 - Sensor processing unit ok - chamber temperature left side (P.16-TI-018) *)
	tThR2_T_UnitOk_LeftCh : HALioDi_Type; (* Thermal reactor 2 - Sensor processing unit ok - chamber temperature left side (P.16-TI-018) *)
	ThR2_T_UnitOk_RightCh : BOOL; (* Thermal reactor 2 - Sensor processing unit ok - chamber temperature right side (P.16-TI-017) *)
	tThR2_T_UnitOk_RightCh : HALioDi_Type; (* Thermal reactor 2 - Sensor processing unit ok - chamber temperature right side (P.16-TI-017) *)
	ThR2_T_UnitOk_Downstream : BOOL; (* Thermal reactor 2 - Sensor processing unit ok - downstream temperature (P.16-TI-021) *)
	tThR2_T_UnitOk_Downstream : HALioDi_Type; (* Thermal reactor 2 - Sensor processing unit ok - downstream temperature (P.16-TI-021) *)
	tPr_GT_b_Reg : HALioAi_Type; (* Gas pressure before pressure regulator [bar] (P.01-PI-101) *)
	Pr_GT_b_Reg : INT; (* Gas pressure before pressure regulator [bar] (P.01-PI-101) *)
	tPr_GT_a_Reg : HALioAi_Type; (* Gas pressure after pressure regulator [bar] (P.01-PI-109) *)
	Pr_GT_a_Reg : INT; (* Gas pressure after pressure regulator [bar] (P.01-PI-109) *)
	tPr_N2_GT : HALioAi_Type; (* Nitrogen pressure sensor inlet gas train [bar] (P.15-PI-002) *)
	Pr_N2_GT : INT; (* Nitrogen pressure sensor inlet gas train [bar] (P.15-PI-002) *)
	tGV_N2_Open : HALioDo_Type; (* Nitrogen purging valve (P.15-YCS-001) (P.15-YCS-002) *)
	GV_N2_Open : BOOL; (* Nitrogen purging valve (P.15-YCS-001) (P.15-YCS-002) *)
	GasSysErr : BOOL; (*SAFETY PLC: DI System failure - Gas detection system (P.17-JI-200)*) (*OldName: new PV; Cycle: 5;*) (*V04.25.00.00*)
	tGasSysErr : HALioDi_Type; (*SAFETY PLC: DI System failure - Gas detection system (P.17-JI-200)*) (*OldName: new PV; Cycle: 5;*) (*V04.25.00.00*)
	FireSysErr : BOOL; (*SAFETY PLC: DI System failure - Fire detection system (P.17-JI-001)*) (*OldName: new PV; Cycle: 5;*) (*V04.25.00.00*)
	tFireSysErr : HALioDi_Type; (*SAFETY PLC: DI System failure - Fire detection system (P.17-JI-001)*) (*OldName: new PV; Cycle: 5;*) (*V04.25.00.00*)
	SL_TS_ECW : BOOL; (*SAFETY PLC: DI Safety loop - Engine cooling water temperature switch - Engine outlet (M.04-TI-001)*) (*OldName: new PV; Cycle: 5;*) (*V04.25.00.00*)
	tSL_TS_ECW : HALioDi_Type; (*SAFETY PLC: DI Safety loop - Engine cooling water temperature switch - Engine outlet (M.04-TI-001)*) (*OldName: new PV; Cycle: 5;*) (*V04.25.00.00*)
	SL_TS_HW_Su_Unit : BOOL; (*SAFETY PLC: DI Safety loop - Heating water supply temperature switch - Unit (M.06-TI-003)*) (*OldName: new PV; Cycle: 5;*) (*V04.25.00.00*)
	tSL_TS_HW_Su_Unit : HALioDi_Type; (*SAFETY PLC: DI Safety loop - Heating water supply temperature switch - Unit (M.06-TI-003)*) (*OldName: new PV; Cycle: 5;*) (*V04.25.00.00*)
	T_HW_Su_Unit : INT; (*SAFETY PLC: Heating water supply temperature - Unit (M.06-TI-003)*) (*OldName: new PV; Cycle: 5;*) (*V04.25.00.00*)
	tT_HW_Su_Unit : HALioAi_Type; (*SAFETY PLC: Heating water supply temperature - Unit (M.06-TI-003)*) (*OldName: new PV; Cycle: 5;*) (*V04.25.00.00*)
	EmStop_ER1 : BOOL; (*SAFETY PLC: Emergency stop push button - Engine room button 1*) (*OldName: new PV; Cycle: 5;*) (*V04.25.00.00*)
	EmStop_ER2 : BOOL; (*SAFETY PLC: Emergency stop push button - Engine room button 2*) (*OldName: new PV; Cycle: 5;*) (*V04.25.00.00*)
	EmStop_ER3 : BOOL; (*SAFETY PLC: Emergency stop push button - Engine room button 3*) (*OldName: new PV; Cycle: 5;*) (*V04.25.00.00*)
	EmStop_ER4 : BOOL; (*SAFETY PLC: Emergency stop push button - Engine room button 4*) (*OldName: new PV; Cycle: 5;*) (*V04.25.00.00*)
	EmStop_EXT : BOOL; (*SAFETY PLC: Emergency stop push button - External*) (*OldName: new PV; Cycle: 5;*) (*V04.25.00.00*)
	EmStop_TR : BOOL; (*SAFETY PLC: Emergency stop push button - Thermal reactor control panel*) (*OldName: new PV; Cycle: 5;*) (*V04.25.00.00*)
	EmStop_IP : BOOL; (*SAFETY PLC: Emergency stop push button - Interlock control panel*) (*OldName: new PV; Cycle: 5;*) (*V04.25.00.00*)
	EmStop_MCP : BOOL; (*SAFETY PLC: Emergency stop push button - Master control panel*) (*OldName: new PV; Cycle: 5;*) (*V04.25.00.00*)
	EmStop_EGAT : BOOL; (*SAFETY PLC: Emergency stop push button - Exhaust gas after treatment control panel*) (*OldName: new PV; Cycle: 5;*) (*V04.25.00.00*)
	EmStop_PCGC : BOOL; (*SAFETY PLC: Emergency stop push button - Prechamber gas compressor*) (*OldName: new PV; Cycle: 5;*) (*V04.25.00.00*)
	EmStop_AUX : BOOL; (*SAFETY PLC: Emergency stop push button - Auxiliaries control panel*) (*OldName: new PV; Cycle: 5;*) (*V04.25.00.00*)
	tEmStop_ER1 : HALioDi_Type; (*SAFETY PLC: Emergency stop push button - Engine room button 1*) (*OldName: new PV; Cycle: 5;*) (*V04.25.00.00*)
	tEmStop_ER2 : HALioDi_Type; (*SAFETY PLC: Emergency stop push button - Engine room button 2*) (*OldName: new PV; Cycle: 5;*) (*V04.25.00.00*)
	tEmStop_ER3 : HALioDi_Type; (*SAFETY PLC: Emergency stop push button - Engine room button 3*) (*OldName: new PV; Cycle: 5;*) (*V04.25.00.00*)
	tEmStop_ER4 : HALioDi_Type; (*SAFETY PLC: Emergency stop push button - Engine room button 4*) (*OldName: new PV; Cycle: 5;*) (*V04.25.00.00*)
	tEmStop_EXT : HALioDi_Type; (*SAFETY PLC: Emergency stop push button - External*) (*OldName: new PV; Cycle: 5;*) (*V04.25.00.00*)
	tEmStop_TR : HALioDi_Type; (*SAFETY PLC: Emergency stop push button - Thermal reactor control panel*) (*OldName: new PV; Cycle: 5;*) (*V04.25.00.00*)
	tEmStop_IP : HALioDi_Type; (*SAFETY PLC: Emergency stop push button - Interlock control panel*) (*OldName: new PV; Cycle: 5;*) (*V04.25.00.00*)
	tEmStop_MCP : HALioDi_Type; (*SAFETY PLC: Emergency stop push button - Master control panel*) (*OldName: new PV; Cycle: 5;*) (*V04.25.00.00*)
	tEmStop_EGAT : HALioDi_Type; (*SAFETY PLC: Emergency stop push button - Exhaust gas after treatment control panel*) (*OldName: new PV; Cycle: 5;*) (*V04.25.00.00*)
	tEmStop_PCGC : HALioDi_Type; (*SAFETY PLC: Emergency stop push button - Prechamber gas compressor*) (*OldName: new PV; Cycle: 5;*) (*V04.25.00.00*)
	tEmStop_AUX : HALioDi_Type; (*SAFETY PLC: Emergency stop push button - Auxiliaries control panel*) (*OldName: new PV; Cycle: 5;*) (*V04.25.00.00*)
	DCGA_GV_Open : BOOL; (*DOopen Decentral gas admission valve*) (*SAFETY PLC*) (*V04.25.00.00*)
	tDCGA_GV_Open : HALioDo_Type; (*DOopen Decentral gas admission valve*) (*SAFETY PLC*) (*V04.25.00.00*)
	DCGA_GV1_Open : BOOL; (*DO Decentral gas admission - Gasvalve 1*) (*SAFETY PLC*) (*V04.25.00.00*)
	tDCGA_GV1_Open : HALioDo_Type; (*DO Decentral gas admission - Gasvalve 1*) (*SAFETY PLC*) (*V04.25.00.00*)
	DCGA_GV2_Open : BOOL; (*DO Decentral gas admission - Gasvalve 2*) (*SAFETY PLC*) (*V04.25.00.00*)
	tDCGA_GV2_Open : HALioDo_Type; (*DO Decentral gas admission - Gasvalve 2*) (*SAFETY PLC*) (*V04.25.00.00*)
	ERV_INL1_Lou_OP : BOOL; (*Engine room ventilation inlet air louvre - Group 1 opened (P.17-S-100)*)
	tERV_INL1_Lou_OP : HALioDi_Type; (*Engine room ventilation inlet air louvre - Group 1 opened (P.17-S-100)*)
	ERV_INL2_Lou_OP : BOOL; (*Engine room ventilation inlet air louvre - Group 2 opened (P.17-S-110)*)
	tERV_INL2_Lou_OP : HALioDi_Type; (*Engine room ventilation inlet air louvre - Group 2 opened (P.17-S-110)*)
	ERV_INL3_Lou_OP : BOOL; (*Engine room ventilation inlet air louvre - Group 3 opened (P.17-S-120)*)
	tERV_INL3_Lou_OP : HALioDi_Type; (*Engine room ventilation inlet air louvre - Group 3 opened (P.17-S-120)*)
	ERV_INL4_Lou_OP : BOOL; (*Engine room ventilation inlet air louvre - Group 4 opened (P.17-S-130)*)
	tERV_INL4_Lou_OP : HALioDi_Type; (*Engine room ventilation inlet air louvre - Group 4 opened (P.17-S-130)*)
	ERV_INL5_Lou_OP : BOOL; (*Engine room ventilation inlet air louvre - Group 5 opened (P.17-S-140) *)
	tERV_INL5_Lou_OP : HALioDi_Type; (*Engine room ventilation inlet air louvre - Group 5 opened (P.17-S-140)*)
	ERV_INL6_Lou_OP : BOOL; (*Engine room ventilation inlet air louvre - Group 6 opened (P.17-S-150)*)
	tERV_INL6_Lou_OP : HALioDi_Type; (*Engine room ventilation inlet air louvre - Group 6 opened (P.17-S-150)*)
	ERV_INL1_Lou_CL : BOOL; (*Engine room ventilation inlet air louvre - Group 1 closed (P.17-S-102)*)
	tERV_INL1_Lou_CL : HALioDi_Type; (*Engine room ventilation inlet air louvre - Group 1 closed (P.17-S-102)*)
	ERV_INL2_Lou_CL : BOOL; (*Engine room ventilation inlet air louvre - Group 2 closed (P.17-S-112)*)
	tERV_INL2_Lou_CL : HALioDi_Type; (*Engine room ventilation inlet air louvre - Group 2 closed (P.17-S-112)*)
	ERV_INL3_Lou_CL : BOOL; (*Engine room ventilation inlet air louvre - Group 3 closed (P.17-S-122)*)
	tERV_INL3_Lou_CL : HALioDi_Type; (*Engine room ventilation inlet air louvre - Group 3 closed (P.17-S-122)*)
	ERV_INL4_Lou_CL : BOOL; (*Engine room ventilation inlet air louvre - Group 4 closed (P.17-S-132)*)
	tERV_INL4_Lou_CL : HALioDi_Type; (*Engine room ventilation inlet air louvre - Group 4 closed (P.17-S-132)*)
	ERV_INL5_Lou_CL : BOOL; (*Engine room ventilation inlet air louvre - Group 5 closed (P.17-S-142)*)
	tERV_INL5_Lou_CL : HALioDi_Type; (*Engine room ventilation inlet air louvre - Group 5 closed (P.17-S-142)*)
	ERV_INL6_Lou_CL : BOOL; (*Engine room ventilation inlet air louvre - Group 6 closed (P.17-S-152)*)
	tERV_INL6_Lou_CL : HALioDi_Type; (*Engine room ventilation inlet air louvre - Group 6 closed (P.17-S-152) *)
	ERV_OTL1_Lou_OP : BOOL; (*Engine room ventilation outlet air louvre - Group 1 opened (P.17-S-101)*)
	tERV_OTL1_Lou_OP : HALioDi_Type; (*Engine room ventilation outlet air louvre - Group 1 opened (P.17-S-101)*)
	ERV_OTL2_Lou_OP : BOOL; (*Engine room ventilation outlet air louvre - Group 2 opened (P.17-S-111)*)
	tERV_OTL2_Lou_OP : HALioDi_Type; (*Engine room ventilation outlet air louvre - Group 2 opened (P.17-S-111) *)
	ERV_OTL3_Lou_OP : BOOL; (*Engine room ventilation outlet air louvre - Group 3 opened (P.17-S-121)*)
	tERV_OTL3_Lou_OP : HALioDi_Type; (*Engine room ventilation outlet air louvre - Group 3 opened (P.17-S-121)*)
	ERV_OTL4_Lou_OP : BOOL; (*Engine room ventilation outlet air louvre - Group 4 opened (P.17-S-131)*)
	tERV_OTL4_Lou_OP : HALioDi_Type; (*Engine room ventilation outlet air louvre - Group 4 opened (P.17-S-131)*)
	ERV_OTL5_Lou_OP : BOOL; (*Engine room ventilation outlet air louvre - Group 5 opened (P.17-S-141)*)
	tERV_OTL5_Lou_OP : HALioDi_Type; (*Engine room ventilation outlet air louvre - Group 5 opened (P.17-S-141)*)
	ERV_OTL6_Lou_OP : BOOL; (*Engine room ventilation outlet air louvre - Group 6 opened (P.17-S-151)*)
	tERV_OTL6_Lou_OP : HALioDi_Type; (*Engine room ventilation outlet air louvre - Group 6 opened (P.17-S-151)*)
	ERV_OTL1_Lou_CL : BOOL; (*Engine room ventilation outlet air louvre - Group 1 closed (P.17-S-103)*)
	tERV_OTL1_Lou_CL : HALioDi_Type; (*Engine room ventilation outlet air louvre - Group 1 closed (P.17-S-103)*)
	ERV_OTL2_Lou_CL : BOOL; (*Engine room ventilation outlet air louvre - Group 2 closed (P.17-S-113)*)
	tERV_OTL2_Lou_CL : HALioDi_Type; (*Engine room ventilation outlet air louvre - Group 2 closed (P.17-S-113)*)
	ERV_OTL3_Lou_CL : BOOL; (*Engine room ventilation outlet air louvre - Group 3 closed (P.17-S-123)*)
	tERV_OTL3_Lou_CL : HALioDi_Type; (*Engine room ventilation outlet air louvre - Group 3 closed (P.17-S-123)*)
	ERV_OTL4_Lou_CL : BOOL; (*Engine room ventilation outlet air louvre - Group 4 closed (P.17-S-133)*)
	tERV_OTL4_Lou_CL : HALioDi_Type; (*Engine room ventilation outlet air louvre - Group 4 closed (P.17-S-133)*)
	ERV_OTL5_Lou_CL : BOOL; (*Engine room ventilation outlet air louvre - Group 5 closed (P.17-S-143)*)
	tERV_OTL5_Lou_CL : HALioDi_Type; (*Engine room ventilation outlet air louvre - Group 5 closed (P.17-S-143)*)
	ERV_OTL6_Lou_CL : BOOL; (*Engine room ventilation outlet air louvre - Group 6 closed (P.17-S-153)*)
	tERV_OTL6_Lou_CL : HALioDi_Type; (*Engine room ventilation outlet air louvre - Group 6 closed (P.17-S-153)*)
	ERV_INL1_Fan_Run : BOOL; (*Engine room ventilation inlet air fan - Group 1 in operation (P.17-SC-200)*)
	tERV_INL1_Fan_Run : HALioDi_Type; (*Engine room ventilation inlet air fan - Group 1 in operation (P.17-SC-200)*)
	ERV_INL2_Fan_Run : BOOL; (*Engine room ventilation inlet air fan - Group 2 in operation (P.17-SC-210)*)
	tERV_INL2_Fan_Run : HALioDi_Type; (*Engine room ventilation inlet air fan - Group 2 in operation (P.17-SC-210)*)
	ERV_INL3_Fan_Run : BOOL; (*Engine room ventilation inlet air fan - Group 3 in operation (P.17-SC-220)*)
	tERV_INL3_Fan_Run : HALioDi_Type; (*Engine room ventilation inlet air fan - Group 3 in operation (P.17-SC-220)*)
	ERV_INL4_Fan_Run : BOOL; (*Engine room ventilation inlet air fan - Group 4 in operation (P.17-SC-230)*)
	tERV_INL4_Fan_Run : HALioDi_Type; (*Engine room ventilation inlet air fan - Group 4 in operation (P.17-SC-230)*)
	ERV_INL5_Fan_Run : BOOL; (*Engine room ventilation inlet air fan - Group 5 in operation (P.17-SC-240)*)
	tERV_INL5_Fan_Run : HALioDi_Type; (*Engine room ventilation inlet air fan - Group 5 in operation (P.17-SC-240)*)
	ERV_INL6_Fan_Run : BOOL; (*Engine room ventilation inlet air fan - Group 6 in operation (P.17-SC-250)*)
	tERV_INL6_Fan_Run : HALioDi_Type; (*Engine room ventilation inlet air fan - Group 6 in operation (P.17-SC-250)*)
END_VAR
```
